// TIA Portal V20 export
// export: Created 2025-12-01T14:57:29.98862Z, ExportSetting None, DisplayName Totally Integrated Automation Portal, DisplayVersion V20 Update 3, DisplayName TIA Portal Openness, DisplayVersion V20 Update 3, DisplayName TIA Portal Version Control Interface, DisplayVersion V20 Update 3, DisplayName STEP 7 Professional, DisplayVersion V20 Update 3, DisplayName STEP 7 Safety, DisplayVersion V20 Update 2, DisplayName WinCC Basic/Comfort/Advanced, DisplayVersion V20 Update 3, DisplayName WinCC Professional, DisplayVersion V20 Update 3, DisplayName WinCC Unified, DisplayVersion V20 Update 3
FUNCTION_BLOCK "FB265_M_TL_E01234_S01234"   // FB265, LAD
TITLE = Control del Ramal de Salidas
{ S7_Optimized_Access := 'FALSE' }
AUTHOR : TE_FSS
NAME : 20170822
VERSION : 3.7
// stored: AutoNumber false, SetENOAutomatically false
   VAR_INPUT
      Mesa : UInt;   // Mesa de la FB
      Error_Tx : Bool;   // Error en el Tx
      EnTension : Bool;   // Existe Tension en la Mesa
      Termico_E1_Tx : Bool;   // Proteccion del Tx en E1E3
      Termico_E2_Tx : Bool;   // Proteccion del Tx en E2E4
      pHsMx_Carretilla : Bool;   // pHs de Carretilla
      pHsMx_1 : Bool;   // pHs de la Mesa Mesa (Para Entrada por E3,E2)
      pHsMx_2 : Bool;   // pHs de la Mesa Mesa (Para Entrada por E1,E4)
      pHsMx_Seg_1 : Bool;   // pHs de Protrusion de la Mesa. Nota: No existe >> ON
      pHsMx_Seg_2 : Bool;   // pHs de Protrusion de la Mesa. Nota: No existe >> ON
      Avance_E1_Tx_Ok : Bool;   // Avance del Tx en E1E3
      Avance_E2_Tx_Ok : Bool;   // Avance del Tx en E2E4
      PosTR_E1 : Bool;   // Posicion del TR en E1E3
      PosTR_E2 : Bool;   // Posicion del TR en E2E4
      EnMovimiento_TR : Bool;   // En movimiento el TR
      TP1_UP : Bool;   // TP1 Arriba. Nota Movimiento E1 >> S3
      TP1_DW : Bool;   // TP1 Abajo. Nota Movimiento E1 >> S3
      EnMovimiento_TP1 { ExternalVisible := 'False'} : Bool;   // En movimiento el TP1
      TP2_UP : Bool;   // TP2 Arriba. Nota Movimiento E2 >> S4
      TP2_DW : Bool;   // TP2 Abajo. Nota Movimiento E2 >> S4
      EnMovimiento_TP2 : Bool;   // En movimiento el TP2
      DescargaAct_Ent_M1 : Bool;   // E1 >> Mesa Anterior DescargaAct
      AVTF_Ent_M1 : Bool;   // E1 >> Mesa Anterior AVTF
      P_Mens_Ent_M1 : Bool;   // E1 >> Mesa Anterior P_Mens
      DescargaAct_Ent_M2 : Bool;   // E2 >> Mesa Anterior DescargaAct
      AVTF_Ent_M2 : Bool;   // E2 >> Mesa Anterior AVTF
      P_Mens_Ent_M2 : Bool;   // E2 >> Mesa Anterior P_Mens
      DescargaAct_Ent_M3 : Bool;   // E3 >> Mesa Anterior DescargaAct
      AVTF_Ent_M3 : Bool;   // E3 >> Mesa Anterior AVTF
      P_Mens_Ent_M3 : Bool;   // E3 >> Mesa Anterior P_Mens
      DescargaAct_Ent_M4 : Bool;   // E4 >> Mesa Anterior DescargaAct
      AVTF_Ent_M4 : Bool;   // E4 >> Mesa Anterior AVTF
      P_Mens_Ent_M4 : Bool;   // E4 >> Mesa Anterior P_Mens
      PTF_Sal_M1 : Bool;   // S1 >> Mesa Siguiente PTF
      FTF_Sal_M1 : Bool;   // S1 >> Mesa Siguiente FTF
      PTF_Sal_M2 : Bool;   // S2 >> Mesa Siguiente PTF
      FTF_Sal_M2 : Bool;   // S2 >> Mesa Siguiente FTF
      PTF_Sal_M3 : Bool;   // S3 >> Mesa Siguiente PTF
      FTF_Sal_M3 : Bool;   // S3 >> Mesa Siguiente FTF
      PTF_Sal_M4 : Bool;   // S4 >> Mesa Siguiente PTF
      FTF_Sal_M4 : Bool;   // S4 >> Mesa Siguiente FTF
      MSig_CargaAct_Sal_M1 : Bool;   // S1 >> Mesa Siguiente En Carga
      MSig_CargaAct_Sal_M2 : Bool;   // S2 >> Mesa Siguiente En Carga
      MSig_CargaAct_Sal_M3 : Bool;   // S3 >> Mesa Siguiente En Carga
      MSig_CargaAct_Sal_M4 : Bool;   // S4 >> Mesa Siguiente En Carga
      PosTR_EnReposo_E2 : Bool;   // Posicion de Reposo en E2 para el Transfer
      PosTR_EnReposo_E1 : Bool;   // Posicion de Reposo en E1 para el Transfer
      PermisoMov_PosTR_E2 : Bool;   // Permiso de Mover el Trasnfer hacia E2
      PermisoMov_PosTR_E1 : Bool;   // Permiso de Mover el Trasnfer hacia E1
      Mx_Centraje : Bool;   // Config >> Activar Centraje de Carga
      Mx_UP_E1E3 : Bool;   // Config >> TR Arriba en E1E3
      Mx_TRElectrico : Bool;   // Config >> Mesa con Transfer Electrico
      Mx_VelocidadLenta_In : Bool;   // Forzar a Velociada Lenta
      F_EnvMens_Mx : Bool;   // Fin de Envio de Mensaje
      OrdSal_M1 : Bool;   // Orden de Salida por S1
      OrdSal_M2 : Bool;   // Orden de Salida por S2
      OrdSal_M3 : Bool;   // Orden de Salida por S3
      OrdSal_M4 : Bool;   // Orden de Salida por S4
      OrdSal_Retirar : Bool;   // Orden de Salida por S0
      BloqueoActivo_OK : Bool;   // Bloqueo Activo de la Mesa
      V_CNT_pHsMx_E1 : Int := 400;   // Valor de Presencia
      V_CNT_pHsMx_FTF_E1 : Int := 200;   // Valor para activar FTF. Nota: < = V_CNT_pHsMx.
      V_CNTSeg_pHsMx_E1 : Int := 2000;   // Valor de Seguriadad para Presencia
      V_CNT_pHsMx_E2 : Int := 400;   // Valor de Presencia
      V_CNT_pHsMx_FTF_E2 : Int := 200;   // Valor para activar FTF. Nota: < = V_CNT_pHsMx.
      V_CNTSeg_pHsMx_E2 : Int := 2000;   // Valor de Seguriadad para Presencia
      V_Subir_TP_Min : Int := 20;   // Valor Minimo para Subir Tope
      V_Bajar_TP_Max : Int := 40;   // Valor Maximo para Bajar Tope
      V_CNT_ApHsMx : Int := 500;   // Valor de Ausencia
      V_CNTSeg_ApHsMx : Int := 2000;   // Valor de Seguriadad para Ausencia
      V_TIM_Bloqueo : Int := 3000;   // Valor del Tiempo de Espera para Bloqueo
      V_TIM_Entrada : Int := 5000;   // Valor de Entrada de Carga >> E0
      V_TIM_Retirar : Int := 5000;   // Valor de Retirada de Carga >> S0
      V_CNT_Centrado : Int := 2000;   // Valor de Centrado de Carga
      V_CNT_Reposo : Int := 500;   // Valor de Reposo de Carga Nota: > Centrado
      V_CNT_Simultaneo : Int := 2000;   // Valor de Simultaneo
      V_InicioSimultaneo : Int := 0;   // Inicio de Simultaneo. Nota: <= V_CNT_Simultaneo
      V_FinSimultaneo : Int := 0;   // Final de Simultaneo. Nota: <= V_InicioSimultaneo
      V_TOut_Tx_Mx_E1 : Int := 10000;   // TimeOut de Entrada por E1
      V_TOut_Tx_Mx_E2 : Int := 10000;   // TimeOut de Entrada por E2
      V_TOut_TR : Int := 5000;   // TimeOut de Transfer
      V_TOut_TP : Int := 5000;   // TimeOut de Tope
      V_TMP_Protrusion : Int := 200;   // TMP de Protrusion
      V_CNT_PerdidapHs : Int := 10;   // CNT de Perdida de pHs
   END_VAR
   VAR_OUTPUT
      P_EnvMens_PMx : Bool;   // Permiso de Enviar Mensaje de Presencia
      P_EnvMens_PBM : Bool;   // Permiso de Enviar Mensaje de Bloqueo
      P_EnvMens_AMx : Bool;   // Permiso de Enviar Mensaje de Ausencia
      P_RecepOK_Mx : Bool;   // Recepcion OK
      PTF_Ent_M1 : Bool;   // E1 >> Mesa Anterior PTF
      FTF_Ent_M1 : Bool;   // E1 >> Mesa Anterior FTF
      PTF_Ent_M2 : Bool;   // E2 >> Mesa Anterior PTF
      FTF_Ent_M2 : Bool;   // E2 >> Mesa Anterior FTF
      PTF_Ent_M3 : Bool;   // E3 >> Mesa Anterior PTF
      FTF_Ent_M3 : Bool;   // E3 >> Mesa Anterior FTF
      PTF_Ent_M4 : Bool;   // E4 >> Mesa Anterior PTF
      FTF_Ent_M4 : Bool;   // E4 >> Mesa Anterior FTF
      AVTF_Sal_M1 : Bool;   // S1 >> Mesa Siguiente AVTF
      P_Mens_Sal_M1 : Bool;   // S1 >> Mesa Siguiente P_Mens
      AVTF_Sal_M2 : Bool;   // S2 >> Mesa Siguiente AVTF
      P_Mens_Sal_M2 : Bool;   // S2 >> Mesa Siguiente P_Mens
      AVTF_Sal_M3 : Bool;   // S3 >> Mesa Siguiente AVTF
      P_Mens_Sal_M3 : Bool;   // S3 >> Mesa Siguiente P_Mens
      AVTF_Sal_M4 : Bool;   // S4 >> Mesa Siguiente AVTF
      P_Mens_Sal_M4 : Bool;   // S4 >> Mesa Siguiente P_Mens
   END_VAR
   VAR
      Anular_prE1 : Bool;   // ???
      Anular_prS3 : Bool;   // ???
      Mx_ET00 : Bool;
      Mx_ET01 : Bool;
      Mx_ET02 : Bool;
      Mx_ET08 : Bool;
      Mx_ET09 : Bool;
      Mx_ET10 : Bool;
      Mx_ET11 : Bool;
      Mx_ET12 : Bool;
      Mx_ET110 : Bool;
      Mx_ET111 : Bool;
      Mx_ET20 : Bool;
      Mx_ET21 : Bool;
      Mx_ET22 : Bool;
      Mx_ET120 : Bool;
      Mx_ET121 : Bool;
      Mx_ET40 : Bool;
      Mx_ET41 : Bool;
      Mx_ET42 : Bool;
      Mx_ET43 : Bool;
      Mx_ET140 : Bool;
      Mx_ET141 : Bool;
      Mx_ET50 : Bool;
      Mx_ET51 : Bool;
      Mx_ET150 : Bool;
      Mx_ET151 : Bool;
      Mx_ET60 : Bool;
      Mx_ET61 : Bool;
      Mx_ET160 : Bool;
      Mx_ET161 : Bool;
      Mx_ET180 : Bool;
      Mx_ET181 : Bool;
      Mx_ET90 : Bool;
      Mx_ET91 : Bool;
      Mx_ET190 : Bool;
      Mx_ET191 : Bool;
      Mx_ET192 : Bool;
      Selec_M1_Entrada : Bool;   // Seleccionado Entrada por E1
      Selec_M1_Salida : Bool;   // Seleccionado Entrada por E2
      Selec_M2_Entrada : Bool;   // Seleccionado Entrada por E3
      Selec_M2_Salida : Bool;   // Seleccionado Entrada por E4
      Selec_M3_Entrada : Bool;   // Seleccionado Salida por S1
      Selec_M3_Salida : Bool;   // Seleccionado Salida por S2
      Selec_M4_Entrada : Bool;   // Seleccionado Salida por S3
      Selec_M4_Salida : Bool;   // Seleccionado Salida por S4
      Selec_Retirar : Bool;   // Seleccionado Retirar
      MEnt_DescargaAct : Bool;   // Interlock >> DesCargaAct de MAnt >> Mx
      ATF_MEnt : Bool;   // Interlock >> AVTF de MAnt >> Mx
      P_Mens_MEnt : Bool;   // Interlock >> P_Mens de MAnt >> Mx
      PTF_MEnt : Bool;   // Interlock >> PTF de MAnt >> Mx
      FTF_MEnt : Bool;   // Interlock >> FTF de MAnt >> Mx
      ATF_MSal : Bool;   // Interlock >> AVTF de Mx >> MSig
      P_Mens_MSal { ExternalAccessible := 'False'; ExternalVisible := 'False'; ExternalWritable := 'False'} : Bool;   // Interlock >> P_Mens de Mx >> MSig
      PTF_MSal : Bool;   // Interlock >> PTF de Mx >> MSig
      FTF_MSal : Bool;   // Interlock >> FTF de Mx >> MSig
      ProtocoloIniciado_Mx : Bool;   // Iniciado el Envio del Mensaje de Presencia
      Simultaneo_Mx : Bool;   // Activo Simultaneo E1E2E3E4
      SaliendoCarga : Bool;   // Saliendo Carga de la Mesa
      CNT_pHsMx_FTF_OK_E1E3 : Bool;   // Enviar ya FTF
      CNT_pHsMx_FTF_OK_E2E4 : Bool;   // Enviar ya FTF
      CNT_pHsMx_E1E3 { S7_SetPoint := 'True'} : "FB910_CNT_UHS";   // CNT de la Presencia
      CNTSeg_pHsMx_E1E3 { S7_SetPoint := 'True'} : "FB910_CNT_UHS";   // CNT de Seguridad de la Presencia
      CNT_pHsMx_E2E4 { S7_SetPoint := 'True'} : "FB910_CNT_UHS";   // CNT de la Presencia
      CNTSeg_pHsMx_E2E4 { S7_SetPoint := 'True'} : "FB910_CNT_UHS";   // CNT de Seguridad de la Presencia
      CNT_ApHsMx { S7_SetPoint := 'True'} : "FB910_CNT_UHS";   // CNT de la Ausencia
      CNTSeg_ApHsMx { S7_SetPoint := 'True'} : "FB910_CNT_UHS";   // CNT de Seguridad de la Ausencia
      TIM_Bloqueo { S7_SetPoint := 'True'} : "FB910_CNT_UHS";   // TIM de Espera para Bloqueo
      TMP_Entrada { S7_SetPoint := 'True'} : "FB910_CNT_UHS";   // TMP de Entrada de Carga
      TMP_Retirar { S7_SetPoint := 'True'} : "FB910_CNT_UHS";   // TMP de Retirada de Carga
      CNT_Centrado { S7_SetPoint := 'True'} : "FB910_CNT_UHS";   // Contador de Centrado de Carga
      CNT_Simultaneo { S7_SetPoint := 'True'} : "FB910_CNT_UHS";   // CNT de Simultaneo
      TMP_EnTension { S7_SetPoint := 'True'} : "FB910_CNT_UHS";
      TOut_Av_Mx_E1E3 { S7_SetPoint := 'True'} : "FB910_CNT_UHS";   // Time Out de Entrada de E1
      TOut_Ret_Mx_E1E3 { S7_SetPoint := 'True'} : "FB910_CNT_UHS";   // Time Out de Entrada de E3
      TOut_Av_Mx_E2E4 { S7_SetPoint := 'True'} : "FB910_CNT_UHS";   // Time Out de Entrada de E2
      TOut_Ret_Mx_E2E4 { S7_SetPoint := 'True'} : "FB910_CNT_UHS";   // Time Out de Entrada de E4
      TOut_Subir_TR { S7_SetPoint := 'True'} : "FB910_CNT_UHS";   // Time Out de Subida del TR
      TOut_Bajar_TR { S7_SetPoint := 'True'} : "FB910_CNT_UHS";   // Time Out de Bajada del TR
      TOut_Subir_Tp { S7_SetPoint := 'True'} : "FB910_CNT_UHS";   // Time Out de Subida del TP
      TOut_Bajar_Tp { S7_SetPoint := 'True'} : "FB910_CNT_UHS";   // Time Out de Bajada del TP
      TMP_Protrusion { S7_SetPoint := 'True'} : "FB910_CNT_UHS";   // TMP de la Protrusion
      CNT_PerdidapHs { S7_SetPoint := 'True'} : "FB910_CNT_UHS";   // CNT de Perdida de pHs
      STAT_EnvMens_PMx : Bool;   // Interna >> Envio del Mensaje de Presencia
      STAT_EnvMens_AMx : Bool;   // Interna >> Envio del Mensaje de Ausencia
      STAT_EnvMens_PBMx : Bool;   // Interna >> Envio del Mensaje de Bloqueo
   END_VAR
   VAR_TEMP
      EstadoZona : "EstadoZona";   // Estado de Zona de la Mesa
      EstadoVI : "EstadosMesa";   // Estado del Vehiculo Inteliguente de la Mesa
      ConfigFB : "UDT_ConfigFB";   // Configuracion de la FB de la Mesa
      V_Protrusion : Int;
      Aux_ET00 : Bool;
      Pos_TR_OK : Bool;
      OK_TP1_DW : Bool;
      OK_TP2_DW : Bool;
   END_VAR
   VAR_TEMP   // added for the SCL form of the ladder/FBD networks
      _w1 : Bool;
      _w2 : Bool;
      _w3 : Bool;
      _w4 : Bool;
   END_VAR
BEGIN

REGION Network 1: INICIALIZAR - Recoger las Variables de Estado de la Mesa
   // Se recoge - Estado_CBx
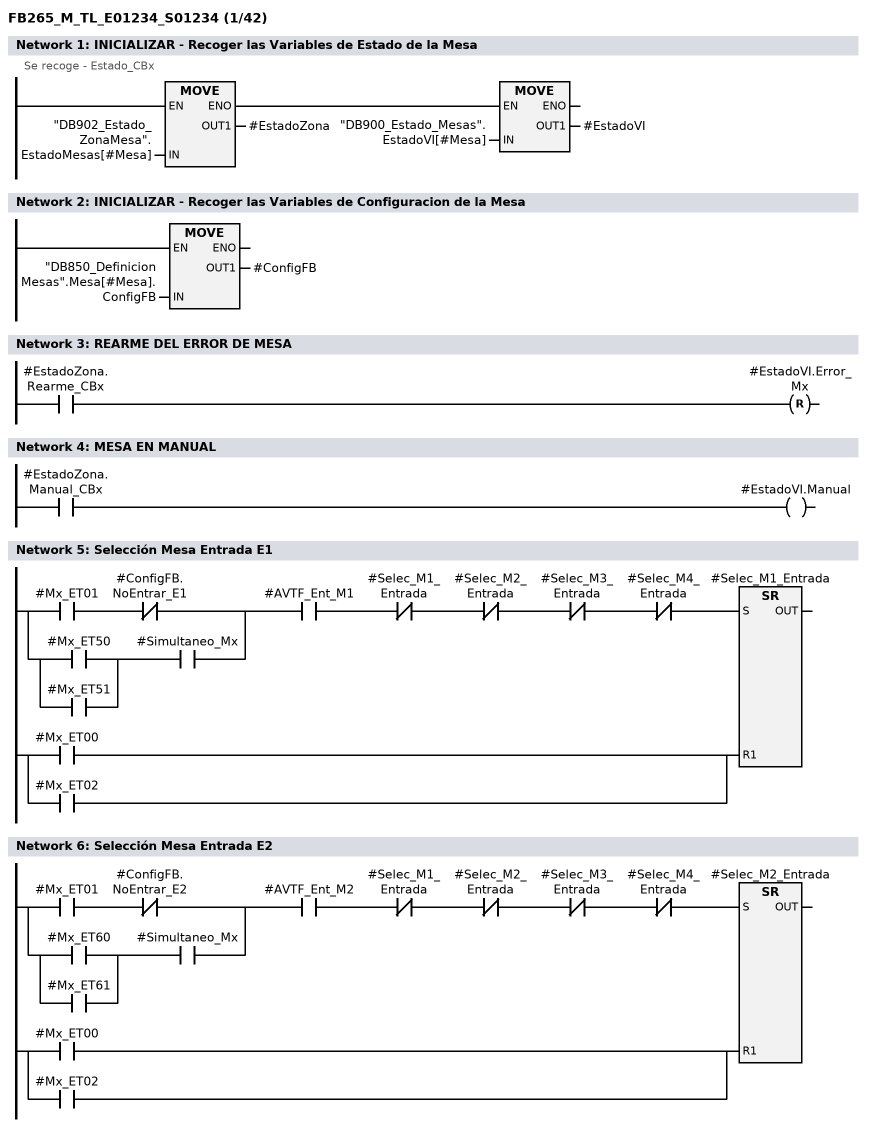
   RUNG wire#powerrail
      Move(in := "DB902_Estado_ZonaMesa".EstadoMesas[#Mesa], out1 => #EstadoZona)
      Move(in := "DB900_Estado_Mesas".EstadoVI[#Mesa], out1 => #EstadoVI)
   END_RUNG
   // the same network as SCL:
   #EstadoZona := "DB902_Estado_ZonaMesa".EstadoMesas[#Mesa];
   #EstadoVI := "DB900_Estado_Mesas".EstadoVI[#Mesa];
END_REGION

REGION Network 2: INICIALIZAR - Recoger las Variables de Configuracion de la Mesa
   RUNG wire#powerrail
      Move(in := "DB850_DefinicionMesas".Mesa[#Mesa].ConfigFB, out1 => #ConfigFB)
   END_RUNG
   // the same network as SCL:
   #ConfigFB := "DB850_DefinicionMesas".Mesa[#Mesa].ConfigFB;
END_REGION

REGION Network 3: REARME DEL ERROR DE MESA
   RUNG wire#powerrail
      Contact( #EstadoZona.Rearme_CBx )
      R_Coil( #EstadoVI.Error_Mx )
   END_RUNG
   // the same network as SCL:
   IF #EstadoZona.Rearme_CBx THEN #EstadoVI.Error_Mx := FALSE; END_IF;
END_REGION

REGION Network 4: MESA EN MANUAL
   RUNG wire#powerrail
      Contact( #EstadoZona.Manual_CBx )
      Coil( #EstadoVI.Manual )
   END_RUNG
   // the same network as SCL:
   #EstadoVI.Manual := #EstadoZona.Manual_CBx;
END_REGION

REGION Network 5: Selección Mesa Entrada E1
   RUNG wire#powerrail
      Contact( #Mx_ET01 )
      I_Contact( #ConfigFB.NoEntrar_E1 )
      wire#w1
      Contact( #AVTF_Ent_M1 )
      I_Contact( #Selec_M1_Entrada )
      I_Contact( #Selec_M2_Entrada )
      I_Contact( #Selec_M3_Entrada )
      I_Contact( #Selec_M4_Entrada )
      S_SR(operand := #Selec_M1_Entrada, r1 := wire#w3)
   END_RUNG
   RUNG wire#powerrail
      Contact( #Mx_ET50 )
      wire#w2
      Contact( #Simultaneo_Mx )
   END_RUNG wire#w1
   RUNG wire#powerrail
      Contact( #Mx_ET51 )
   END_RUNG wire#w2
   RUNG wire#powerrail
      Contact( #Mx_ET00 )
   END_RUNG wire#w3
   RUNG wire#powerrail
      Contact( #Mx_ET02 )
   END_RUNG wire#w3
   // the same network as SCL:
   IF ((#Mx_ET01 AND NOT #ConfigFB.NoEntrar_E1) OR ((#Mx_ET50 OR #Mx_ET51) AND #Simultaneo_Mx)) AND #AVTF_Ent_M1 AND NOT #Selec_M1_Entrada AND NOT #Selec_M2_Entrada AND NOT #Selec_M3_Entrada AND NOT #Selec_M4_Entrada THEN
       #Selec_M1_Entrada := TRUE;   // SR flip-flop
   END_IF;
   IF #Mx_ET00 OR #Mx_ET02 THEN #Selec_M1_Entrada := FALSE; END_IF;
END_REGION

REGION Network 6: Selección Mesa Entrada E2
   RUNG wire#powerrail
      Contact( #Mx_ET01 )
      I_Contact( #ConfigFB.NoEntrar_E2 )
      wire#w1
      Contact( #AVTF_Ent_M2 )
      I_Contact( #Selec_M1_Entrada )
      I_Contact( #Selec_M2_Entrada )
      I_Contact( #Selec_M3_Entrada )
      I_Contact( #Selec_M4_Entrada )
      S_SR(operand := #Selec_M2_Entrada, r1 := wire#w3)
   END_RUNG
   RUNG wire#powerrail
      Contact( #Mx_ET60 )
      wire#w2
      Contact( #Simultaneo_Mx )
   END_RUNG wire#w1
   RUNG wire#powerrail
      Contact( #Mx_ET61 )
   END_RUNG wire#w2
   RUNG wire#powerrail
      Contact( #Mx_ET00 )
   END_RUNG wire#w3
   RUNG wire#powerrail
      Contact( #Mx_ET02 )
   END_RUNG wire#w3
   // the same network as SCL:
   IF ((#Mx_ET01 AND NOT #ConfigFB.NoEntrar_E2) OR ((#Mx_ET60 OR #Mx_ET61) AND #Simultaneo_Mx)) AND #AVTF_Ent_M2 AND NOT #Selec_M1_Entrada AND NOT #Selec_M2_Entrada AND NOT #Selec_M3_Entrada AND NOT #Selec_M4_Entrada THEN
       #Selec_M2_Entrada := TRUE;   // SR flip-flop
   END_IF;
   IF #Mx_ET00 OR #Mx_ET02 THEN #Selec_M2_Entrada := FALSE; END_IF;
END_REGION

REGION Network 7: Selección Mesa Entrada E3
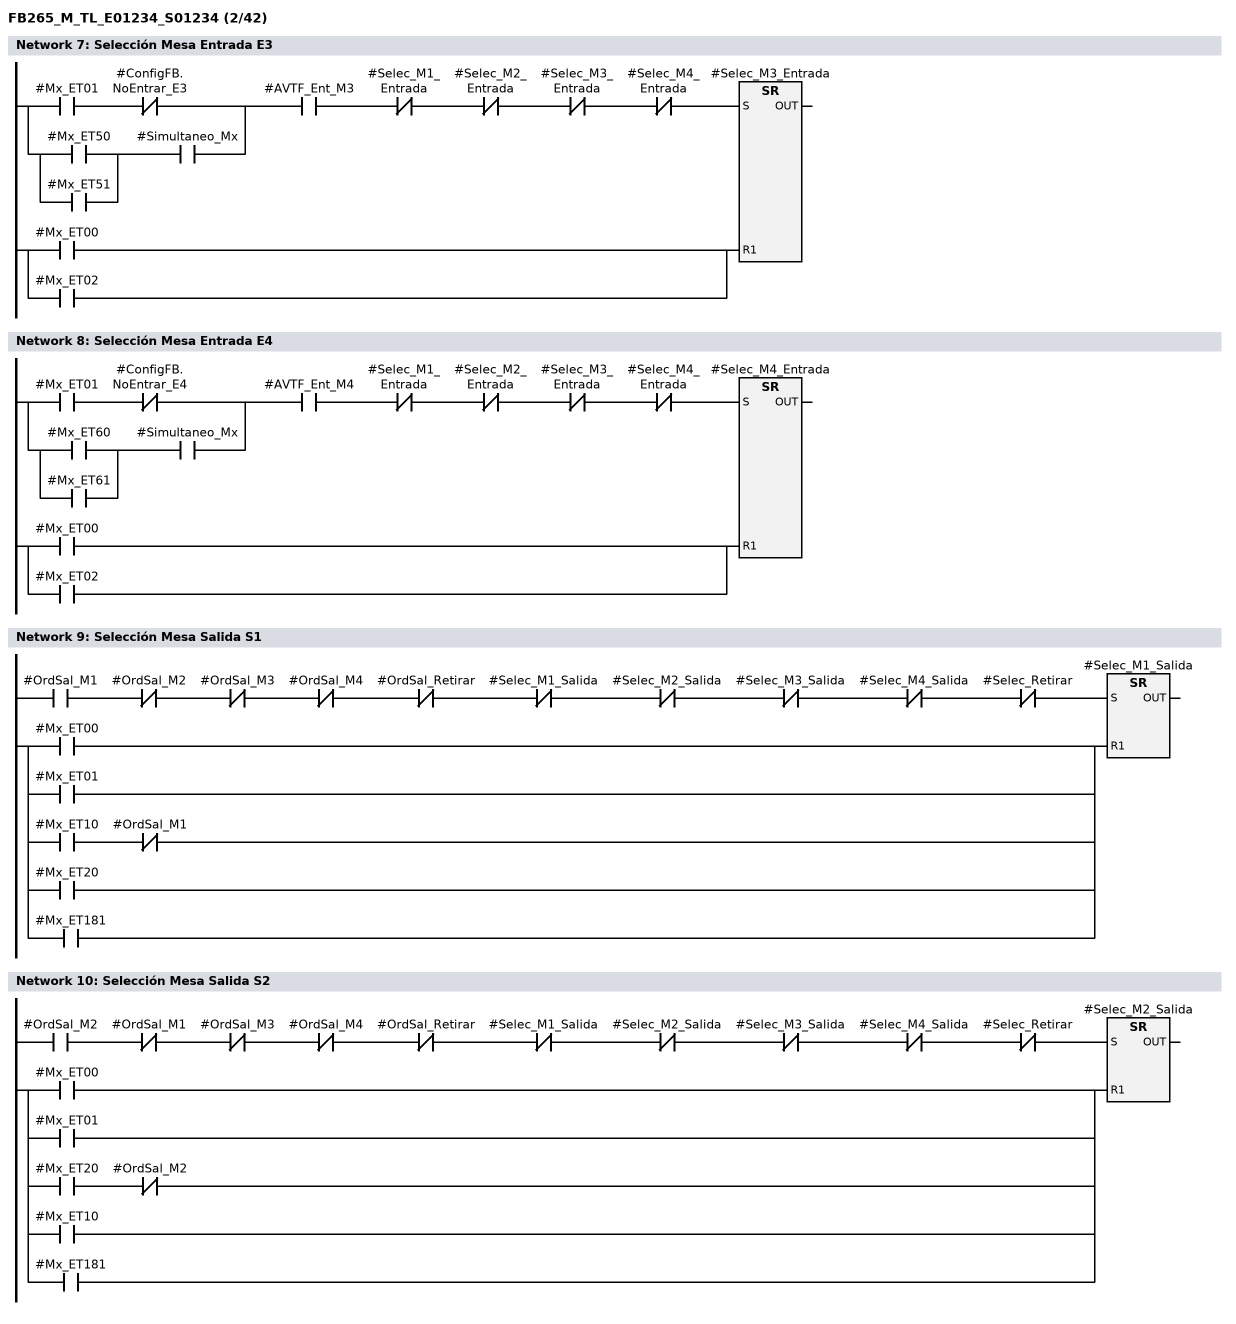
   RUNG wire#powerrail
      Contact( #Mx_ET01 )
      I_Contact( #ConfigFB.NoEntrar_E3 )
      wire#w1
      Contact( #AVTF_Ent_M3 )
      I_Contact( #Selec_M1_Entrada )
      I_Contact( #Selec_M2_Entrada )
      I_Contact( #Selec_M3_Entrada )
      I_Contact( #Selec_M4_Entrada )
      S_SR(operand := #Selec_M3_Entrada, r1 := wire#w3)
   END_RUNG
   RUNG wire#powerrail
      Contact( #Mx_ET50 )
      wire#w2
      Contact( #Simultaneo_Mx )
   END_RUNG wire#w1
   RUNG wire#powerrail
      Contact( #Mx_ET51 )
   END_RUNG wire#w2
   RUNG wire#powerrail
      Contact( #Mx_ET00 )
   END_RUNG wire#w3
   RUNG wire#powerrail
      Contact( #Mx_ET02 )
   END_RUNG wire#w3
   // the same network as SCL:
   IF ((#Mx_ET01 AND NOT #ConfigFB.NoEntrar_E3) OR ((#Mx_ET50 OR #Mx_ET51) AND #Simultaneo_Mx)) AND #AVTF_Ent_M3 AND NOT #Selec_M1_Entrada AND NOT #Selec_M2_Entrada AND NOT #Selec_M3_Entrada AND NOT #Selec_M4_Entrada THEN
       #Selec_M3_Entrada := TRUE;   // SR flip-flop
   END_IF;
   IF #Mx_ET00 OR #Mx_ET02 THEN #Selec_M3_Entrada := FALSE; END_IF;
END_REGION

REGION Network 8: Selección Mesa Entrada E4
   RUNG wire#powerrail
      Contact( #Mx_ET01 )
      I_Contact( #ConfigFB.NoEntrar_E4 )
      wire#w1
      Contact( #AVTF_Ent_M4 )
      I_Contact( #Selec_M1_Entrada )
      I_Contact( #Selec_M2_Entrada )
      I_Contact( #Selec_M3_Entrada )
      I_Contact( #Selec_M4_Entrada )
      S_SR(operand := #Selec_M4_Entrada, r1 := wire#w3)
   END_RUNG
   RUNG wire#powerrail
      Contact( #Mx_ET60 )
      wire#w2
      Contact( #Simultaneo_Mx )
   END_RUNG wire#w1
   RUNG wire#powerrail
      Contact( #Mx_ET61 )
   END_RUNG wire#w2
   RUNG wire#powerrail
      Contact( #Mx_ET00 )
   END_RUNG wire#w3
   RUNG wire#powerrail
      Contact( #Mx_ET02 )
   END_RUNG wire#w3
   // the same network as SCL:
   IF ((#Mx_ET01 AND NOT #ConfigFB.NoEntrar_E4) OR ((#Mx_ET60 OR #Mx_ET61) AND #Simultaneo_Mx)) AND #AVTF_Ent_M4 AND NOT #Selec_M1_Entrada AND NOT #Selec_M2_Entrada AND NOT #Selec_M3_Entrada AND NOT #Selec_M4_Entrada THEN
       #Selec_M4_Entrada := TRUE;   // SR flip-flop
   END_IF;
   IF #Mx_ET00 OR #Mx_ET02 THEN #Selec_M4_Entrada := FALSE; END_IF;
END_REGION

REGION Network 9: Selección Mesa Salida S1
   RUNG wire#powerrail
      Contact( #OrdSal_M1 )
      I_Contact( #OrdSal_M2 )
      I_Contact( #OrdSal_M3 )
      I_Contact( #OrdSal_M4 )
      I_Contact( #OrdSal_Retirar )
      I_Contact( #Selec_M1_Salida )
      I_Contact( #Selec_M2_Salida )
      I_Contact( #Selec_M3_Salida )
      I_Contact( #Selec_M4_Salida )
      I_Contact( #Selec_Retirar )
      S_SR(operand := #Selec_M1_Salida, r1 := wire#w1)
   END_RUNG
   RUNG wire#powerrail
      Contact( #Mx_ET00 )
   END_RUNG wire#w1
   RUNG wire#powerrail
      Contact( #Mx_ET01 )
   END_RUNG wire#w1
   RUNG wire#powerrail
      Contact( #Mx_ET10 )
      I_Contact( #OrdSal_M1 )
   END_RUNG wire#w1
   RUNG wire#powerrail
      Contact( #Mx_ET20 )
   END_RUNG wire#w1
   RUNG wire#powerrail
      Contact( #Mx_ET181 )
   END_RUNG wire#w1
   // the same network as SCL:
   IF #OrdSal_M1 AND NOT #OrdSal_M2 AND NOT #OrdSal_M3 AND NOT #OrdSal_M4 AND NOT #OrdSal_Retirar AND NOT #Selec_M1_Salida AND NOT #Selec_M2_Salida AND NOT #Selec_M3_Salida AND NOT #Selec_M4_Salida AND NOT #Selec_Retirar THEN
       #Selec_M1_Salida := TRUE;   // SR flip-flop
   END_IF;
   IF #Mx_ET00 OR #Mx_ET01 OR (#Mx_ET10 AND NOT #OrdSal_M1) OR #Mx_ET20 OR #Mx_ET181 THEN
       #Selec_M1_Salida := FALSE;
   END_IF;
END_REGION

REGION Network 10: Selección Mesa Salida S2
   RUNG wire#powerrail
      Contact( #OrdSal_M2 )
      I_Contact( #OrdSal_M1 )
      I_Contact( #OrdSal_M3 )
      I_Contact( #OrdSal_M4 )
      I_Contact( #OrdSal_Retirar )
      I_Contact( #Selec_M1_Salida )
      I_Contact( #Selec_M2_Salida )
      I_Contact( #Selec_M3_Salida )
      I_Contact( #Selec_M4_Salida )
      I_Contact( #Selec_Retirar )
      S_SR(operand := #Selec_M2_Salida, r1 := wire#w1)
   END_RUNG
   RUNG wire#powerrail
      Contact( #Mx_ET00 )
   END_RUNG wire#w1
   RUNG wire#powerrail
      Contact( #Mx_ET01 )
   END_RUNG wire#w1
   RUNG wire#powerrail
      Contact( #Mx_ET20 )
      I_Contact( #OrdSal_M2 )
   END_RUNG wire#w1
   RUNG wire#powerrail
      Contact( #Mx_ET10 )
   END_RUNG wire#w1
   RUNG wire#powerrail
      Contact( #Mx_ET181 )
   END_RUNG wire#w1
   // the same network as SCL:
   IF #OrdSal_M2 AND NOT #OrdSal_M1 AND NOT #OrdSal_M3 AND NOT #OrdSal_M4 AND NOT #OrdSal_Retirar AND NOT #Selec_M1_Salida AND NOT #Selec_M2_Salida AND NOT #Selec_M3_Salida AND NOT #Selec_M4_Salida AND NOT #Selec_Retirar THEN
       #Selec_M2_Salida := TRUE;   // SR flip-flop
   END_IF;
   IF #Mx_ET00 OR #Mx_ET01 OR (#Mx_ET20 AND NOT #OrdSal_M2) OR #Mx_ET10 OR #Mx_ET181 THEN
       #Selec_M2_Salida := FALSE;
   END_IF;
END_REGION

REGION Network 11: Selección Mesa Salida S3
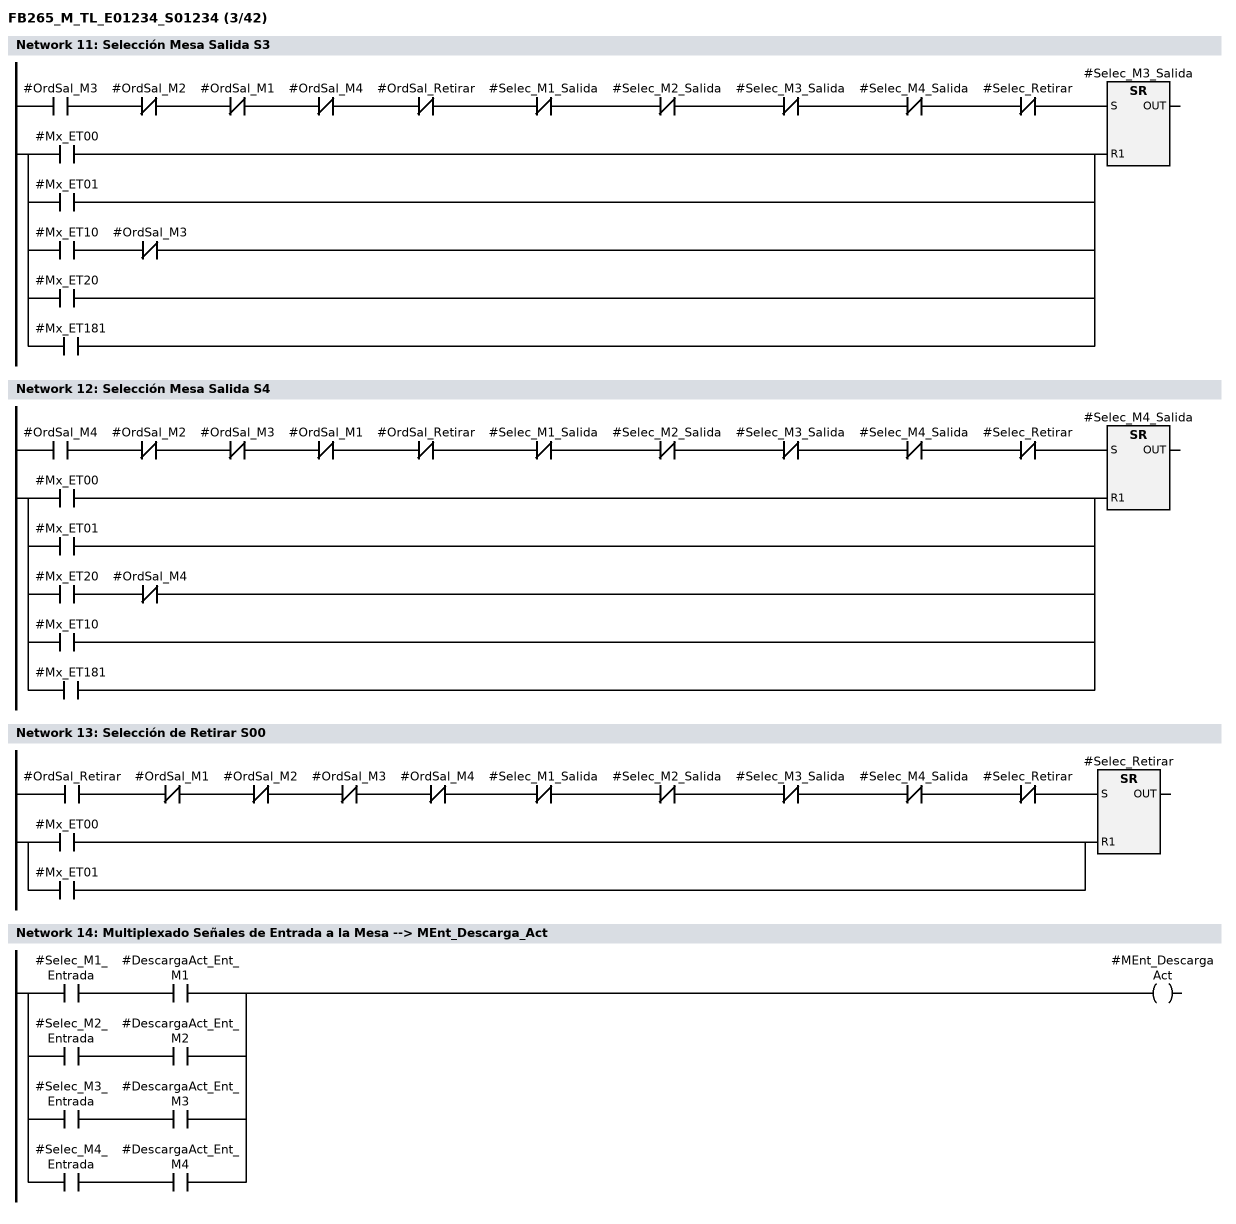
   RUNG wire#powerrail
      Contact( #OrdSal_M3 )
      I_Contact( #OrdSal_M2 )
      I_Contact( #OrdSal_M1 )
      I_Contact( #OrdSal_M4 )
      I_Contact( #OrdSal_Retirar )
      I_Contact( #Selec_M1_Salida )
      I_Contact( #Selec_M2_Salida )
      I_Contact( #Selec_M3_Salida )
      I_Contact( #Selec_M4_Salida )
      I_Contact( #Selec_Retirar )
      S_SR(operand := #Selec_M3_Salida, r1 := wire#w1)
   END_RUNG
   RUNG wire#powerrail
      Contact( #Mx_ET00 )
   END_RUNG wire#w1
   RUNG wire#powerrail
      Contact( #Mx_ET01 )
   END_RUNG wire#w1
   RUNG wire#powerrail
      Contact( #Mx_ET10 )
      I_Contact( #OrdSal_M3 )
   END_RUNG wire#w1
   RUNG wire#powerrail
      Contact( #Mx_ET20 )
   END_RUNG wire#w1
   RUNG wire#powerrail
      Contact( #Mx_ET181 )
   END_RUNG wire#w1
   // the same network as SCL:
   IF #OrdSal_M3 AND NOT #OrdSal_M2 AND NOT #OrdSal_M1 AND NOT #OrdSal_M4 AND NOT #OrdSal_Retirar AND NOT #Selec_M1_Salida AND NOT #Selec_M2_Salida AND NOT #Selec_M3_Salida AND NOT #Selec_M4_Salida AND NOT #Selec_Retirar THEN
       #Selec_M3_Salida := TRUE;   // SR flip-flop
   END_IF;
   IF #Mx_ET00 OR #Mx_ET01 OR (#Mx_ET10 AND NOT #OrdSal_M3) OR #Mx_ET20 OR #Mx_ET181 THEN
       #Selec_M3_Salida := FALSE;
   END_IF;
END_REGION

REGION Network 12: Selección Mesa Salida S4
   RUNG wire#powerrail
      Contact( #OrdSal_M4 )
      I_Contact( #OrdSal_M2 )
      I_Contact( #OrdSal_M3 )
      I_Contact( #OrdSal_M1 )
      I_Contact( #OrdSal_Retirar )
      I_Contact( #Selec_M1_Salida )
      I_Contact( #Selec_M2_Salida )
      I_Contact( #Selec_M3_Salida )
      I_Contact( #Selec_M4_Salida )
      I_Contact( #Selec_Retirar )
      S_SR(operand := #Selec_M4_Salida, r1 := wire#w1)
   END_RUNG
   RUNG wire#powerrail
      Contact( #Mx_ET00 )
   END_RUNG wire#w1
   RUNG wire#powerrail
      Contact( #Mx_ET01 )
   END_RUNG wire#w1
   RUNG wire#powerrail
      Contact( #Mx_ET20 )
      I_Contact( #OrdSal_M4 )
   END_RUNG wire#w1
   RUNG wire#powerrail
      Contact( #Mx_ET10 )
   END_RUNG wire#w1
   RUNG wire#powerrail
      Contact( #Mx_ET181 )
   END_RUNG wire#w1
   // the same network as SCL:
   IF #OrdSal_M4 AND NOT #OrdSal_M2 AND NOT #OrdSal_M3 AND NOT #OrdSal_M1 AND NOT #OrdSal_Retirar AND NOT #Selec_M1_Salida AND NOT #Selec_M2_Salida AND NOT #Selec_M3_Salida AND NOT #Selec_M4_Salida AND NOT #Selec_Retirar THEN
       #Selec_M4_Salida := TRUE;   // SR flip-flop
   END_IF;
   IF #Mx_ET00 OR #Mx_ET01 OR (#Mx_ET20 AND NOT #OrdSal_M4) OR #Mx_ET10 OR #Mx_ET181 THEN
       #Selec_M4_Salida := FALSE;
   END_IF;
END_REGION

REGION Network 13: Selección de Retirar S00
   RUNG wire#powerrail
      Contact( #OrdSal_Retirar )
      I_Contact( #OrdSal_M1 )
      I_Contact( #OrdSal_M2 )
      I_Contact( #OrdSal_M3 )
      I_Contact( #OrdSal_M4 )
      I_Contact( #Selec_M1_Salida )
      I_Contact( #Selec_M2_Salida )
      I_Contact( #Selec_M3_Salida )
      I_Contact( #Selec_M4_Salida )
      I_Contact( #Selec_Retirar )
      S_SR(operand := #Selec_Retirar, r1 := wire#w1)
   END_RUNG
   RUNG wire#powerrail
      Contact( #Mx_ET00 )
   END_RUNG wire#w1
   RUNG wire#powerrail
      Contact( #Mx_ET01 )
   END_RUNG wire#w1
   // the same network as SCL:
   IF #OrdSal_Retirar AND NOT #OrdSal_M1 AND NOT #OrdSal_M2 AND NOT #OrdSal_M3 AND NOT #OrdSal_M4 AND NOT #Selec_M1_Salida AND NOT #Selec_M2_Salida AND NOT #Selec_M3_Salida AND NOT #Selec_M4_Salida AND NOT #Selec_Retirar THEN
       #Selec_Retirar := TRUE;   // SR flip-flop
   END_IF;
   IF #Mx_ET00 OR #Mx_ET01 THEN #Selec_Retirar := FALSE; END_IF;
END_REGION

REGION Network 14: Multiplexado Señales de Entrada a la Mesa --> MEnt_Descarga_Act
   RUNG wire#powerrail
      Contact( #Selec_M1_Entrada )
      Contact( #DescargaAct_Ent_M1 )
      wire#w1
      Coil( #MEnt_DescargaAct )
   END_RUNG
   RUNG wire#powerrail
      Contact( #Selec_M2_Entrada )
      Contact( #DescargaAct_Ent_M2 )
   END_RUNG wire#w1
   RUNG wire#powerrail
      Contact( #Selec_M3_Entrada )
      Contact( #DescargaAct_Ent_M3 )
   END_RUNG wire#w1
   RUNG wire#powerrail
      Contact( #Selec_M4_Entrada )
      Contact( #DescargaAct_Ent_M4 )
   END_RUNG wire#w1
   // the same network as SCL:
   #MEnt_DescargaAct := (#Selec_M1_Entrada AND #DescargaAct_Ent_M1) OR (#Selec_M2_Entrada AND #DescargaAct_Ent_M2) OR (#Selec_M3_Entrada AND #DescargaAct_Ent_M3) OR (#Selec_M4_Entrada AND #DescargaAct_Ent_M4);
END_REGION

REGION Network 15: Multiplexado Señales de Entrada a la Mesa --> AVTF
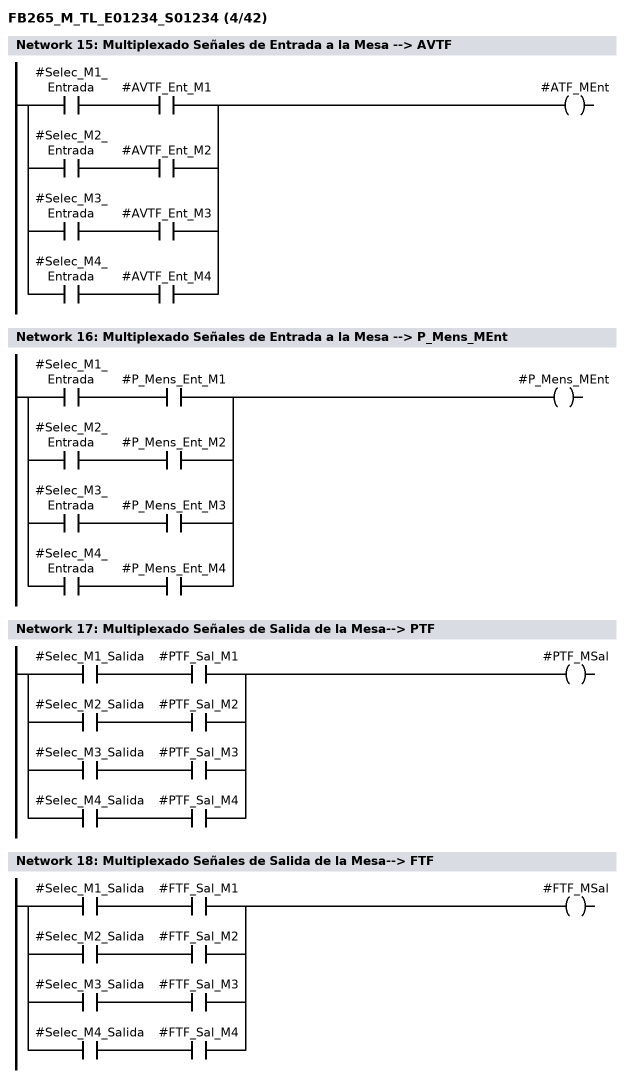
   RUNG wire#powerrail
      Contact( #Selec_M1_Entrada )
      Contact( #AVTF_Ent_M1 )
      wire#w1
      Coil( #ATF_MEnt )
   END_RUNG
   RUNG wire#powerrail
      Contact( #Selec_M2_Entrada )
      Contact( #AVTF_Ent_M2 )
   END_RUNG wire#w1
   RUNG wire#powerrail
      Contact( #Selec_M3_Entrada )
      Contact( #AVTF_Ent_M3 )
   END_RUNG wire#w1
   RUNG wire#powerrail
      Contact( #Selec_M4_Entrada )
      Contact( #AVTF_Ent_M4 )
   END_RUNG wire#w1
   // the same network as SCL:
   #ATF_MEnt := (#Selec_M1_Entrada AND #AVTF_Ent_M1) OR (#Selec_M2_Entrada AND #AVTF_Ent_M2) OR (#Selec_M3_Entrada AND #AVTF_Ent_M3) OR (#Selec_M4_Entrada AND #AVTF_Ent_M4);
END_REGION

REGION Network 16: Multiplexado Señales de Entrada a la Mesa --> P_Mens_MEnt
   RUNG wire#powerrail
      Contact( #Selec_M1_Entrada )
      Contact( #P_Mens_Ent_M1 )
      wire#w1
      Coil( #P_Mens_MEnt )
   END_RUNG
   RUNG wire#powerrail
      Contact( #Selec_M2_Entrada )
      Contact( #P_Mens_Ent_M2 )
   END_RUNG wire#w1
   RUNG wire#powerrail
      Contact( #Selec_M3_Entrada )
      Contact( #P_Mens_Ent_M3 )
   END_RUNG wire#w1
   RUNG wire#powerrail
      Contact( #Selec_M4_Entrada )
      Contact( #P_Mens_Ent_M4 )
   END_RUNG wire#w1
   // the same network as SCL:
   #P_Mens_MEnt := (#Selec_M1_Entrada AND #P_Mens_Ent_M1) OR (#Selec_M2_Entrada AND #P_Mens_Ent_M2) OR (#Selec_M3_Entrada AND #P_Mens_Ent_M3) OR (#Selec_M4_Entrada AND #P_Mens_Ent_M4);
END_REGION

REGION Network 17: Multiplexado Señales de Salida de la Mesa--> PTF
   RUNG wire#powerrail
      Contact( #Selec_M1_Salida )
      Contact( #PTF_Sal_M1 )
      wire#w1
      Coil( #PTF_MSal )
   END_RUNG
   RUNG wire#powerrail
      Contact( #Selec_M2_Salida )
      Contact( #PTF_Sal_M2 )
   END_RUNG wire#w1
   RUNG wire#powerrail
      Contact( #Selec_M3_Salida )
      Contact( #PTF_Sal_M3 )
   END_RUNG wire#w1
   RUNG wire#powerrail
      Contact( #Selec_M4_Salida )
      Contact( #PTF_Sal_M4 )
   END_RUNG wire#w1
   // the same network as SCL:
   #PTF_MSal := (#Selec_M1_Salida AND #PTF_Sal_M1) OR (#Selec_M2_Salida AND #PTF_Sal_M2) OR (#Selec_M3_Salida AND #PTF_Sal_M3) OR (#Selec_M4_Salida AND #PTF_Sal_M4);
END_REGION

REGION Network 18: Multiplexado Señales de Salida de la Mesa--> FTF
   RUNG wire#powerrail
      Contact( #Selec_M1_Salida )
      Contact( #FTF_Sal_M1 )
      wire#w1
      Coil( #FTF_MSal )
   END_RUNG
   RUNG wire#powerrail
      Contact( #Selec_M2_Salida )
      Contact( #FTF_Sal_M2 )
   END_RUNG wire#w1
   RUNG wire#powerrail
      Contact( #Selec_M3_Salida )
      Contact( #FTF_Sal_M3 )
   END_RUNG wire#w1
   RUNG wire#powerrail
      Contact( #Selec_M4_Salida )
      Contact( #FTF_Sal_M4 )
   END_RUNG wire#w1
   // the same network as SCL:
   #FTF_MSal := (#Selec_M1_Salida AND #FTF_Sal_M1) OR (#Selec_M2_Salida AND #FTF_Sal_M2) OR (#Selec_M3_Salida AND #FTF_Sal_M3) OR (#Selec_M4_Salida AND #FTF_Sal_M4);
END_REGION

REGION Network 19: VARIABLES AUXILIARES - Saliendo Carga de la Mesa
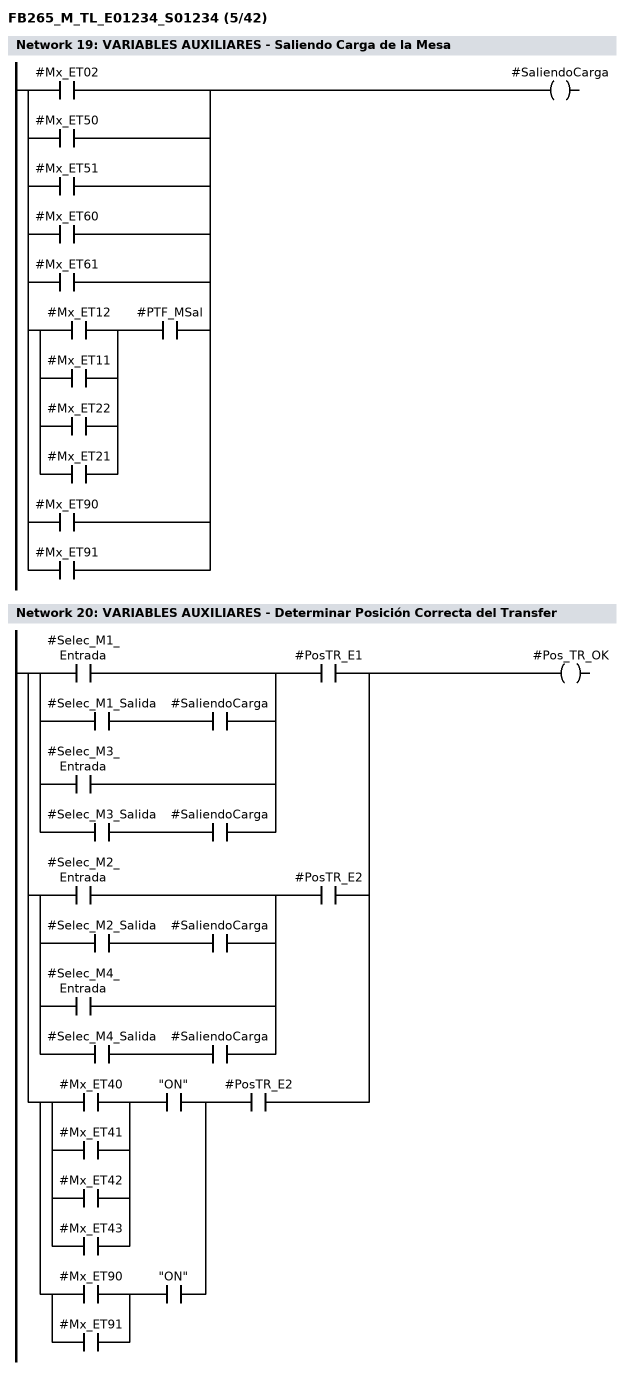
   RUNG wire#powerrail
      Contact( #Mx_ET02 )
      wire#w1
      Coil( #SaliendoCarga )
   END_RUNG
   RUNG wire#powerrail
      Contact( #Mx_ET50 )
   END_RUNG wire#w1
   RUNG wire#powerrail
      Contact( #Mx_ET51 )
   END_RUNG wire#w1
   RUNG wire#powerrail
      Contact( #Mx_ET60 )
   END_RUNG wire#w1
   RUNG wire#powerrail
      Contact( #Mx_ET61 )
   END_RUNG wire#w1
   RUNG wire#powerrail
      Contact( #Mx_ET12 )
      wire#w2
      Contact( #PTF_MSal )
   END_RUNG wire#w1
   RUNG wire#powerrail
      Contact( #Mx_ET11 )
   END_RUNG wire#w2
   RUNG wire#powerrail
      Contact( #Mx_ET22 )
   END_RUNG wire#w2
   RUNG wire#powerrail
      Contact( #Mx_ET21 )
   END_RUNG wire#w2
   RUNG wire#powerrail
      Contact( #Mx_ET90 )
   END_RUNG wire#w1
   RUNG wire#powerrail
      Contact( #Mx_ET91 )
   END_RUNG wire#w1
   // the same network as SCL:
   #SaliendoCarga := #Mx_ET02 OR #Mx_ET50 OR #Mx_ET51 OR #Mx_ET60 OR #Mx_ET61 OR ((#Mx_ET12 OR #Mx_ET11 OR #Mx_ET22 OR #Mx_ET21) AND #PTF_MSal) OR #Mx_ET90 OR #Mx_ET91;
END_REGION

REGION Network 20: VARIABLES AUXILIARES - Determinar Posición Correcta del Transfer
   RUNG wire#powerrail
      Contact( #Selec_M1_Entrada )
      wire#w1
      Contact( #PosTR_E1 )
      wire#w2
      Coil( #Pos_TR_OK )
   END_RUNG
   RUNG wire#powerrail
      Contact( #Selec_M1_Salida )
      Contact( #SaliendoCarga )
   END_RUNG wire#w1
   RUNG wire#powerrail
      Contact( #Selec_M3_Entrada )
   END_RUNG wire#w1
   RUNG wire#powerrail
      Contact( #Selec_M3_Salida )
      Contact( #SaliendoCarga )
   END_RUNG wire#w1
   RUNG wire#powerrail
      Contact( #Selec_M2_Entrada )
      wire#w3
      Contact( #PosTR_E2 )
   END_RUNG wire#w2
   RUNG wire#powerrail
      Contact( #Selec_M2_Salida )
      Contact( #SaliendoCarga )
   END_RUNG wire#w3
   RUNG wire#powerrail
      Contact( #Selec_M4_Entrada )
   END_RUNG wire#w3
   RUNG wire#powerrail
      Contact( #Selec_M4_Salida )
      Contact( #SaliendoCarga )
   END_RUNG wire#w3
   RUNG wire#powerrail
      Contact( #Mx_ET40 )
      wire#w4
      Contact( "ON" )
      wire#w5
      Contact( #PosTR_E2 )
   END_RUNG wire#w2
   RUNG wire#powerrail
      Contact( #Mx_ET41 )
   END_RUNG wire#w4
   RUNG wire#powerrail
      Contact( #Mx_ET42 )
   END_RUNG wire#w4
   RUNG wire#powerrail
      Contact( #Mx_ET43 )
   END_RUNG wire#w4
   RUNG wire#powerrail
      Contact( #Mx_ET90 )
      wire#w6
      Contact( "ON" )
   END_RUNG wire#w5
   RUNG wire#powerrail
      Contact( #Mx_ET91 )
   END_RUNG wire#w6
   // the same network as SCL:
   #Pos_TR_OK := ((#Selec_M1_Entrada OR (#Selec_M1_Salida AND #SaliendoCarga) OR #Selec_M3_Entrada OR (#Selec_M3_Salida AND #SaliendoCarga)) AND #PosTR_E1) OR ((#Selec_M2_Entrada OR (#Selec_M2_Salida AND #SaliendoCarga) OR #Selec_M4_Entrada OR (#Selec_M4_Salida AND #SaliendoCarga)) AND #PosTR_E2) OR ((((#Mx_ET40 OR #Mx_ET41 OR #Mx_ET42 OR #Mx_ET43) AND "ON") OR ((#Mx_ET90 OR #Mx_ET91) AND "ON")) AND #PosTR_E2);
END_REGION

REGION Network 21: VARIABLES AUXILIARES - FTF de Entrada
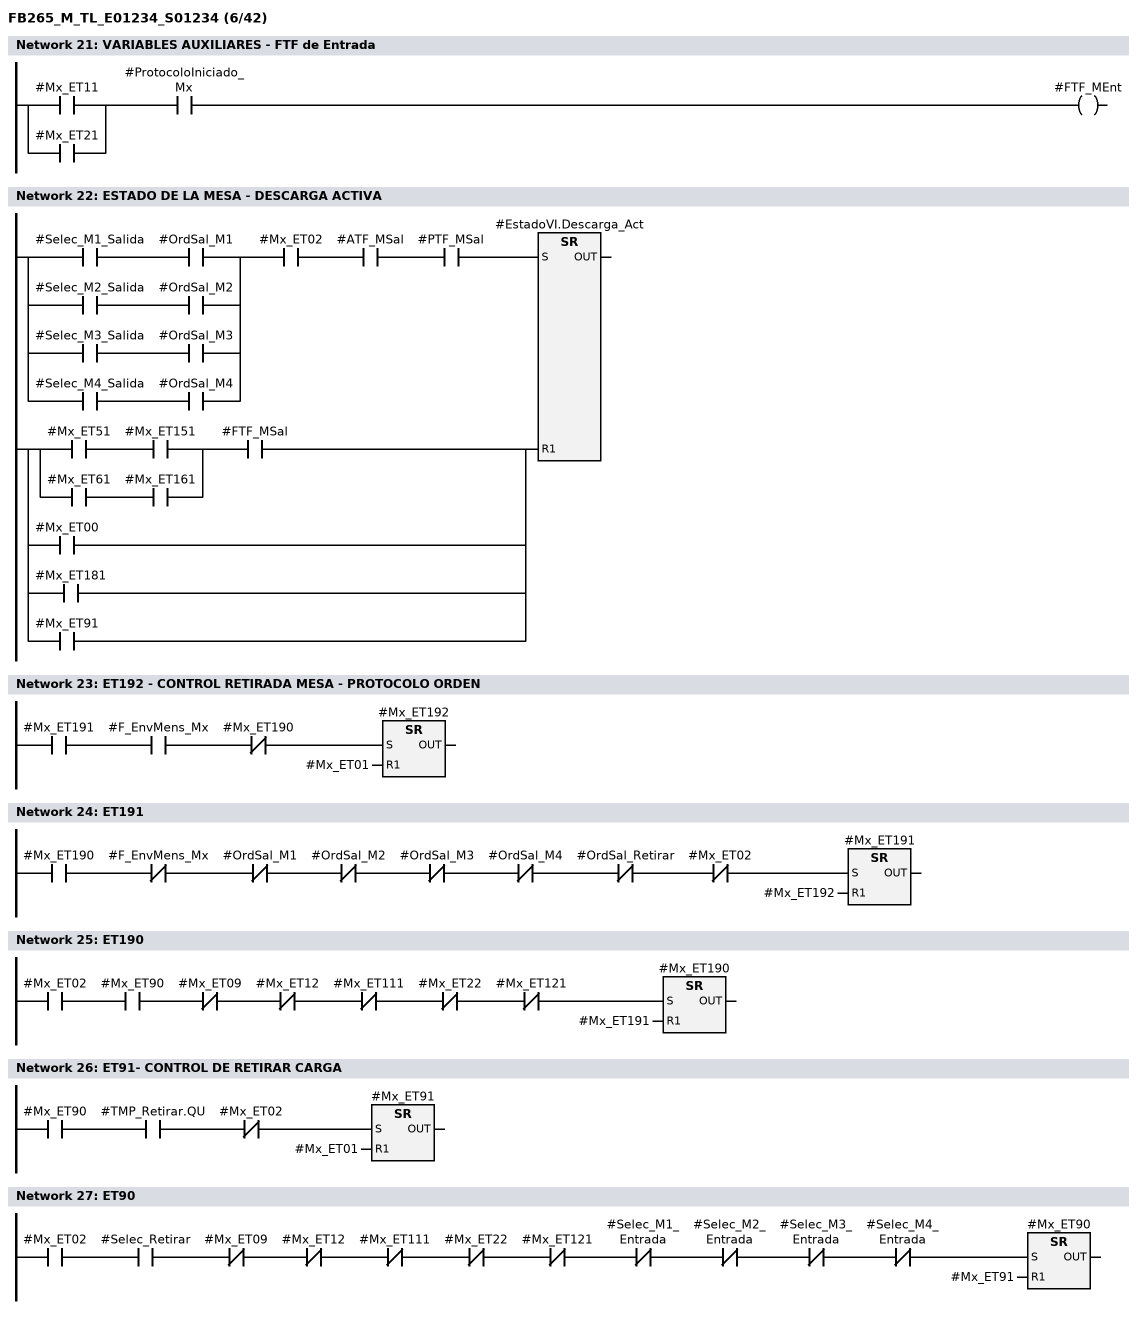
   RUNG wire#powerrail
      Contact( #Mx_ET11 )
      wire#w1
      Contact( #ProtocoloIniciado_Mx )
      Coil( #FTF_MEnt )
   END_RUNG
   RUNG wire#powerrail
      Contact( #Mx_ET21 )
   END_RUNG wire#w1
   // the same network as SCL:
   #FTF_MEnt := (#Mx_ET11 OR #Mx_ET21) AND #ProtocoloIniciado_Mx;
END_REGION

REGION Network 22: ESTADO DE LA MESA - DESCARGA ACTIVA
   RUNG wire#powerrail
      Contact( #Selec_M1_Salida )
      Contact( #OrdSal_M1 )
      wire#w1
      Contact( #Mx_ET02 )
      Contact( #ATF_MSal )
      Contact( #PTF_MSal )
      S_SR(operand := #EstadoVI.Descarga_Act, r1 := wire#w3)
   END_RUNG
   RUNG wire#powerrail
      Contact( #Selec_M2_Salida )
      Contact( #OrdSal_M2 )
   END_RUNG wire#w1
   RUNG wire#powerrail
      Contact( #Selec_M3_Salida )
      Contact( #OrdSal_M3 )
   END_RUNG wire#w1
   RUNG wire#powerrail
      Contact( #Selec_M4_Salida )
      Contact( #OrdSal_M4 )
   END_RUNG wire#w1
   RUNG wire#powerrail
      Contact( #Mx_ET51 )
      Contact( #Mx_ET151 )
      wire#w2
      Contact( #FTF_MSal )
   END_RUNG wire#w3
   RUNG wire#powerrail
      Contact( #Mx_ET61 )
      Contact( #Mx_ET161 )
   END_RUNG wire#w2
   RUNG wire#powerrail
      Contact( #Mx_ET00 )
   END_RUNG wire#w3
   RUNG wire#powerrail
      Contact( #Mx_ET181 )
   END_RUNG wire#w3
   RUNG wire#powerrail
      Contact( #Mx_ET91 )
   END_RUNG wire#w3
   // the same network as SCL:
   IF ((#Selec_M1_Salida AND #OrdSal_M1) OR (#Selec_M2_Salida AND #OrdSal_M2) OR (#Selec_M3_Salida AND #OrdSal_M3) OR (#Selec_M4_Salida AND #OrdSal_M4)) AND #Mx_ET02 AND #ATF_MSal AND #PTF_MSal THEN
       #EstadoVI.Descarga_Act := TRUE;   // SR flip-flop
   END_IF;
   IF (((#Mx_ET51 AND #Mx_ET151) OR (#Mx_ET61 AND #Mx_ET161)) AND #FTF_MSal) OR #Mx_ET00 OR #Mx_ET181 OR #Mx_ET91 THEN
       #EstadoVI.Descarga_Act := FALSE;
   END_IF;
END_REGION

REGION Network 23: ET192 - CONTROL RETIRADA MESA - PROTOCOLO ORDEN
   RUNG wire#powerrail
      Contact( #Mx_ET191 )
      Contact( #F_EnvMens_Mx )
      I_Contact( #Mx_ET190 )
      S_SR(operand := #Mx_ET192, r1 := #Mx_ET01)
   END_RUNG
   // the same network as SCL:
   IF #Mx_ET191 AND #F_EnvMens_Mx AND NOT #Mx_ET190 THEN
       #Mx_ET192 := TRUE;   // SR flip-flop
   END_IF;
   IF #Mx_ET01 THEN #Mx_ET192 := FALSE; END_IF;
END_REGION

REGION Network 24: ET191
   RUNG wire#powerrail
      Contact( #Mx_ET190 )
      I_Contact( #F_EnvMens_Mx )
      I_Contact( #OrdSal_M1 )
      I_Contact( #OrdSal_M2 )
      I_Contact( #OrdSal_M3 )
      I_Contact( #OrdSal_M4 )
      I_Contact( #OrdSal_Retirar )
      I_Contact( #Mx_ET02 )
      S_SR(operand := #Mx_ET191, r1 := #Mx_ET192)
   END_RUNG
   // the same network as SCL:
   IF #Mx_ET190 AND NOT #F_EnvMens_Mx AND NOT #OrdSal_M1 AND NOT #OrdSal_M2 AND NOT #OrdSal_M3 AND NOT #OrdSal_M4 AND NOT #OrdSal_Retirar AND NOT #Mx_ET02 THEN
       #Mx_ET191 := TRUE;   // SR flip-flop
   END_IF;
   IF #Mx_ET192 THEN #Mx_ET191 := FALSE; END_IF;
END_REGION

REGION Network 25: ET190
   RUNG wire#powerrail
      Contact( #Mx_ET02 )
      Contact( #Mx_ET90 )
      I_Contact( #Mx_ET09 )
      I_Contact( #Mx_ET12 )
      I_Contact( #Mx_ET111 )
      I_Contact( #Mx_ET22 )
      I_Contact( #Mx_ET121 )
      S_SR(operand := #Mx_ET190, r1 := #Mx_ET191)
   END_RUNG
   // the same network as SCL:
   IF #Mx_ET02 AND #Mx_ET90 AND NOT #Mx_ET09 AND NOT #Mx_ET12 AND NOT #Mx_ET111 AND NOT #Mx_ET22 AND NOT #Mx_ET121 THEN
       #Mx_ET190 := TRUE;   // SR flip-flop
   END_IF;
   IF #Mx_ET191 THEN #Mx_ET190 := FALSE; END_IF;
END_REGION

REGION Network 26: ET91- CONTROL DE RETIRAR CARGA
   RUNG wire#powerrail
      Contact( #Mx_ET90 )
      Contact( #TMP_Retirar.QU )
      I_Contact( #Mx_ET02 )
      S_SR(operand := #Mx_ET91, r1 := #Mx_ET01)
   END_RUNG
   // the same network as SCL:
   IF #Mx_ET90 AND #TMP_Retirar.QU AND NOT #Mx_ET02 THEN
       #Mx_ET91 := TRUE;   // SR flip-flop
   END_IF;
   IF #Mx_ET01 THEN #Mx_ET91 := FALSE; END_IF;
END_REGION

REGION Network 27: ET90
   RUNG wire#powerrail
      Contact( #Mx_ET02 )
      Contact( #Selec_Retirar )
      I_Contact( #Mx_ET09 )
      I_Contact( #Mx_ET12 )
      I_Contact( #Mx_ET111 )
      I_Contact( #Mx_ET22 )
      I_Contact( #Mx_ET121 )
      I_Contact( #Selec_M1_Entrada )
      I_Contact( #Selec_M2_Entrada )
      I_Contact( #Selec_M3_Entrada )
      I_Contact( #Selec_M4_Entrada )
      S_SR(operand := #Mx_ET90, r1 := #Mx_ET91)
   END_RUNG
   // the same network as SCL:
   IF #Mx_ET02 AND #Selec_Retirar AND NOT #Mx_ET09 AND NOT #Mx_ET12 AND NOT #Mx_ET111 AND NOT #Mx_ET22 AND NOT #Mx_ET121 AND NOT #Selec_M1_Entrada AND NOT #Selec_M2_Entrada AND NOT #Selec_M3_Entrada AND NOT #Selec_M4_Entrada THEN
       #Mx_ET90 := TRUE;   // SR flip-flop
   END_IF;
   IF #Mx_ET91 THEN #Mx_ET90 := FALSE; END_IF;
END_REGION

REGION Network 28: ET181 - BLOQUEO DE MESA - PROTOCOLO PRESENCIA CON BLOQUEO
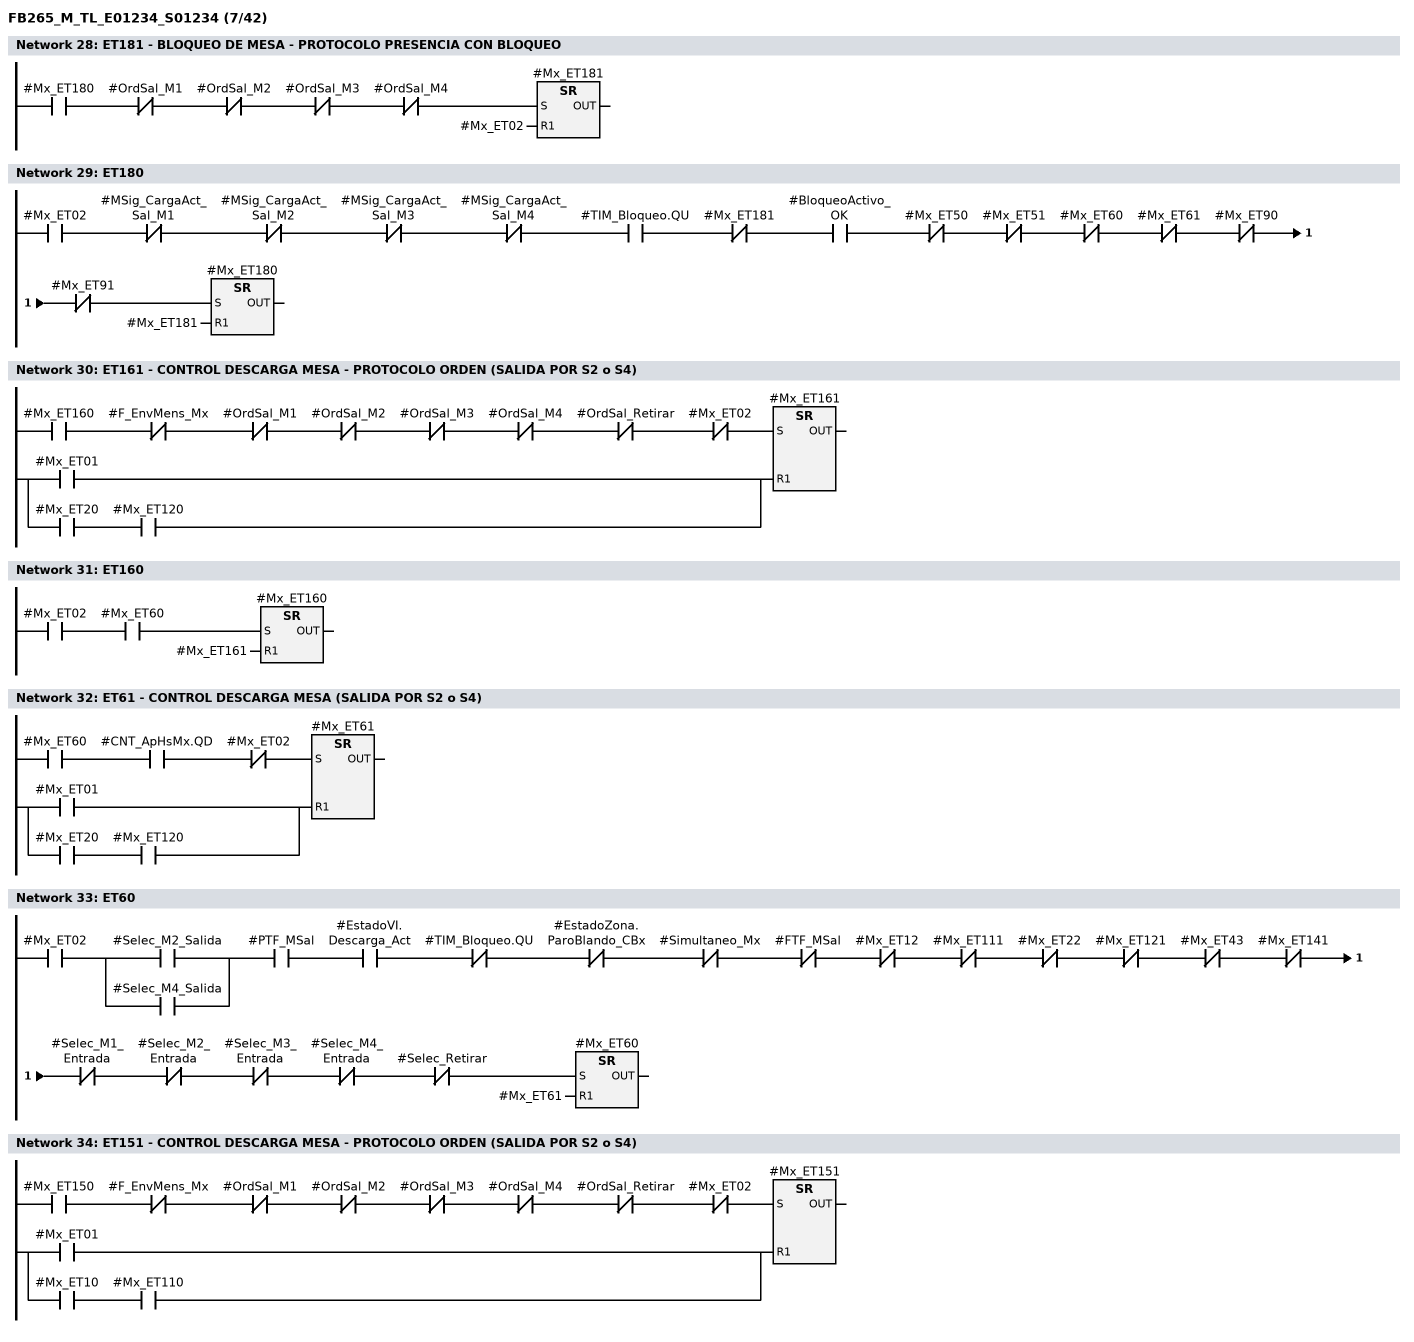
   RUNG wire#powerrail
      Contact( #Mx_ET180 )
      I_Contact( #OrdSal_M1 )
      I_Contact( #OrdSal_M2 )
      I_Contact( #OrdSal_M3 )
      I_Contact( #OrdSal_M4 )
      S_SR(operand := #Mx_ET181, r1 := #Mx_ET02)
   END_RUNG
   // the same network as SCL:
   IF #Mx_ET180 AND NOT #OrdSal_M1 AND NOT #OrdSal_M2 AND NOT #OrdSal_M3 AND NOT #OrdSal_M4 THEN
       #Mx_ET181 := TRUE;   // SR flip-flop
   END_IF;
   IF #Mx_ET02 THEN #Mx_ET181 := FALSE; END_IF;
END_REGION

REGION Network 29: ET180
   RUNG wire#powerrail
      Contact( #Mx_ET02 )
      I_Contact( #MSig_CargaAct_Sal_M1 )
      I_Contact( #MSig_CargaAct_Sal_M2 )
      I_Contact( #MSig_CargaAct_Sal_M3 )
      I_Contact( #MSig_CargaAct_Sal_M4 )
      Contact( #TIM_Bloqueo.QU )
      I_Contact( #Mx_ET181 )
      Contact( #BloqueoActivo_OK )
      I_Contact( #Mx_ET50 )
      I_Contact( #Mx_ET51 )
      I_Contact( #Mx_ET60 )
      I_Contact( #Mx_ET61 )
      I_Contact( #Mx_ET90 )
      I_Contact( #Mx_ET91 )
      S_SR(operand := #Mx_ET180, r1 := #Mx_ET181)
   END_RUNG
   // the same network as SCL:
   IF #Mx_ET02 AND NOT #MSig_CargaAct_Sal_M1 AND NOT #MSig_CargaAct_Sal_M2 AND NOT #MSig_CargaAct_Sal_M3 AND NOT #MSig_CargaAct_Sal_M4 AND #TIM_Bloqueo.QU AND NOT #Mx_ET181 AND #BloqueoActivo_OK AND NOT #Mx_ET50 AND NOT #Mx_ET51 AND NOT #Mx_ET60 AND NOT #Mx_ET61 AND NOT #Mx_ET90 AND NOT #Mx_ET91 THEN
       #Mx_ET180 := TRUE;   // SR flip-flop
   END_IF;
   IF #Mx_ET181 THEN #Mx_ET180 := FALSE; END_IF;
END_REGION

REGION Network 30: ET161 - CONTROL DESCARGA MESA - PROTOCOLO ORDEN (SALIDA POR S2 o S4)
   RUNG wire#powerrail
      Contact( #Mx_ET160 )
      I_Contact( #F_EnvMens_Mx )
      I_Contact( #OrdSal_M1 )
      I_Contact( #OrdSal_M2 )
      I_Contact( #OrdSal_M3 )
      I_Contact( #OrdSal_M4 )
      I_Contact( #OrdSal_Retirar )
      I_Contact( #Mx_ET02 )
      S_SR(operand := #Mx_ET161, r1 := wire#w1)
   END_RUNG
   RUNG wire#powerrail
      Contact( #Mx_ET01 )
   END_RUNG wire#w1
   RUNG wire#powerrail
      Contact( #Mx_ET20 )
      Contact( #Mx_ET120 )
   END_RUNG wire#w1
   // the same network as SCL:
   IF #Mx_ET160 AND NOT #F_EnvMens_Mx AND NOT #OrdSal_M1 AND NOT #OrdSal_M2 AND NOT #OrdSal_M3 AND NOT #OrdSal_M4 AND NOT #OrdSal_Retirar AND NOT #Mx_ET02 THEN
       #Mx_ET161 := TRUE;   // SR flip-flop
   END_IF;
   IF #Mx_ET01 OR (#Mx_ET20 AND #Mx_ET120) THEN #Mx_ET161 := FALSE; END_IF;
END_REGION

REGION Network 31: ET160
   RUNG wire#powerrail
      Contact( #Mx_ET02 )
      Contact( #Mx_ET60 )
      S_SR(operand := #Mx_ET160, r1 := #Mx_ET161)
   END_RUNG
   // the same network as SCL:
   IF #Mx_ET02 AND #Mx_ET60 THEN
       #Mx_ET160 := TRUE;   // SR flip-flop
   END_IF;
   IF #Mx_ET161 THEN #Mx_ET160 := FALSE; END_IF;
END_REGION

REGION Network 32: ET61 - CONTROL DESCARGA MESA (SALIDA POR S2 o S4)
   RUNG wire#powerrail
      Contact( #Mx_ET60 )
      Contact( #CNT_ApHsMx.QD )
      I_Contact( #Mx_ET02 )
      S_SR(operand := #Mx_ET61, r1 := wire#w1)
   END_RUNG
   RUNG wire#powerrail
      Contact( #Mx_ET01 )
   END_RUNG wire#w1
   RUNG wire#powerrail
      Contact( #Mx_ET20 )
      Contact( #Mx_ET120 )
   END_RUNG wire#w1
   // the same network as SCL:
   IF #Mx_ET60 AND #CNT_ApHsMx.QD AND NOT #Mx_ET02 THEN
       #Mx_ET61 := TRUE;   // SR flip-flop
   END_IF;
   IF #Mx_ET01 OR (#Mx_ET20 AND #Mx_ET120) THEN #Mx_ET61 := FALSE; END_IF;
END_REGION

REGION Network 33: ET60
   RUNG wire#powerrail
      Contact( #Mx_ET02 )
      wire#w1
      Contact( #Selec_M2_Salida )
      wire#w2
      Contact( #PTF_MSal )
      Contact( #EstadoVI.Descarga_Act )
      I_Contact( #TIM_Bloqueo.QU )
      I_Contact( #EstadoZona.ParoBlando_CBx )
      I_Contact( #Simultaneo_Mx )
      I_Contact( #FTF_MSal )
      I_Contact( #Mx_ET12 )
      I_Contact( #Mx_ET111 )
      I_Contact( #Mx_ET22 )
      I_Contact( #Mx_ET121 )
      I_Contact( #Mx_ET43 )
      I_Contact( #Mx_ET141 )
      I_Contact( #Selec_M1_Entrada )
      I_Contact( #Selec_M2_Entrada )
      I_Contact( #Selec_M3_Entrada )
      I_Contact( #Selec_M4_Entrada )
      I_Contact( #Selec_Retirar )
      S_SR(operand := #Mx_ET60, r1 := #Mx_ET61)
   END_RUNG
   RUNG wire#w1
      Contact( #Selec_M4_Salida )
   END_RUNG wire#w2
   // the same network as SCL:
   IF #Mx_ET02 AND (#Selec_M2_Salida OR #Selec_M4_Salida) AND #PTF_MSal AND #EstadoVI.Descarga_Act AND NOT #TIM_Bloqueo.QU AND NOT #EstadoZona.ParoBlando_CBx AND NOT #Simultaneo_Mx AND NOT #FTF_MSal AND NOT #Mx_ET12 AND NOT #Mx_ET111 AND NOT #Mx_ET22 AND NOT #Mx_ET121 AND NOT #Mx_ET43 AND NOT #Mx_ET141 AND NOT #Selec_M1_Entrada AND NOT #Selec_M2_Entrada AND NOT #Selec_M3_Entrada AND NOT #Selec_M4_Entrada AND NOT #Selec_Retirar THEN
       #Mx_ET60 := TRUE;   // SR flip-flop
   END_IF;
   IF #Mx_ET61 THEN #Mx_ET60 := FALSE; END_IF;
END_REGION

REGION Network 34: ET151 - CONTROL DESCARGA MESA - PROTOCOLO ORDEN (SALIDA POR S2 o S4)
   RUNG wire#powerrail
      Contact( #Mx_ET150 )
      I_Contact( #F_EnvMens_Mx )
      I_Contact( #OrdSal_M1 )
      I_Contact( #OrdSal_M2 )
      I_Contact( #OrdSal_M3 )
      I_Contact( #OrdSal_M4 )
      I_Contact( #OrdSal_Retirar )
      I_Contact( #Mx_ET02 )
      S_SR(operand := #Mx_ET151, r1 := wire#w1)
   END_RUNG
   RUNG wire#powerrail
      Contact( #Mx_ET01 )
   END_RUNG wire#w1
   RUNG wire#powerrail
      Contact( #Mx_ET10 )
      Contact( #Mx_ET110 )
   END_RUNG wire#w1
   // the same network as SCL:
   IF #Mx_ET150 AND NOT #F_EnvMens_Mx AND NOT #OrdSal_M1 AND NOT #OrdSal_M2 AND NOT #OrdSal_M3 AND NOT #OrdSal_M4 AND NOT #OrdSal_Retirar AND NOT #Mx_ET02 THEN
       #Mx_ET151 := TRUE;   // SR flip-flop
   END_IF;
   IF #Mx_ET01 OR (#Mx_ET10 AND #Mx_ET110) THEN #Mx_ET151 := FALSE; END_IF;
END_REGION

REGION Network 35: ET150
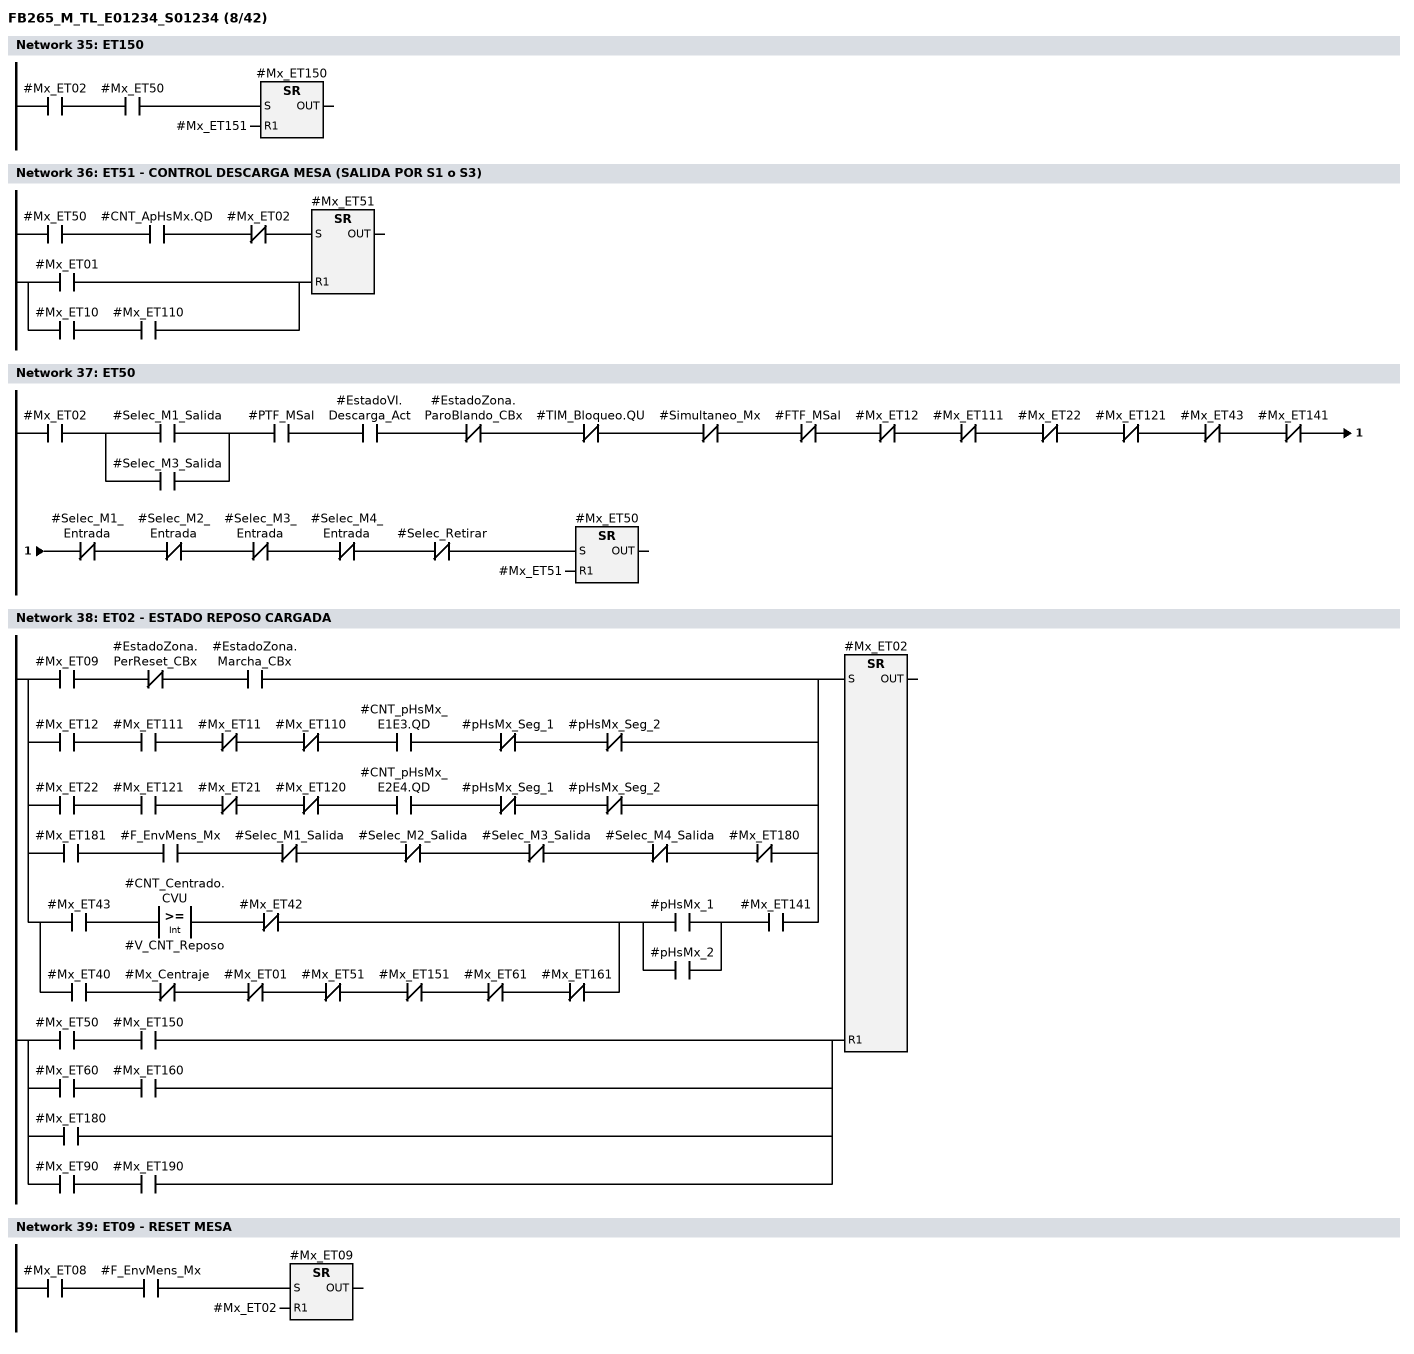
   RUNG wire#powerrail
      Contact( #Mx_ET02 )
      Contact( #Mx_ET50 )
      S_SR(operand := #Mx_ET150, r1 := #Mx_ET151)
   END_RUNG
   // the same network as SCL:
   IF #Mx_ET02 AND #Mx_ET50 THEN
       #Mx_ET150 := TRUE;   // SR flip-flop
   END_IF;
   IF #Mx_ET151 THEN #Mx_ET150 := FALSE; END_IF;
END_REGION

REGION Network 36: ET51 - CONTROL DESCARGA MESA (SALIDA POR S1 o S3)
   RUNG wire#powerrail
      Contact( #Mx_ET50 )
      Contact( #CNT_ApHsMx.QD )
      I_Contact( #Mx_ET02 )
      S_SR(operand := #Mx_ET51, r1 := wire#w1)
   END_RUNG
   RUNG wire#powerrail
      Contact( #Mx_ET01 )
   END_RUNG wire#w1
   RUNG wire#powerrail
      Contact( #Mx_ET10 )
      Contact( #Mx_ET110 )
   END_RUNG wire#w1
   // the same network as SCL:
   IF #Mx_ET50 AND #CNT_ApHsMx.QD AND NOT #Mx_ET02 THEN
       #Mx_ET51 := TRUE;   // SR flip-flop
   END_IF;
   IF #Mx_ET01 OR (#Mx_ET10 AND #Mx_ET110) THEN #Mx_ET51 := FALSE; END_IF;
END_REGION

REGION Network 37: ET50
   RUNG wire#powerrail
      Contact( #Mx_ET02 )
      wire#w1
      Contact( #Selec_M1_Salida )
      wire#w2
      Contact( #PTF_MSal )
      Contact( #EstadoVI.Descarga_Act )
      I_Contact( #EstadoZona.ParoBlando_CBx )
      I_Contact( #TIM_Bloqueo.QU )
      I_Contact( #Simultaneo_Mx )
      I_Contact( #FTF_MSal )
      I_Contact( #Mx_ET12 )
      I_Contact( #Mx_ET111 )
      I_Contact( #Mx_ET22 )
      I_Contact( #Mx_ET121 )
      I_Contact( #Mx_ET43 )
      I_Contact( #Mx_ET141 )
      I_Contact( #Selec_M1_Entrada )
      I_Contact( #Selec_M2_Entrada )
      I_Contact( #Selec_M3_Entrada )
      I_Contact( #Selec_M4_Entrada )
      I_Contact( #Selec_Retirar )
      S_SR(operand := #Mx_ET50, r1 := #Mx_ET51)
   END_RUNG
   RUNG wire#w1
      Contact( #Selec_M3_Salida )
   END_RUNG wire#w2
   // the same network as SCL:
   IF #Mx_ET02 AND (#Selec_M1_Salida OR #Selec_M3_Salida) AND #PTF_MSal AND #EstadoVI.Descarga_Act AND NOT #EstadoZona.ParoBlando_CBx AND NOT #TIM_Bloqueo.QU AND NOT #Simultaneo_Mx AND NOT #FTF_MSal AND NOT #Mx_ET12 AND NOT #Mx_ET111 AND NOT #Mx_ET22 AND NOT #Mx_ET121 AND NOT #Mx_ET43 AND NOT #Mx_ET141 AND NOT #Selec_M1_Entrada AND NOT #Selec_M2_Entrada AND NOT #Selec_M3_Entrada AND NOT #Selec_M4_Entrada AND NOT #Selec_Retirar THEN
       #Mx_ET50 := TRUE;   // SR flip-flop
   END_IF;
   IF #Mx_ET51 THEN #Mx_ET50 := FALSE; END_IF;
END_REGION

REGION Network 38: ET02 - ESTADO REPOSO CARGADA
   RUNG wire#powerrail
      Contact( #Mx_ET09 )
      I_Contact( #EstadoZona.PerReset_CBx )
      Contact( #EstadoZona.Marcha_CBx )
      wire#w1
      S_SR(operand := #Mx_ET02, r1 := wire#w4)
   END_RUNG
   RUNG wire#powerrail
      Contact( #Mx_ET12 )
      Contact( #Mx_ET111 )
      I_Contact( #Mx_ET11 )
      I_Contact( #Mx_ET110 )
      Contact( #CNT_pHsMx_E1E3.QD )
      I_Contact( #pHsMx_Seg_1 )
      I_Contact( #pHsMx_Seg_2 )
   END_RUNG wire#w1
   RUNG wire#powerrail
      Contact( #Mx_ET22 )
      Contact( #Mx_ET121 )
      I_Contact( #Mx_ET21 )
      I_Contact( #Mx_ET120 )
      Contact( #CNT_pHsMx_E2E4.QD )
      I_Contact( #pHsMx_Seg_1 )
      I_Contact( #pHsMx_Seg_2 )
   END_RUNG wire#w1
   RUNG wire#powerrail
      Contact( #Mx_ET181 )
      Contact( #F_EnvMens_Mx )
      I_Contact( #Selec_M1_Salida )
      I_Contact( #Selec_M2_Salida )
      I_Contact( #Selec_M3_Salida )
      I_Contact( #Selec_M4_Salida )
      I_Contact( #Mx_ET180 )
   END_RUNG wire#w1
   RUNG wire#powerrail
      Contact( #Mx_ET43 )
      { S7_Templates := "SrcType := Int" } GE_Contact(in1 := #CNT_Centrado.CVU, in2 := #V_CNT_Reposo)
      I_Contact( #Mx_ET42 )
      wire#w2
      Contact( #pHsMx_1 )
      wire#w3
      Contact( #Mx_ET141 )
   END_RUNG wire#w1
   RUNG wire#powerrail
      Contact( #Mx_ET40 )
      I_Contact( #Mx_Centraje )
      I_Contact( #Mx_ET01 )
      I_Contact( #Mx_ET51 )
      I_Contact( #Mx_ET151 )
      I_Contact( #Mx_ET61 )
      I_Contact( #Mx_ET161 )
   END_RUNG wire#w2
   RUNG wire#w2
      Contact( #pHsMx_2 )
   END_RUNG wire#w3
   RUNG wire#powerrail
      Contact( #Mx_ET50 )
      Contact( #Mx_ET150 )
   END_RUNG wire#w4
   RUNG wire#powerrail
      Contact( #Mx_ET60 )
      Contact( #Mx_ET160 )
   END_RUNG wire#w4
   RUNG wire#powerrail
      Contact( #Mx_ET180 )
   END_RUNG wire#w4
   RUNG wire#powerrail
      Contact( #Mx_ET90 )
      Contact( #Mx_ET190 )
   END_RUNG wire#w4
   // the same network as SCL:
   IF (#Mx_ET09 AND NOT #EstadoZona.PerReset_CBx AND #EstadoZona.Marcha_CBx) OR (#Mx_ET12 AND #Mx_ET111 AND NOT #Mx_ET11 AND NOT #Mx_ET110 AND #CNT_pHsMx_E1E3.QD AND NOT #pHsMx_Seg_1 AND NOT #pHsMx_Seg_2) OR (#Mx_ET22 AND #Mx_ET121 AND NOT #Mx_ET21 AND NOT #Mx_ET120 AND #CNT_pHsMx_E2E4.QD AND NOT #pHsMx_Seg_1 AND NOT #pHsMx_Seg_2) OR (#Mx_ET181 AND #F_EnvMens_Mx AND NOT #Selec_M1_Salida AND NOT #Selec_M2_Salida AND NOT #Selec_M3_Salida AND NOT #Selec_M4_Salida AND NOT #Mx_ET180) OR (((#Mx_ET43 AND (#CNT_Centrado.CVU >= #V_CNT_Reposo) AND NOT #Mx_ET42) OR (#Mx_ET40 AND NOT #Mx_Centraje AND NOT #Mx_ET01 AND NOT #Mx_ET51 AND NOT #Mx_ET151 AND NOT #Mx_ET61 AND NOT #Mx_ET161)) AND (#pHsMx_1 OR #pHsMx_2) AND #Mx_ET141) THEN
       #Mx_ET02 := TRUE;   // SR flip-flop
   END_IF;
   IF (#Mx_ET50 AND #Mx_ET150) OR (#Mx_ET60 AND #Mx_ET160) OR #Mx_ET180 OR (#Mx_ET90 AND #Mx_ET190) THEN
       #Mx_ET02 := FALSE;
   END_IF;
END_REGION

REGION Network 39: ET09 - RESET MESA
   RUNG wire#powerrail
      Contact( #Mx_ET08 )
      Contact( #F_EnvMens_Mx )
      S_SR(operand := #Mx_ET09, r1 := #Mx_ET02)
   END_RUNG
   // the same network as SCL:
   IF #Mx_ET08 AND #F_EnvMens_Mx THEN
       #Mx_ET09 := TRUE;   // SR flip-flop
   END_IF;
   IF #Mx_ET02 THEN #Mx_ET09 := FALSE; END_IF;
END_REGION

REGION Network 40: ET08
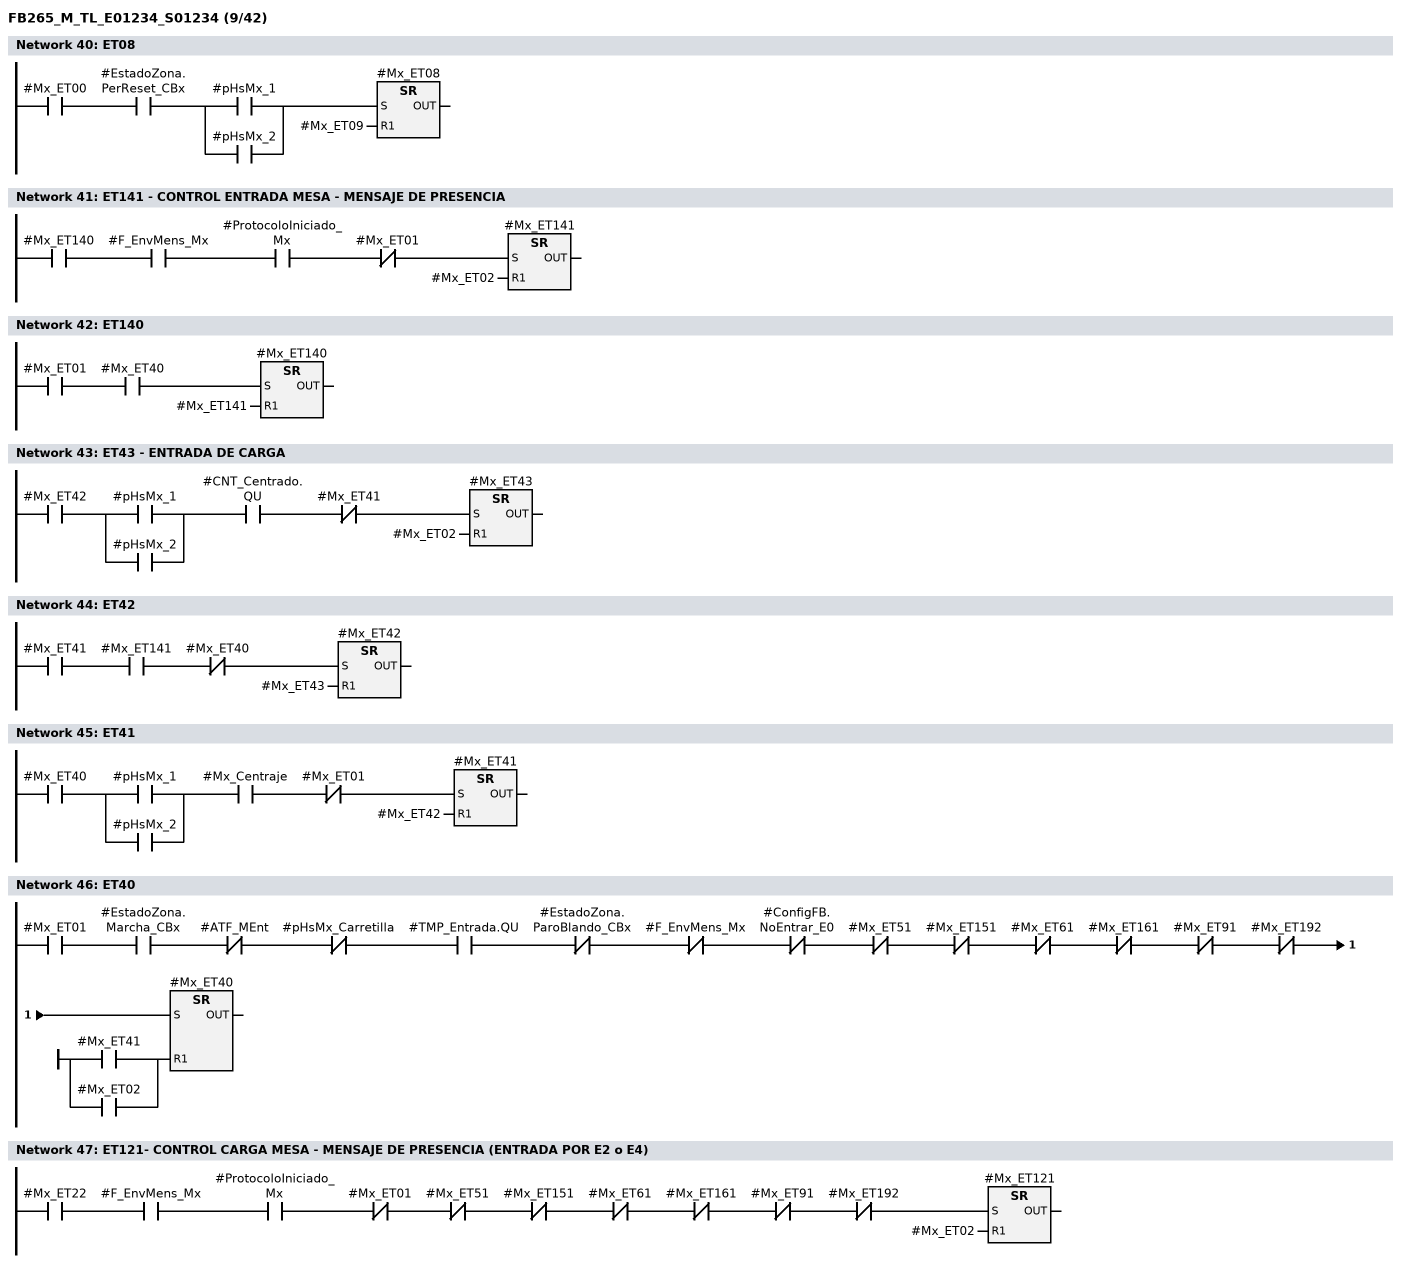
   RUNG wire#powerrail
      Contact( #Mx_ET00 )
      Contact( #EstadoZona.PerReset_CBx )
      wire#w1
      Contact( #pHsMx_1 )
      wire#w2
      S_SR(operand := #Mx_ET08, r1 := #Mx_ET09)
   END_RUNG
   RUNG wire#w1
      Contact( #pHsMx_2 )
   END_RUNG wire#w2
   // the same network as SCL:
   IF #Mx_ET00 AND #EstadoZona.PerReset_CBx AND (#pHsMx_1 OR #pHsMx_2) THEN
       #Mx_ET08 := TRUE;   // SR flip-flop
   END_IF;
   IF #Mx_ET09 THEN #Mx_ET08 := FALSE; END_IF;
END_REGION

REGION Network 41: ET141 - CONTROL ENTRADA MESA - MENSAJE DE PRESENCIA
   RUNG wire#powerrail
      Contact( #Mx_ET140 )
      Contact( #F_EnvMens_Mx )
      Contact( #ProtocoloIniciado_Mx )
      I_Contact( #Mx_ET01 )
      S_SR(operand := #Mx_ET141, r1 := #Mx_ET02)
   END_RUNG
   // the same network as SCL:
   IF #Mx_ET140 AND #F_EnvMens_Mx AND #ProtocoloIniciado_Mx AND NOT #Mx_ET01 THEN
       #Mx_ET141 := TRUE;   // SR flip-flop
   END_IF;
   IF #Mx_ET02 THEN #Mx_ET141 := FALSE; END_IF;
END_REGION

REGION Network 42: ET140
   RUNG wire#powerrail
      Contact( #Mx_ET01 )
      Contact( #Mx_ET40 )
      S_SR(operand := #Mx_ET140, r1 := #Mx_ET141)
   END_RUNG
   // the same network as SCL:
   IF #Mx_ET01 AND #Mx_ET40 THEN
       #Mx_ET140 := TRUE;   // SR flip-flop
   END_IF;
   IF #Mx_ET141 THEN #Mx_ET140 := FALSE; END_IF;
END_REGION

REGION Network 43: ET43 - ENTRADA DE CARGA
   RUNG wire#powerrail
      Contact( #Mx_ET42 )
      wire#w1
      Contact( #pHsMx_1 )
      wire#w2
      Contact( #CNT_Centrado.QU )
      I_Contact( #Mx_ET41 )
      S_SR(operand := #Mx_ET43, r1 := #Mx_ET02)
   END_RUNG
   RUNG wire#w1
      Contact( #pHsMx_2 )
   END_RUNG wire#w2
   // the same network as SCL:
   IF #Mx_ET42 AND (#pHsMx_1 OR #pHsMx_2) AND #CNT_Centrado.QU AND NOT #Mx_ET41 THEN
       #Mx_ET43 := TRUE;   // SR flip-flop
   END_IF;
   IF #Mx_ET02 THEN #Mx_ET43 := FALSE; END_IF;
END_REGION

REGION Network 44: ET42
   RUNG wire#powerrail
      Contact( #Mx_ET41 )
      Contact( #Mx_ET141 )
      I_Contact( #Mx_ET40 )
      S_SR(operand := #Mx_ET42, r1 := #Mx_ET43)
   END_RUNG
   // the same network as SCL:
   IF #Mx_ET41 AND #Mx_ET141 AND NOT #Mx_ET40 THEN
       #Mx_ET42 := TRUE;   // SR flip-flop
   END_IF;
   IF #Mx_ET43 THEN #Mx_ET42 := FALSE; END_IF;
END_REGION

REGION Network 45: ET41
   RUNG wire#powerrail
      Contact( #Mx_ET40 )
      wire#w1
      Contact( #pHsMx_1 )
      wire#w2
      Contact( #Mx_Centraje )
      I_Contact( #Mx_ET01 )
      S_SR(operand := #Mx_ET41, r1 := #Mx_ET42)
   END_RUNG
   RUNG wire#w1
      Contact( #pHsMx_2 )
   END_RUNG wire#w2
   // the same network as SCL:
   IF #Mx_ET40 AND (#pHsMx_1 OR #pHsMx_2) AND #Mx_Centraje AND NOT #Mx_ET01 THEN
       #Mx_ET41 := TRUE;   // SR flip-flop
   END_IF;
   IF #Mx_ET42 THEN #Mx_ET41 := FALSE; END_IF;
END_REGION

REGION Network 46: ET40
   RUNG wire#powerrail
      Contact( #Mx_ET01 )
      Contact( #EstadoZona.Marcha_CBx )
      I_Contact( #ATF_MEnt )
      I_Contact( #pHsMx_Carretilla )
      Contact( #TMP_Entrada.QU )
      I_Contact( #EstadoZona.ParoBlando_CBx )
      I_Contact( #F_EnvMens_Mx )
      I_Contact( #ConfigFB.NoEntrar_E0 )
      I_Contact( #Mx_ET51 )
      I_Contact( #Mx_ET151 )
      I_Contact( #Mx_ET61 )
      I_Contact( #Mx_ET161 )
      I_Contact( #Mx_ET91 )
      I_Contact( #Mx_ET192 )
      S_SR(operand := #Mx_ET40, r1 := wire#w1)
   END_RUNG
   RUNG wire#powerrail
      Contact( #Mx_ET41 )
   END_RUNG wire#w1
   RUNG wire#powerrail
      Contact( #Mx_ET02 )
   END_RUNG wire#w1
   // the same network as SCL:
   IF #Mx_ET01 AND #EstadoZona.Marcha_CBx AND NOT #ATF_MEnt AND NOT #pHsMx_Carretilla AND #TMP_Entrada.QU AND NOT #EstadoZona.ParoBlando_CBx AND NOT #F_EnvMens_Mx AND NOT #ConfigFB.NoEntrar_E0 AND NOT #Mx_ET51 AND NOT #Mx_ET151 AND NOT #Mx_ET61 AND NOT #Mx_ET161 AND NOT #Mx_ET91 AND NOT #Mx_ET192 THEN
       #Mx_ET40 := TRUE;   // SR flip-flop
   END_IF;
   IF #Mx_ET41 OR #Mx_ET02 THEN #Mx_ET40 := FALSE; END_IF;
END_REGION

REGION Network 47: ET121- CONTROL CARGA MESA - MENSAJE DE PRESENCIA (ENTRADA POR E2 o E4)
   RUNG wire#powerrail
      Contact( #Mx_ET22 )
      Contact( #F_EnvMens_Mx )
      Contact( #ProtocoloIniciado_Mx )
      I_Contact( #Mx_ET01 )
      I_Contact( #Mx_ET51 )
      I_Contact( #Mx_ET151 )
      I_Contact( #Mx_ET61 )
      I_Contact( #Mx_ET161 )
      I_Contact( #Mx_ET91 )
      I_Contact( #Mx_ET192 )
      S_SR(operand := #Mx_ET121, r1 := #Mx_ET02)
   END_RUNG
   // the same network as SCL:
   IF #Mx_ET22 AND #F_EnvMens_Mx AND #ProtocoloIniciado_Mx AND NOT #Mx_ET01 AND NOT #Mx_ET51 AND NOT #Mx_ET151 AND NOT #Mx_ET61 AND NOT #Mx_ET161 AND NOT #Mx_ET91 AND NOT #Mx_ET192 THEN
       #Mx_ET121 := TRUE;   // SR flip-flop
   END_IF;
   IF #Mx_ET02 THEN #Mx_ET121 := FALSE; END_IF;
END_REGION

REGION Network 48: ET120
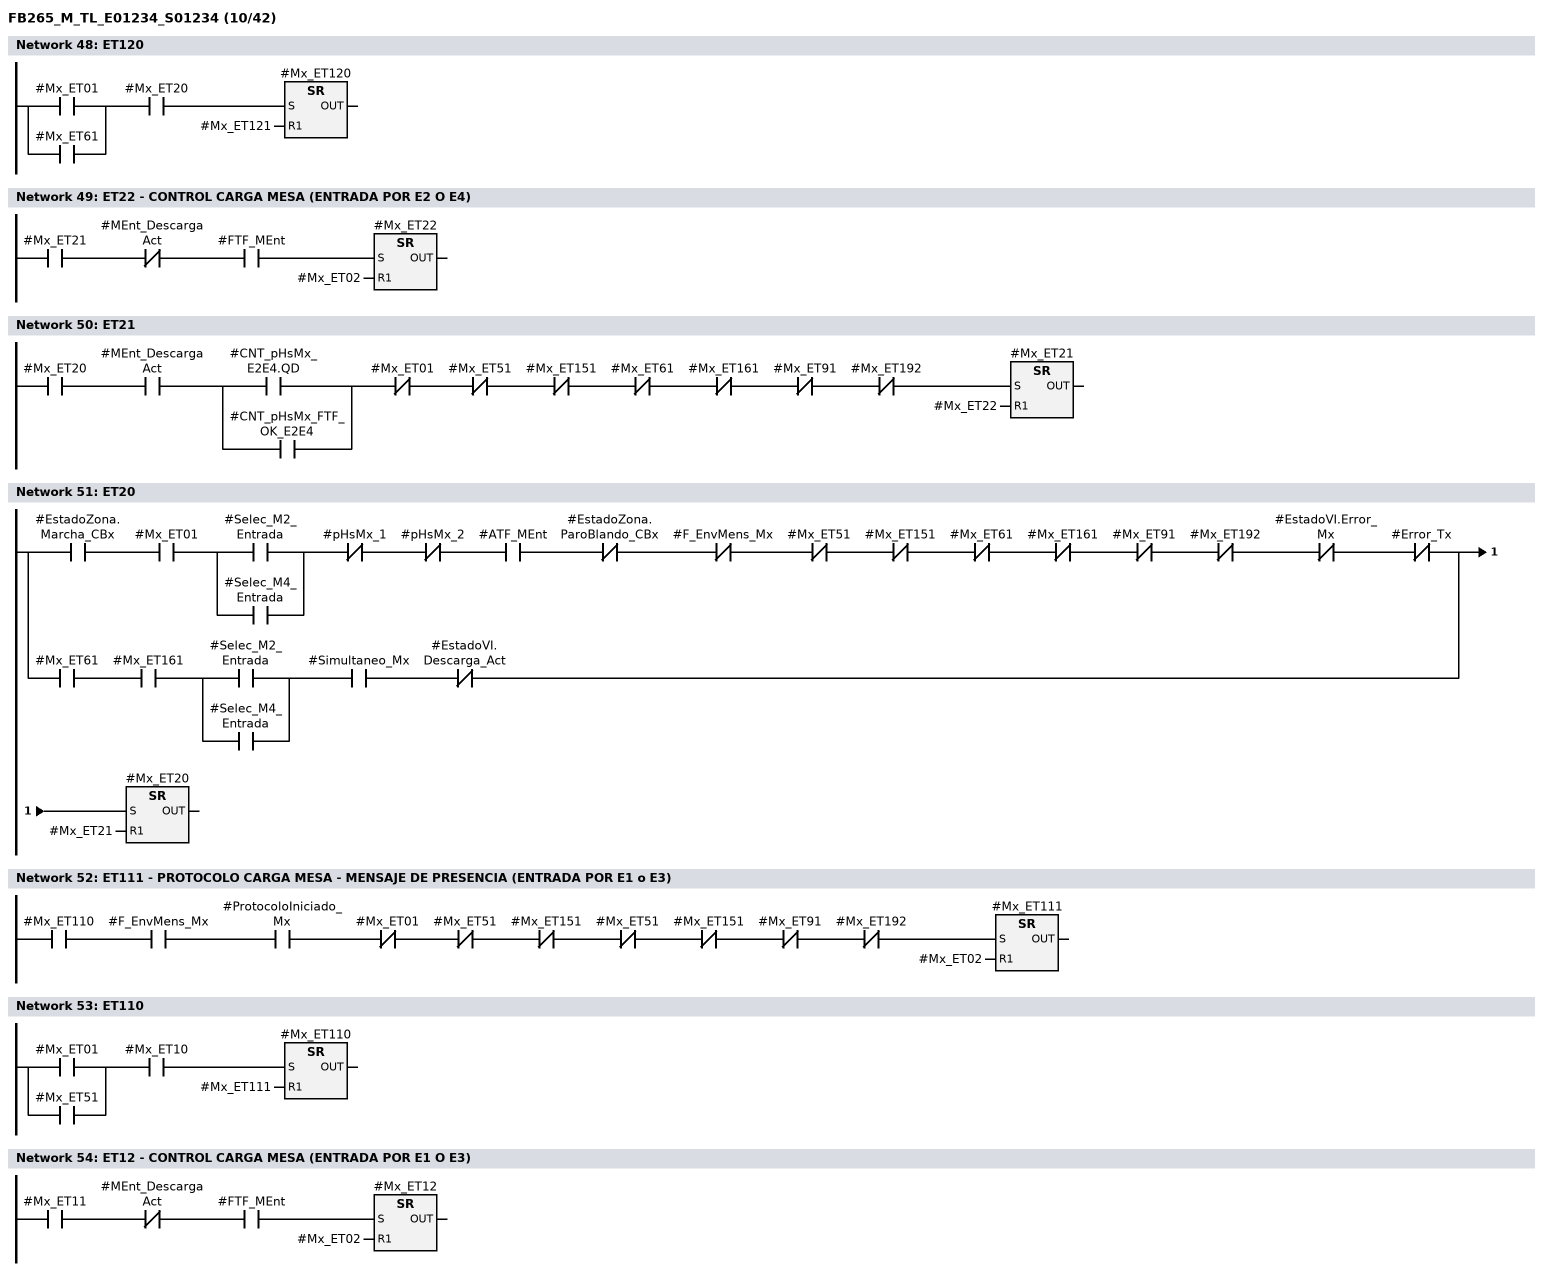
   RUNG wire#powerrail
      Contact( #Mx_ET01 )
      wire#w1
      Contact( #Mx_ET20 )
      S_SR(operand := #Mx_ET120, r1 := #Mx_ET121)
   END_RUNG
   RUNG wire#powerrail
      Contact( #Mx_ET61 )
   END_RUNG wire#w1
   // the same network as SCL:
   IF (#Mx_ET01 OR #Mx_ET61) AND #Mx_ET20 THEN
       #Mx_ET120 := TRUE;   // SR flip-flop
   END_IF;
   IF #Mx_ET121 THEN #Mx_ET120 := FALSE; END_IF;
END_REGION

REGION Network 49: ET22 - CONTROL CARGA MESA (ENTRADA POR E2 O E4)
   RUNG wire#powerrail
      Contact( #Mx_ET21 )
      I_Contact( #MEnt_DescargaAct )
      Contact( #FTF_MEnt )
      S_SR(operand := #Mx_ET22, r1 := #Mx_ET02)
   END_RUNG
   // the same network as SCL:
   IF #Mx_ET21 AND NOT #MEnt_DescargaAct AND #FTF_MEnt THEN
       #Mx_ET22 := TRUE;   // SR flip-flop
   END_IF;
   IF #Mx_ET02 THEN #Mx_ET22 := FALSE; END_IF;
END_REGION

REGION Network 50: ET21
   RUNG wire#powerrail
      Contact( #Mx_ET20 )
      Contact( #MEnt_DescargaAct )
      wire#w1
      Contact( #CNT_pHsMx_E2E4.QD )
      wire#w2
      I_Contact( #Mx_ET01 )
      I_Contact( #Mx_ET51 )
      I_Contact( #Mx_ET151 )
      I_Contact( #Mx_ET61 )
      I_Contact( #Mx_ET161 )
      I_Contact( #Mx_ET91 )
      I_Contact( #Mx_ET192 )
      S_SR(operand := #Mx_ET21, r1 := #Mx_ET22)
   END_RUNG
   RUNG wire#w1
      Contact( #CNT_pHsMx_FTF_OK_E2E4 )
   END_RUNG wire#w2
   // the same network as SCL:
   IF #Mx_ET20 AND #MEnt_DescargaAct AND (#CNT_pHsMx_E2E4.QD OR #CNT_pHsMx_FTF_OK_E2E4) AND NOT #Mx_ET01 AND NOT #Mx_ET51 AND NOT #Mx_ET151 AND NOT #Mx_ET61 AND NOT #Mx_ET161 AND NOT #Mx_ET91 AND NOT #Mx_ET192 THEN
       #Mx_ET21 := TRUE;   // SR flip-flop
   END_IF;
   IF #Mx_ET22 THEN #Mx_ET21 := FALSE; END_IF;
END_REGION

REGION Network 51: ET20
   RUNG wire#powerrail
      Contact( #EstadoZona.Marcha_CBx )
      Contact( #Mx_ET01 )
      wire#w1
      Contact( #Selec_M2_Entrada )
      wire#w2
      I_Contact( #pHsMx_1 )
      I_Contact( #pHsMx_2 )
      Contact( #ATF_MEnt )
      I_Contact( #EstadoZona.ParoBlando_CBx )
      I_Contact( #F_EnvMens_Mx )
      I_Contact( #Mx_ET51 )
      I_Contact( #Mx_ET151 )
      I_Contact( #Mx_ET61 )
      I_Contact( #Mx_ET161 )
      I_Contact( #Mx_ET91 )
      I_Contact( #Mx_ET192 )
      I_Contact( #EstadoVI.Error_Mx )
      I_Contact( #Error_Tx )
      wire#w3
      S_SR(operand := #Mx_ET20, r1 := #Mx_ET21)
   END_RUNG
   RUNG wire#w1
      Contact( #Selec_M4_Entrada )
   END_RUNG wire#w2
   RUNG wire#powerrail
      Contact( #Mx_ET61 )
      Contact( #Mx_ET161 )
      wire#w4
      Contact( #Selec_M2_Entrada )
      wire#w5
      Contact( #Simultaneo_Mx )
      I_Contact( #EstadoVI.Descarga_Act )
   END_RUNG wire#w3
   RUNG wire#w4
      Contact( #Selec_M4_Entrada )
   END_RUNG wire#w5
   // the same network as SCL:
   IF (#EstadoZona.Marcha_CBx AND #Mx_ET01 AND (#Selec_M2_Entrada OR #Selec_M4_Entrada) AND NOT #pHsMx_1 AND NOT #pHsMx_2 AND #ATF_MEnt AND NOT #EstadoZona.ParoBlando_CBx AND NOT #F_EnvMens_Mx AND NOT #Mx_ET51 AND NOT #Mx_ET151 AND NOT #Mx_ET61 AND NOT #Mx_ET161 AND NOT #Mx_ET91 AND NOT #Mx_ET192 AND NOT #EstadoVI.Error_Mx AND NOT #Error_Tx) OR (#Mx_ET61 AND #Mx_ET161 AND (#Selec_M2_Entrada OR #Selec_M4_Entrada) AND #Simultaneo_Mx AND NOT #EstadoVI.Descarga_Act) THEN
       #Mx_ET20 := TRUE;   // SR flip-flop
   END_IF;
   IF #Mx_ET21 THEN #Mx_ET20 := FALSE; END_IF;
END_REGION

REGION Network 52: ET111 - PROTOCOLO CARGA MESA - MENSAJE DE PRESENCIA (ENTRADA POR E1 o E3)
   RUNG wire#powerrail
      Contact( #Mx_ET110 )
      Contact( #F_EnvMens_Mx )
      Contact( #ProtocoloIniciado_Mx )
      I_Contact( #Mx_ET01 )
      I_Contact( #Mx_ET51 )
      I_Contact( #Mx_ET151 )
      I_Contact( #Mx_ET51 )
      I_Contact( #Mx_ET151 )
      I_Contact( #Mx_ET91 )
      I_Contact( #Mx_ET192 )
      S_SR(operand := #Mx_ET111, r1 := #Mx_ET02)
   END_RUNG
   // the same network as SCL:
   IF #Mx_ET110 AND #F_EnvMens_Mx AND #ProtocoloIniciado_Mx AND NOT #Mx_ET01 AND NOT #Mx_ET51 AND NOT #Mx_ET151 AND NOT #Mx_ET51 AND NOT #Mx_ET151 AND NOT #Mx_ET91 AND NOT #Mx_ET192 THEN
       #Mx_ET111 := TRUE;   // SR flip-flop
   END_IF;
   IF #Mx_ET02 THEN #Mx_ET111 := FALSE; END_IF;
END_REGION

REGION Network 53: ET110
   RUNG wire#powerrail
      Contact( #Mx_ET01 )
      wire#w1
      Contact( #Mx_ET10 )
      S_SR(operand := #Mx_ET110, r1 := #Mx_ET111)
   END_RUNG
   RUNG wire#powerrail
      Contact( #Mx_ET51 )
   END_RUNG wire#w1
   // the same network as SCL:
   IF (#Mx_ET01 OR #Mx_ET51) AND #Mx_ET10 THEN
       #Mx_ET110 := TRUE;   // SR flip-flop
   END_IF;
   IF #Mx_ET111 THEN #Mx_ET110 := FALSE; END_IF;
END_REGION

REGION Network 54: ET12 - CONTROL CARGA MESA (ENTRADA POR E1 O E3)
   RUNG wire#powerrail
      Contact( #Mx_ET11 )
      I_Contact( #MEnt_DescargaAct )
      Contact( #FTF_MEnt )
      S_SR(operand := #Mx_ET12, r1 := #Mx_ET02)
   END_RUNG
   // the same network as SCL:
   IF #Mx_ET11 AND NOT #MEnt_DescargaAct AND #FTF_MEnt THEN
       #Mx_ET12 := TRUE;   // SR flip-flop
   END_IF;
   IF #Mx_ET02 THEN #Mx_ET12 := FALSE; END_IF;
END_REGION

REGION Network 55: ET11
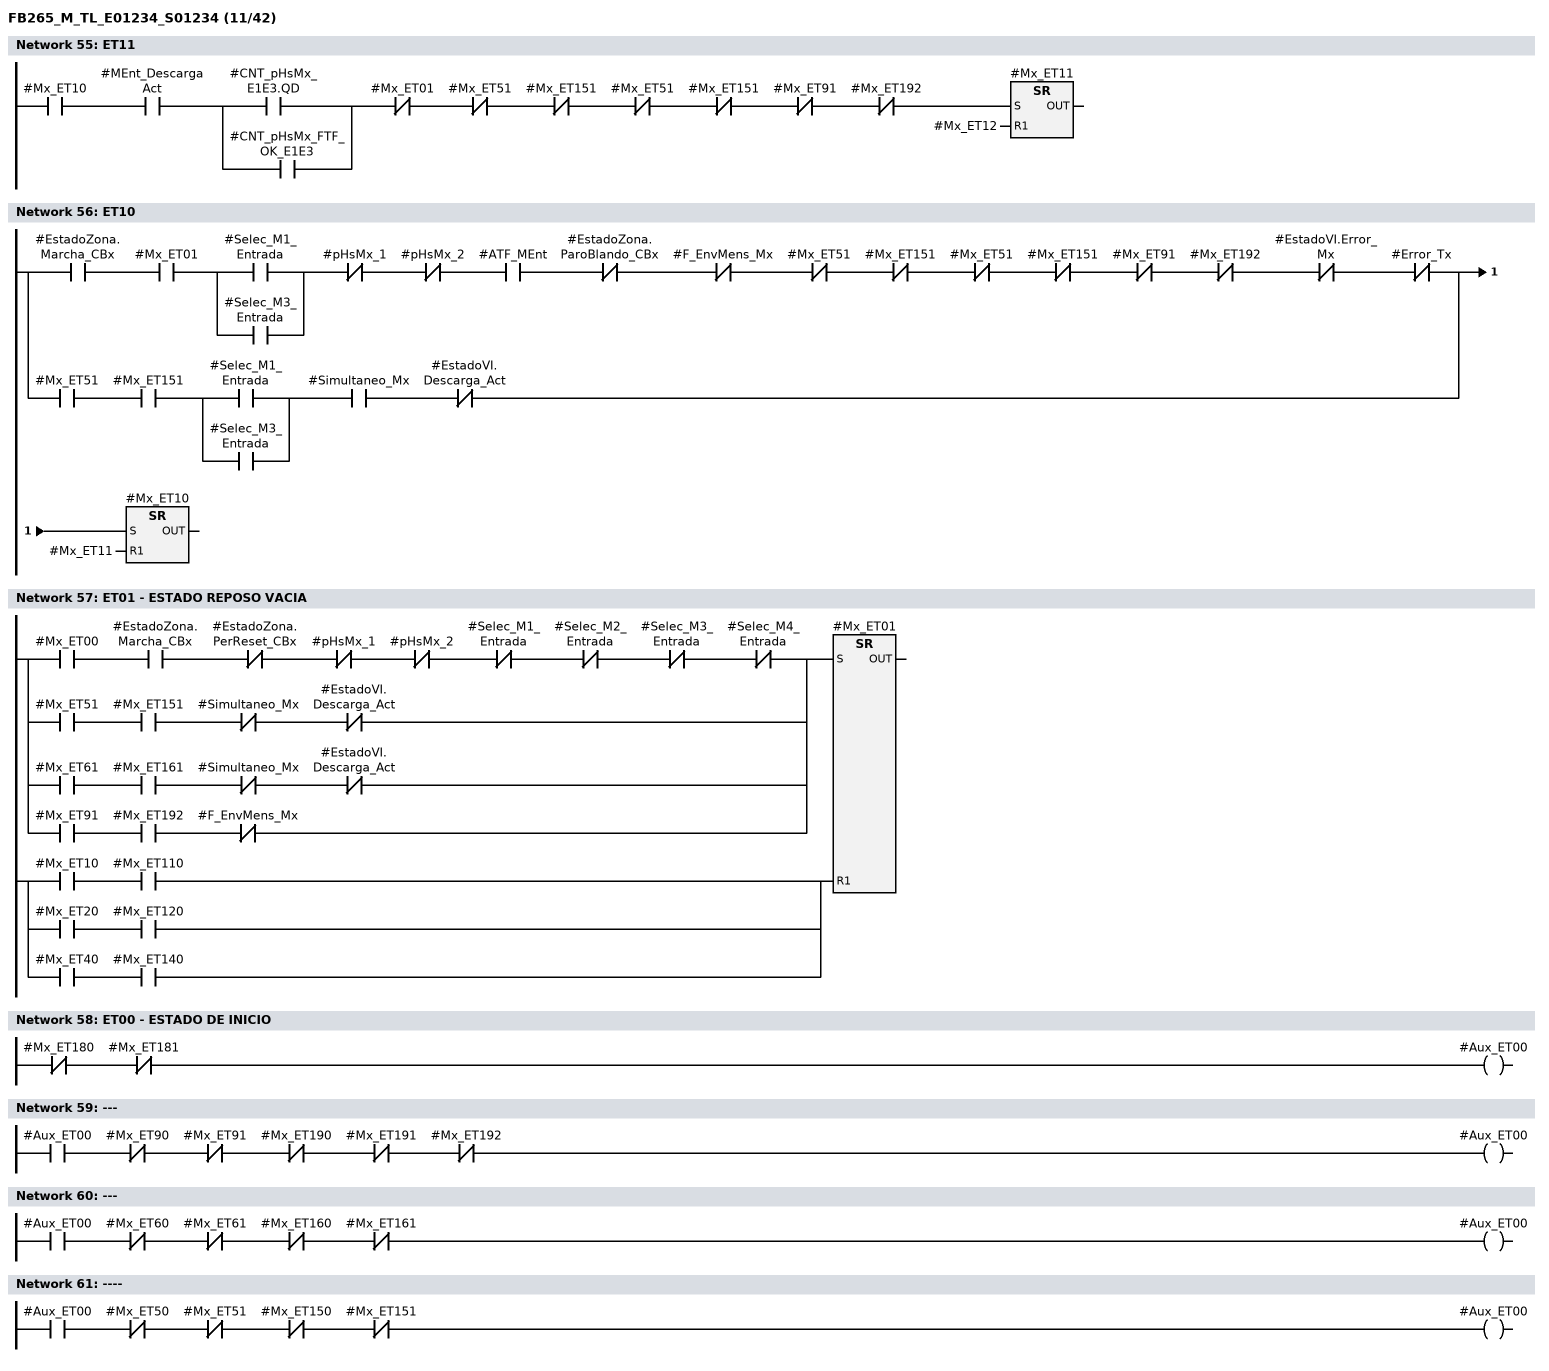
   RUNG wire#powerrail
      Contact( #Mx_ET10 )
      Contact( #MEnt_DescargaAct )
      wire#w1
      Contact( #CNT_pHsMx_E1E3.QD )
      wire#w2
      I_Contact( #Mx_ET01 )
      I_Contact( #Mx_ET51 )
      I_Contact( #Mx_ET151 )
      I_Contact( #Mx_ET51 )
      I_Contact( #Mx_ET151 )
      I_Contact( #Mx_ET91 )
      I_Contact( #Mx_ET192 )
      S_SR(operand := #Mx_ET11, r1 := #Mx_ET12)
   END_RUNG
   RUNG wire#w1
      Contact( #CNT_pHsMx_FTF_OK_E1E3 )
   END_RUNG wire#w2
   // the same network as SCL:
   IF #Mx_ET10 AND #MEnt_DescargaAct AND (#CNT_pHsMx_E1E3.QD OR #CNT_pHsMx_FTF_OK_E1E3) AND NOT #Mx_ET01 AND NOT #Mx_ET51 AND NOT #Mx_ET151 AND NOT #Mx_ET51 AND NOT #Mx_ET151 AND NOT #Mx_ET91 AND NOT #Mx_ET192 THEN
       #Mx_ET11 := TRUE;   // SR flip-flop
   END_IF;
   IF #Mx_ET12 THEN #Mx_ET11 := FALSE; END_IF;
END_REGION

REGION Network 56: ET10
   RUNG wire#powerrail
      Contact( #EstadoZona.Marcha_CBx )
      Contact( #Mx_ET01 )
      wire#w1
      Contact( #Selec_M1_Entrada )
      wire#w2
      I_Contact( #pHsMx_1 )
      I_Contact( #pHsMx_2 )
      Contact( #ATF_MEnt )
      I_Contact( #EstadoZona.ParoBlando_CBx )
      I_Contact( #F_EnvMens_Mx )
      I_Contact( #Mx_ET51 )
      I_Contact( #Mx_ET151 )
      I_Contact( #Mx_ET51 )
      I_Contact( #Mx_ET151 )
      I_Contact( #Mx_ET91 )
      I_Contact( #Mx_ET192 )
      I_Contact( #EstadoVI.Error_Mx )
      I_Contact( #Error_Tx )
      wire#w3
      S_SR(operand := #Mx_ET10, r1 := #Mx_ET11)
   END_RUNG
   RUNG wire#w1
      Contact( #Selec_M3_Entrada )
   END_RUNG wire#w2
   RUNG wire#powerrail
      Contact( #Mx_ET51 )
      Contact( #Mx_ET151 )
      wire#w4
      Contact( #Selec_M1_Entrada )
      wire#w5
      Contact( #Simultaneo_Mx )
      I_Contact( #EstadoVI.Descarga_Act )
   END_RUNG wire#w3
   RUNG wire#w4
      Contact( #Selec_M3_Entrada )
   END_RUNG wire#w5
   // the same network as SCL:
   IF (#EstadoZona.Marcha_CBx AND #Mx_ET01 AND (#Selec_M1_Entrada OR #Selec_M3_Entrada) AND NOT #pHsMx_1 AND NOT #pHsMx_2 AND #ATF_MEnt AND NOT #EstadoZona.ParoBlando_CBx AND NOT #F_EnvMens_Mx AND NOT #Mx_ET51 AND NOT #Mx_ET151 AND NOT #Mx_ET51 AND NOT #Mx_ET151 AND NOT #Mx_ET91 AND NOT #Mx_ET192 AND NOT #EstadoVI.Error_Mx AND NOT #Error_Tx) OR (#Mx_ET51 AND #Mx_ET151 AND (#Selec_M1_Entrada OR #Selec_M3_Entrada) AND #Simultaneo_Mx AND NOT #EstadoVI.Descarga_Act) THEN
       #Mx_ET10 := TRUE;   // SR flip-flop
   END_IF;
   IF #Mx_ET11 THEN #Mx_ET10 := FALSE; END_IF;
END_REGION

REGION Network 57: ET01 - ESTADO REPOSO VACIA
   RUNG wire#powerrail
      Contact( #Mx_ET00 )
      Contact( #EstadoZona.Marcha_CBx )
      I_Contact( #EstadoZona.PerReset_CBx )
      I_Contact( #pHsMx_1 )
      I_Contact( #pHsMx_2 )
      I_Contact( #Selec_M1_Entrada )
      I_Contact( #Selec_M2_Entrada )
      I_Contact( #Selec_M3_Entrada )
      I_Contact( #Selec_M4_Entrada )
      wire#w1
      S_SR(operand := #Mx_ET01, r1 := wire#w2)
   END_RUNG
   RUNG wire#powerrail
      Contact( #Mx_ET51 )
      Contact( #Mx_ET151 )
      I_Contact( #Simultaneo_Mx )
      I_Contact( #EstadoVI.Descarga_Act )
   END_RUNG wire#w1
   RUNG wire#powerrail
      Contact( #Mx_ET61 )
      Contact( #Mx_ET161 )
      I_Contact( #Simultaneo_Mx )
      I_Contact( #EstadoVI.Descarga_Act )
   END_RUNG wire#w1
   RUNG wire#powerrail
      Contact( #Mx_ET91 )
      Contact( #Mx_ET192 )
      I_Contact( #F_EnvMens_Mx )
   END_RUNG wire#w1
   RUNG wire#powerrail
      Contact( #Mx_ET10 )
      Contact( #Mx_ET110 )
   END_RUNG wire#w2
   RUNG wire#powerrail
      Contact( #Mx_ET20 )
      Contact( #Mx_ET120 )
   END_RUNG wire#w2
   RUNG wire#powerrail
      Contact( #Mx_ET40 )
      Contact( #Mx_ET140 )
   END_RUNG wire#w2
   // the same network as SCL:
   IF (#Mx_ET00 AND #EstadoZona.Marcha_CBx AND NOT #EstadoZona.PerReset_CBx AND NOT #pHsMx_1 AND NOT #pHsMx_2 AND NOT #Selec_M1_Entrada AND NOT #Selec_M2_Entrada AND NOT #Selec_M3_Entrada AND NOT #Selec_M4_Entrada) OR (#Mx_ET51 AND #Mx_ET151 AND NOT #Simultaneo_Mx AND NOT #EstadoVI.Descarga_Act) OR (#Mx_ET61 AND #Mx_ET161 AND NOT #Simultaneo_Mx AND NOT #EstadoVI.Descarga_Act) OR (#Mx_ET91 AND #Mx_ET192 AND NOT #F_EnvMens_Mx) THEN
       #Mx_ET01 := TRUE;   // SR flip-flop
   END_IF;
   IF (#Mx_ET10 AND #Mx_ET110) OR (#Mx_ET20 AND #Mx_ET120) OR (#Mx_ET40 AND #Mx_ET140) THEN
       #Mx_ET01 := FALSE;
   END_IF;
END_REGION

REGION Network 58: ET00 - ESTADO DE INICIO
   RUNG wire#powerrail
      I_Contact( #Mx_ET180 )
      I_Contact( #Mx_ET181 )
      Coil( #Aux_ET00 )
   END_RUNG
   // the same network as SCL:
   #Aux_ET00 := NOT #Mx_ET180 AND NOT #Mx_ET181;
END_REGION

REGION Network 59: ---
   RUNG wire#powerrail
      Contact( #Aux_ET00 )
      I_Contact( #Mx_ET90 )
      I_Contact( #Mx_ET91 )
      I_Contact( #Mx_ET190 )
      I_Contact( #Mx_ET191 )
      I_Contact( #Mx_ET192 )
      Coil( #Aux_ET00 )
   END_RUNG
   // the same network as SCL:
   #Aux_ET00 := #Aux_ET00 AND NOT #Mx_ET90 AND NOT #Mx_ET91 AND NOT #Mx_ET190 AND NOT #Mx_ET191 AND NOT #Mx_ET192;
END_REGION

REGION Network 60: ---
   RUNG wire#powerrail
      Contact( #Aux_ET00 )
      I_Contact( #Mx_ET60 )
      I_Contact( #Mx_ET61 )
      I_Contact( #Mx_ET160 )
      I_Contact( #Mx_ET161 )
      Coil( #Aux_ET00 )
   END_RUNG
   // the same network as SCL:
   #Aux_ET00 := #Aux_ET00 AND NOT #Mx_ET60 AND NOT #Mx_ET61 AND NOT #Mx_ET160 AND NOT #Mx_ET161;
END_REGION

REGION Network 61: ----
   RUNG wire#powerrail
      Contact( #Aux_ET00 )
      I_Contact( #Mx_ET50 )
      I_Contact( #Mx_ET51 )
      I_Contact( #Mx_ET150 )
      I_Contact( #Mx_ET151 )
      Coil( #Aux_ET00 )
   END_RUNG
   // the same network as SCL:
   #Aux_ET00 := #Aux_ET00 AND NOT #Mx_ET50 AND NOT #Mx_ET51 AND NOT #Mx_ET150 AND NOT #Mx_ET151;
END_REGION

REGION Network 62: ----
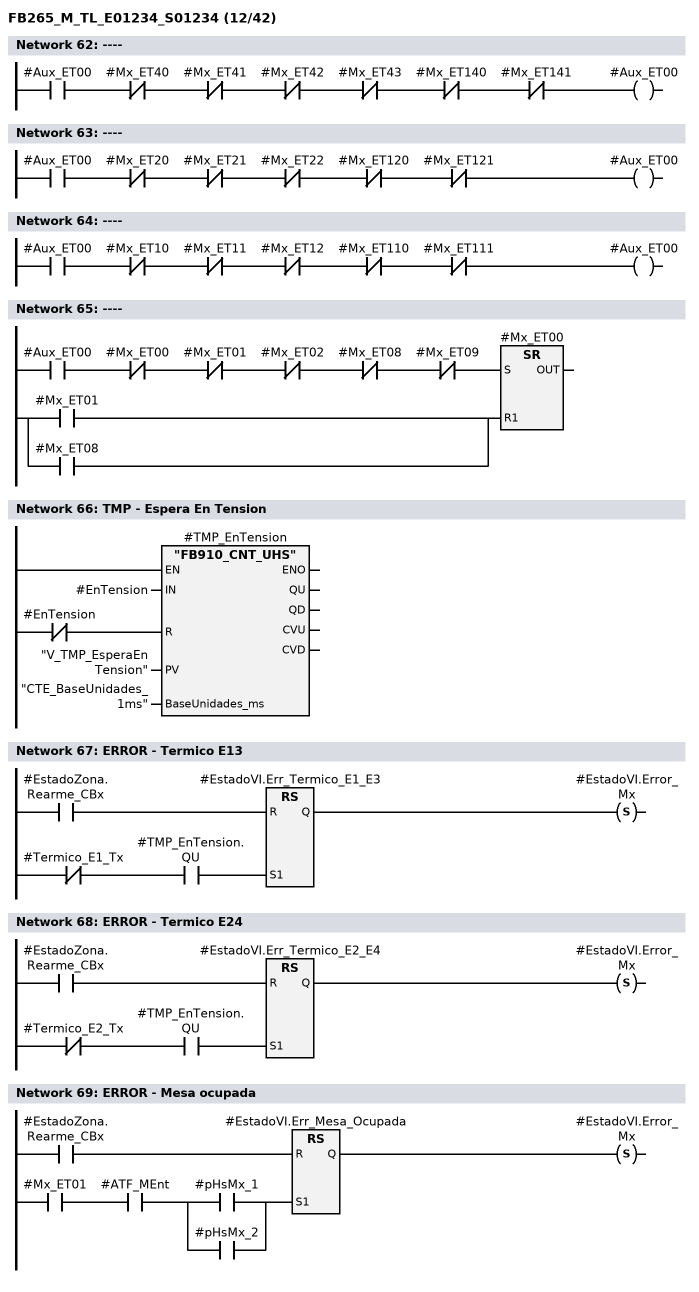
   RUNG wire#powerrail
      Contact( #Aux_ET00 )
      I_Contact( #Mx_ET40 )
      I_Contact( #Mx_ET41 )
      I_Contact( #Mx_ET42 )
      I_Contact( #Mx_ET43 )
      I_Contact( #Mx_ET140 )
      I_Contact( #Mx_ET141 )
      Coil( #Aux_ET00 )
   END_RUNG
   // the same network as SCL:
   #Aux_ET00 := #Aux_ET00 AND NOT #Mx_ET40 AND NOT #Mx_ET41 AND NOT #Mx_ET42 AND NOT #Mx_ET43 AND NOT #Mx_ET140 AND NOT #Mx_ET141;
END_REGION

REGION Network 63: ----
   RUNG wire#powerrail
      Contact( #Aux_ET00 )
      I_Contact( #Mx_ET20 )
      I_Contact( #Mx_ET21 )
      I_Contact( #Mx_ET22 )
      I_Contact( #Mx_ET120 )
      I_Contact( #Mx_ET121 )
      Coil( #Aux_ET00 )
   END_RUNG
   // the same network as SCL:
   #Aux_ET00 := #Aux_ET00 AND NOT #Mx_ET20 AND NOT #Mx_ET21 AND NOT #Mx_ET22 AND NOT #Mx_ET120 AND NOT #Mx_ET121;
END_REGION

REGION Network 64: ----
   RUNG wire#powerrail
      Contact( #Aux_ET00 )
      I_Contact( #Mx_ET10 )
      I_Contact( #Mx_ET11 )
      I_Contact( #Mx_ET12 )
      I_Contact( #Mx_ET110 )
      I_Contact( #Mx_ET111 )
      Coil( #Aux_ET00 )
   END_RUNG
   // the same network as SCL:
   #Aux_ET00 := #Aux_ET00 AND NOT #Mx_ET10 AND NOT #Mx_ET11 AND NOT #Mx_ET12 AND NOT #Mx_ET110 AND NOT #Mx_ET111;
END_REGION

REGION Network 65: ----
   RUNG wire#powerrail
      Contact( #Aux_ET00 )
      I_Contact( #Mx_ET00 )
      I_Contact( #Mx_ET01 )
      I_Contact( #Mx_ET02 )
      I_Contact( #Mx_ET08 )
      I_Contact( #Mx_ET09 )
      S_SR(operand := #Mx_ET00, r1 := wire#w1)
   END_RUNG
   RUNG wire#powerrail
      Contact( #Mx_ET01 )
   END_RUNG wire#w1
   RUNG wire#powerrail
      Contact( #Mx_ET08 )
   END_RUNG wire#w1
   // the same network as SCL:
   IF #Aux_ET00 AND NOT #Mx_ET00 AND NOT #Mx_ET01 AND NOT #Mx_ET02 AND NOT #Mx_ET08 AND NOT #Mx_ET09 THEN
       #Mx_ET00 := TRUE;   // SR flip-flop
   END_IF;
   IF #Mx_ET01 OR #Mx_ET08 THEN #Mx_ET00 := FALSE; END_IF;
END_REGION

REGION Network 66: TMP - Espera En Tension
   RUNG wire#powerrail
      #TMP_EnTension(R := wire#w1, IN := #EnTension, PV := "V_TMP_EsperaEnTension", BaseUnidades_ms := "CTE_BaseUnidades_1ms", QU =>, QD =>, CVU =>, CVD =>)
   END_RUNG
   RUNG wire#powerrail
      I_Contact( #EnTension )
   END_RUNG wire#w1
   // the same network as SCL:
   #TMP_EnTension(IN := #EnTension,   // "FB910_CNT_UHS"
                  R := NOT #EnTension,
                  PV := "V_TMP_EsperaEnTension",
                  BaseUnidades_ms := "CTE_BaseUnidades_1ms");
END_REGION

REGION Network 67: ERROR - Termico E13
   RUNG wire#powerrail
      Contact( #EstadoZona.Rearme_CBx )
      S_RS(operand := #EstadoVI.Err_Termico_E1_E3, s1 := wire#w1)
      S_Coil( #EstadoVI.Error_Mx )
   END_RUNG
   RUNG wire#powerrail
      I_Contact( #Termico_E1_Tx )
      Contact( #TMP_EnTension.QU )
   END_RUNG wire#w1
   // the same network as SCL:
   IF #EstadoZona.Rearme_CBx THEN
       #EstadoVI.Err_Termico_E1_E3 := FALSE;   // RS flip-flop
   END_IF;
   IF NOT #Termico_E1_Tx AND #TMP_EnTension.QU THEN #EstadoVI.Err_Termico_E1_E3 := TRUE; END_IF;
   IF #EstadoVI.Err_Termico_E1_E3 THEN #EstadoVI.Error_Mx := TRUE; END_IF;
END_REGION

REGION Network 68: ERROR - Termico E24
   RUNG wire#powerrail
      Contact( #EstadoZona.Rearme_CBx )
      S_RS(operand := #EstadoVI.Err_Termico_E2_E4, s1 := wire#w1)
      S_Coil( #EstadoVI.Error_Mx )
   END_RUNG
   RUNG wire#powerrail
      I_Contact( #Termico_E2_Tx )
      Contact( #TMP_EnTension.QU )
   END_RUNG wire#w1
   // the same network as SCL:
   IF #EstadoZona.Rearme_CBx THEN
       #EstadoVI.Err_Termico_E2_E4 := FALSE;   // RS flip-flop
   END_IF;
   IF NOT #Termico_E2_Tx AND #TMP_EnTension.QU THEN #EstadoVI.Err_Termico_E2_E4 := TRUE; END_IF;
   IF #EstadoVI.Err_Termico_E2_E4 THEN #EstadoVI.Error_Mx := TRUE; END_IF;
END_REGION

REGION Network 69: ERROR - Mesa ocupada
   RUNG wire#powerrail
      Contact( #EstadoZona.Rearme_CBx )
      S_RS(operand := #EstadoVI.Err_Mesa_Ocupada, s1 := wire#w2)
      S_Coil( #EstadoVI.Error_Mx )
   END_RUNG
   RUNG wire#powerrail
      Contact( #Mx_ET01 )
      Contact( #ATF_MEnt )
      wire#w1
      Contact( #pHsMx_1 )
   END_RUNG wire#w2
   RUNG wire#w1
      Contact( #pHsMx_2 )
   END_RUNG wire#w2
   // the same network as SCL:
   IF #EstadoZona.Rearme_CBx THEN
       #EstadoVI.Err_Mesa_Ocupada := FALSE;   // RS flip-flop
   END_IF;
   IF #Mx_ET01 AND #ATF_MEnt AND (#pHsMx_1 OR #pHsMx_2) THEN #EstadoVI.Err_Mesa_Ocupada := TRUE; END_IF;
   IF #EstadoVI.Err_Mesa_Ocupada THEN #EstadoVI.Error_Mx := TRUE; END_IF;
END_REGION

REGION Network 70: CNT - ERROR - Arrastre
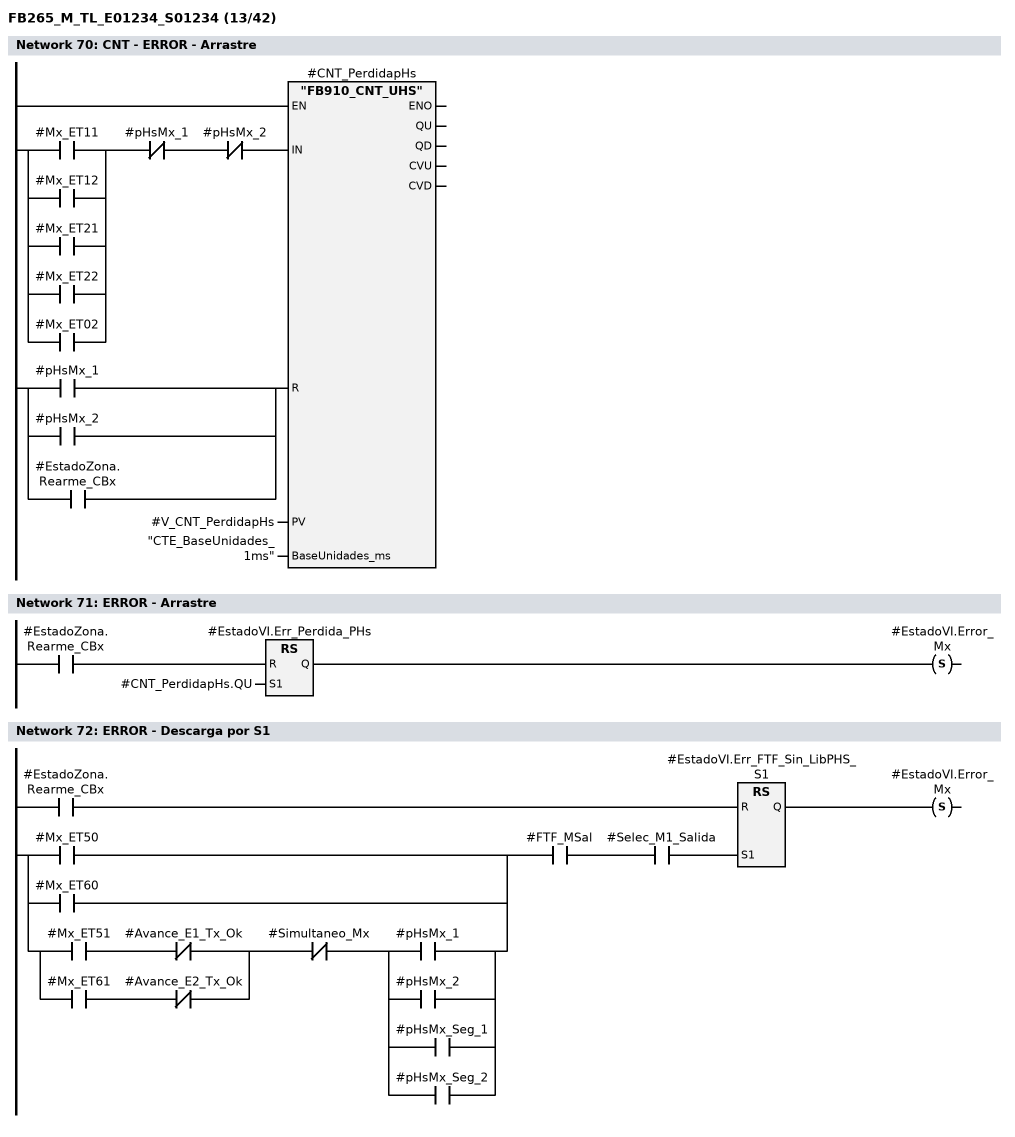
   RUNG wire#powerrail
      #CNT_PerdidapHs(IN := wire#w2, R := wire#w3, PV := #V_CNT_PerdidapHs, BaseUnidades_ms := "CTE_BaseUnidades_1ms", QU =>, QD =>, CVU =>, CVD =>)
   END_RUNG
   RUNG wire#powerrail
      Contact( #Mx_ET11 )
      wire#w1
      I_Contact( #pHsMx_1 )
      I_Contact( #pHsMx_2 )
   END_RUNG wire#w2
   RUNG wire#powerrail
      Contact( #Mx_ET12 )
   END_RUNG wire#w1
   RUNG wire#powerrail
      Contact( #Mx_ET21 )
   END_RUNG wire#w1
   RUNG wire#powerrail
      Contact( #Mx_ET22 )
   END_RUNG wire#w1
   RUNG wire#powerrail
      Contact( #Mx_ET02 )
   END_RUNG wire#w1
   RUNG wire#powerrail
      Contact( #pHsMx_1 )
   END_RUNG wire#w3
   RUNG wire#powerrail
      Contact( #pHsMx_2 )
   END_RUNG wire#w3
   RUNG wire#powerrail
      Contact( #EstadoZona.Rearme_CBx )
   END_RUNG wire#w3
   // the same network as SCL:
   #CNT_PerdidapHs(IN := (#Mx_ET11 OR #Mx_ET12 OR #Mx_ET21 OR #Mx_ET22 OR #Mx_ET02) AND NOT #pHsMx_1 AND NOT #pHsMx_2,   // "FB910_CNT_UHS"
                   R := #pHsMx_1 OR #pHsMx_2 OR #EstadoZona.Rearme_CBx,
                   PV := #V_CNT_PerdidapHs,
                   BaseUnidades_ms := "CTE_BaseUnidades_1ms");
END_REGION

REGION Network 71: ERROR - Arrastre
   RUNG wire#powerrail
      Contact( #EstadoZona.Rearme_CBx )
      S_RS(operand := #EstadoVI.Err_Perdida_PHs, s1 := #CNT_PerdidapHs.QU)
      S_Coil( #EstadoVI.Error_Mx )
   END_RUNG
   // the same network as SCL:
   IF #EstadoZona.Rearme_CBx THEN
       #EstadoVI.Err_Perdida_PHs := FALSE;   // RS flip-flop
   END_IF;
   IF #CNT_PerdidapHs.QU THEN #EstadoVI.Err_Perdida_PHs := TRUE; END_IF;
   IF #EstadoVI.Err_Perdida_PHs THEN #EstadoVI.Error_Mx := TRUE; END_IF;
END_REGION

REGION Network 72: ERROR - Descarga por S1
   RUNG wire#powerrail
      Contact( #EstadoZona.Rearme_CBx )
      S_RS(operand := #EstadoVI.Err_FTF_Sin_LibPHS_S1, s1 := wire#w4)
      S_Coil( #EstadoVI.Error_Mx )
   END_RUNG
   RUNG wire#powerrail
      Contact( #Mx_ET50 )
      wire#w1
      Contact( #FTF_MSal )
      Contact( #Selec_M1_Salida )
   END_RUNG wire#w4
   RUNG wire#powerrail
      Contact( #Mx_ET60 )
   END_RUNG wire#w1
   RUNG wire#powerrail
      Contact( #Mx_ET51 )
      I_Contact( #Avance_E1_Tx_Ok )
      wire#w2
      I_Contact( #Simultaneo_Mx )
      wire#w3
      Contact( #pHsMx_1 )
   END_RUNG wire#w1
   RUNG wire#powerrail
      Contact( #Mx_ET61 )
      I_Contact( #Avance_E2_Tx_Ok )
   END_RUNG wire#w2
   RUNG wire#w3
      Contact( #pHsMx_2 )
   END_RUNG wire#w1
   RUNG wire#w3
      Contact( #pHsMx_Seg_1 )
   END_RUNG wire#w1
   RUNG wire#w3
      Contact( #pHsMx_Seg_2 )
   END_RUNG wire#w1
   // the same network as SCL:
   IF #EstadoZona.Rearme_CBx THEN
       #EstadoVI.Err_FTF_Sin_LibPHS_S1 := FALSE;   // RS flip-flop
   END_IF;
   IF (#Mx_ET50 OR #Mx_ET60 OR (((#Mx_ET51 AND NOT #Avance_E1_Tx_Ok) OR (#Mx_ET61 AND NOT #Avance_E2_Tx_Ok)) AND NOT #Simultaneo_Mx AND (#pHsMx_1 OR #pHsMx_2 OR #pHsMx_Seg_1 OR #pHsMx_Seg_2))) AND #FTF_MSal AND #Selec_M1_Salida THEN
       #EstadoVI.Err_FTF_Sin_LibPHS_S1 := TRUE;
   END_IF;
   IF #EstadoVI.Err_FTF_Sin_LibPHS_S1 THEN #EstadoVI.Error_Mx := TRUE; END_IF;
END_REGION

REGION Network 73: ERROR - Descarga por S2
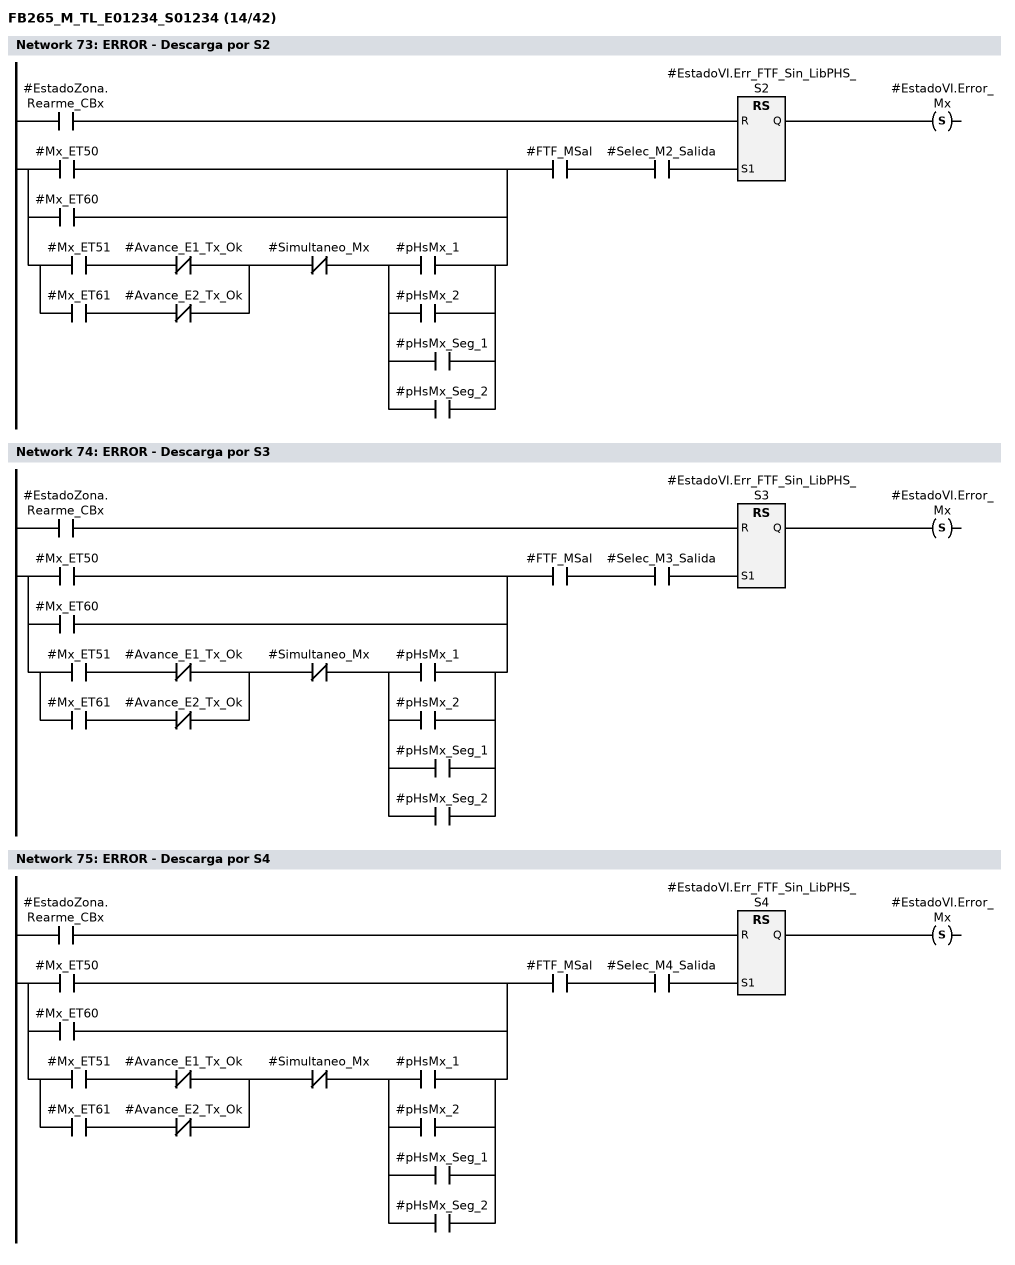
   RUNG wire#powerrail
      Contact( #EstadoZona.Rearme_CBx )
      S_RS(operand := #EstadoVI.Err_FTF_Sin_LibPHS_S2, s1 := wire#w4)
      S_Coil( #EstadoVI.Error_Mx )
   END_RUNG
   RUNG wire#powerrail
      Contact( #Mx_ET50 )
      wire#w1
      Contact( #FTF_MSal )
      Contact( #Selec_M2_Salida )
   END_RUNG wire#w4
   RUNG wire#powerrail
      Contact( #Mx_ET60 )
   END_RUNG wire#w1
   RUNG wire#powerrail
      Contact( #Mx_ET51 )
      I_Contact( #Avance_E1_Tx_Ok )
      wire#w2
      I_Contact( #Simultaneo_Mx )
      wire#w3
      Contact( #pHsMx_1 )
   END_RUNG wire#w1
   RUNG wire#powerrail
      Contact( #Mx_ET61 )
      I_Contact( #Avance_E2_Tx_Ok )
   END_RUNG wire#w2
   RUNG wire#w3
      Contact( #pHsMx_2 )
   END_RUNG wire#w1
   RUNG wire#w3
      Contact( #pHsMx_Seg_1 )
   END_RUNG wire#w1
   RUNG wire#w3
      Contact( #pHsMx_Seg_2 )
   END_RUNG wire#w1
   // the same network as SCL:
   IF #EstadoZona.Rearme_CBx THEN
       #EstadoVI.Err_FTF_Sin_LibPHS_S2 := FALSE;   // RS flip-flop
   END_IF;
   IF (#Mx_ET50 OR #Mx_ET60 OR (((#Mx_ET51 AND NOT #Avance_E1_Tx_Ok) OR (#Mx_ET61 AND NOT #Avance_E2_Tx_Ok)) AND NOT #Simultaneo_Mx AND (#pHsMx_1 OR #pHsMx_2 OR #pHsMx_Seg_1 OR #pHsMx_Seg_2))) AND #FTF_MSal AND #Selec_M2_Salida THEN
       #EstadoVI.Err_FTF_Sin_LibPHS_S2 := TRUE;
   END_IF;
   IF #EstadoVI.Err_FTF_Sin_LibPHS_S2 THEN #EstadoVI.Error_Mx := TRUE; END_IF;
END_REGION

REGION Network 74: ERROR - Descarga por S3
   RUNG wire#powerrail
      Contact( #EstadoZona.Rearme_CBx )
      S_RS(operand := #EstadoVI.Err_FTF_Sin_LibPHS_S3, s1 := wire#w4)
      S_Coil( #EstadoVI.Error_Mx )
   END_RUNG
   RUNG wire#powerrail
      Contact( #Mx_ET50 )
      wire#w1
      Contact( #FTF_MSal )
      Contact( #Selec_M3_Salida )
   END_RUNG wire#w4
   RUNG wire#powerrail
      Contact( #Mx_ET60 )
   END_RUNG wire#w1
   RUNG wire#powerrail
      Contact( #Mx_ET51 )
      I_Contact( #Avance_E1_Tx_Ok )
      wire#w2
      I_Contact( #Simultaneo_Mx )
      wire#w3
      Contact( #pHsMx_1 )
   END_RUNG wire#w1
   RUNG wire#powerrail
      Contact( #Mx_ET61 )
      I_Contact( #Avance_E2_Tx_Ok )
   END_RUNG wire#w2
   RUNG wire#w3
      Contact( #pHsMx_2 )
   END_RUNG wire#w1
   RUNG wire#w3
      Contact( #pHsMx_Seg_1 )
   END_RUNG wire#w1
   RUNG wire#w3
      Contact( #pHsMx_Seg_2 )
   END_RUNG wire#w1
   // the same network as SCL:
   IF #EstadoZona.Rearme_CBx THEN
       #EstadoVI.Err_FTF_Sin_LibPHS_S3 := FALSE;   // RS flip-flop
   END_IF;
   IF (#Mx_ET50 OR #Mx_ET60 OR (((#Mx_ET51 AND NOT #Avance_E1_Tx_Ok) OR (#Mx_ET61 AND NOT #Avance_E2_Tx_Ok)) AND NOT #Simultaneo_Mx AND (#pHsMx_1 OR #pHsMx_2 OR #pHsMx_Seg_1 OR #pHsMx_Seg_2))) AND #FTF_MSal AND #Selec_M3_Salida THEN
       #EstadoVI.Err_FTF_Sin_LibPHS_S3 := TRUE;
   END_IF;
   IF #EstadoVI.Err_FTF_Sin_LibPHS_S3 THEN #EstadoVI.Error_Mx := TRUE; END_IF;
END_REGION

REGION Network 75: ERROR - Descarga por S4
   RUNG wire#powerrail
      Contact( #EstadoZona.Rearme_CBx )
      S_RS(operand := #EstadoVI.Err_FTF_Sin_LibPHS_S4, s1 := wire#w4)
      S_Coil( #EstadoVI.Error_Mx )
   END_RUNG
   RUNG wire#powerrail
      Contact( #Mx_ET50 )
      wire#w1
      Contact( #FTF_MSal )
      Contact( #Selec_M4_Salida )
   END_RUNG wire#w4
   RUNG wire#powerrail
      Contact( #Mx_ET60 )
   END_RUNG wire#w1
   RUNG wire#powerrail
      Contact( #Mx_ET51 )
      I_Contact( #Avance_E1_Tx_Ok )
      wire#w2
      I_Contact( #Simultaneo_Mx )
      wire#w3
      Contact( #pHsMx_1 )
   END_RUNG wire#w1
   RUNG wire#powerrail
      Contact( #Mx_ET61 )
      I_Contact( #Avance_E2_Tx_Ok )
   END_RUNG wire#w2
   RUNG wire#w3
      Contact( #pHsMx_2 )
   END_RUNG wire#w1
   RUNG wire#w3
      Contact( #pHsMx_Seg_1 )
   END_RUNG wire#w1
   RUNG wire#w3
      Contact( #pHsMx_Seg_2 )
   END_RUNG wire#w1
   // the same network as SCL:
   IF #EstadoZona.Rearme_CBx THEN
       #EstadoVI.Err_FTF_Sin_LibPHS_S4 := FALSE;   // RS flip-flop
   END_IF;
   IF (#Mx_ET50 OR #Mx_ET60 OR (((#Mx_ET51 AND NOT #Avance_E1_Tx_Ok) OR (#Mx_ET61 AND NOT #Avance_E2_Tx_Ok)) AND NOT #Simultaneo_Mx AND (#pHsMx_1 OR #pHsMx_2 OR #pHsMx_Seg_1 OR #pHsMx_Seg_2))) AND #FTF_MSal AND #Selec_M4_Salida THEN
       #EstadoVI.Err_FTF_Sin_LibPHS_S4 := TRUE;
   END_IF;
   IF #EstadoVI.Err_FTF_Sin_LibPHS_S4 THEN #EstadoVI.Error_Mx := TRUE; END_IF;
END_REGION

REGION Network 76: TMP - ERROR - Tout Avance E1E3
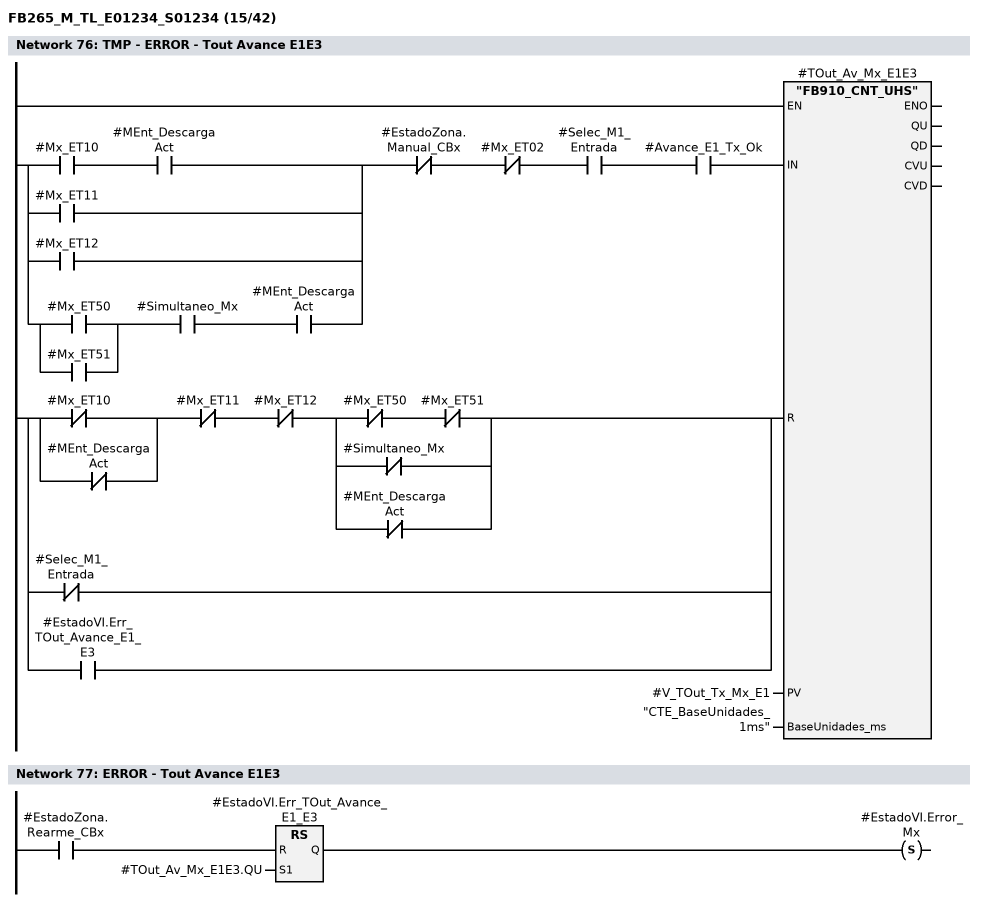
   RUNG wire#powerrail
      #TOut_Av_Mx_E1E3(IN := wire#w3, R := wire#w6, PV := #V_TOut_Tx_Mx_E1, BaseUnidades_ms := "CTE_BaseUnidades_1ms", QU =>, QD =>, CVU =>, CVD =>)
   END_RUNG
   RUNG wire#powerrail
      Contact( #Mx_ET10 )
      Contact( #MEnt_DescargaAct )
      wire#w1
      I_Contact( #EstadoZona.Manual_CBx )
      I_Contact( #Mx_ET02 )
      Contact( #Selec_M1_Entrada )
      Contact( #Avance_E1_Tx_Ok )
   END_RUNG wire#w3
   RUNG wire#powerrail
      Contact( #Mx_ET11 )
   END_RUNG wire#w1
   RUNG wire#powerrail
      Contact( #Mx_ET12 )
   END_RUNG wire#w1
   RUNG wire#powerrail
      Contact( #Mx_ET50 )
      wire#w2
      Contact( #Simultaneo_Mx )
      Contact( #MEnt_DescargaAct )
   END_RUNG wire#w1
   RUNG wire#powerrail
      Contact( #Mx_ET51 )
   END_RUNG wire#w2
   RUNG wire#powerrail
      I_Contact( #Mx_ET10 )
      wire#w4
      I_Contact( #Mx_ET11 )
      I_Contact( #Mx_ET12 )
      wire#w5
      I_Contact( #Mx_ET50 )
      I_Contact( #Mx_ET51 )
   END_RUNG wire#w6
   RUNG wire#powerrail
      I_Contact( #MEnt_DescargaAct )
   END_RUNG wire#w4
   RUNG wire#w5
      I_Contact( #Simultaneo_Mx )
   END_RUNG wire#w6
   RUNG wire#w5
      I_Contact( #MEnt_DescargaAct )
   END_RUNG wire#w6
   RUNG wire#powerrail
      I_Contact( #Selec_M1_Entrada )
   END_RUNG wire#w6
   RUNG wire#powerrail
      Contact( #EstadoVI.Err_TOut_Avance_E1_E3 )
   END_RUNG wire#w6
   // the same network as SCL:
   #TOut_Av_Mx_E1E3(IN := ((#Mx_ET10 AND #MEnt_DescargaAct) OR #Mx_ET11 OR #Mx_ET12 OR ((#Mx_ET50 OR #Mx_ET51) AND #Simultaneo_Mx AND #MEnt_DescargaAct)) AND NOT #EstadoZona.Manual_CBx AND NOT #Mx_ET02 AND #Selec_M1_Entrada AND #Avance_E1_Tx_Ok,   // "FB910_CNT_UHS"
                    R := ((NOT #Mx_ET10 OR NOT #MEnt_DescargaAct) AND NOT #Mx_ET11 AND NOT #Mx_ET12 AND ((NOT #Mx_ET50 AND NOT #Mx_ET51) OR NOT #Simultaneo_Mx OR NOT #MEnt_DescargaAct)) OR NOT #Selec_M1_Entrada OR #EstadoVI.Err_TOut_Avance_E1_E3,
                    PV := #V_TOut_Tx_Mx_E1,
                    BaseUnidades_ms := "CTE_BaseUnidades_1ms");
END_REGION

REGION Network 77: ERROR - Tout Avance E1E3
   RUNG wire#powerrail
      Contact( #EstadoZona.Rearme_CBx )
      S_RS(operand := #EstadoVI.Err_TOut_Avance_E1_E3, s1 := #TOut_Av_Mx_E1E3.QU)
      S_Coil( #EstadoVI.Error_Mx )
   END_RUNG
   // the same network as SCL:
   IF #EstadoZona.Rearme_CBx THEN
       #EstadoVI.Err_TOut_Avance_E1_E3 := FALSE;   // RS flip-flop
   END_IF;
   IF #TOut_Av_Mx_E1E3.QU THEN #EstadoVI.Err_TOut_Avance_E1_E3 := TRUE; END_IF;
   IF #EstadoVI.Err_TOut_Avance_E1_E3 THEN #EstadoVI.Error_Mx := TRUE; END_IF;
END_REGION

REGION Network 78: TMP - ERROR - Tout Retroceso E1E3
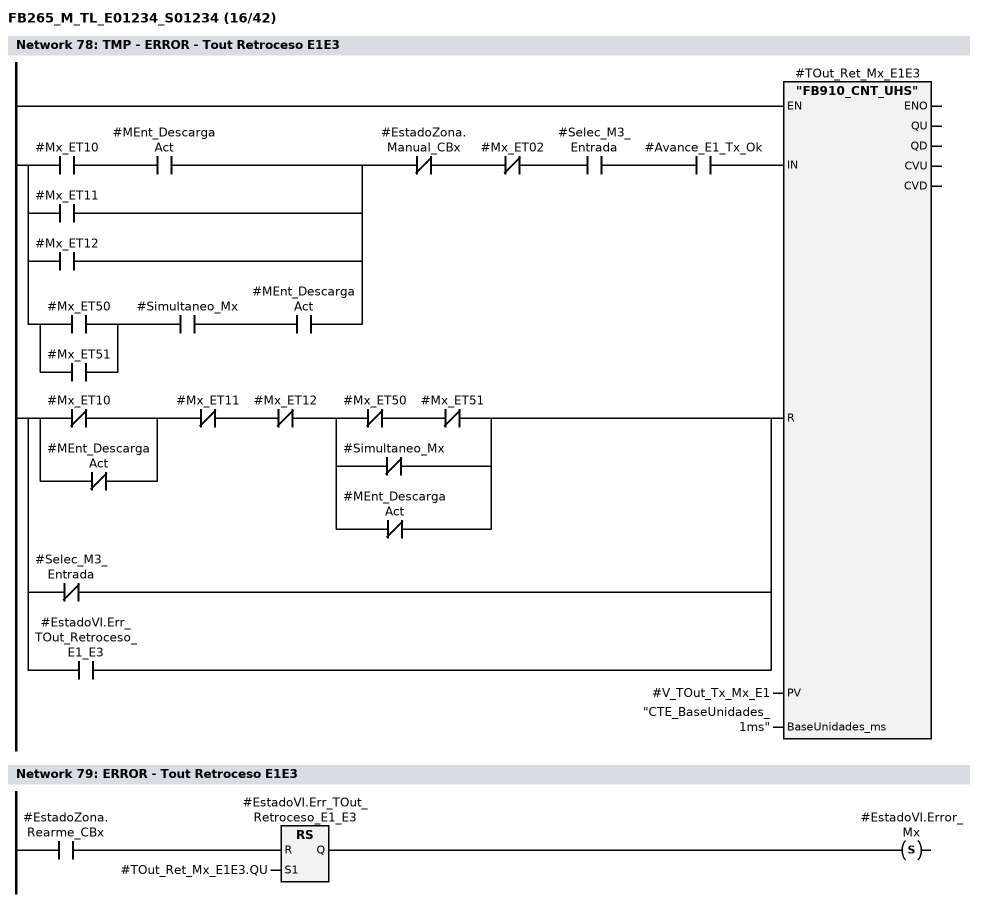
   RUNG wire#powerrail
      #TOut_Ret_Mx_E1E3(IN := wire#w3, R := wire#w6, PV := #V_TOut_Tx_Mx_E1, BaseUnidades_ms := "CTE_BaseUnidades_1ms", QU =>, QD =>, CVU =>, CVD =>)
   END_RUNG
   RUNG wire#powerrail
      Contact( #Mx_ET10 )
      Contact( #MEnt_DescargaAct )
      wire#w1
      I_Contact( #EstadoZona.Manual_CBx )
      I_Contact( #Mx_ET02 )
      Contact( #Selec_M3_Entrada )
      Contact( #Avance_E1_Tx_Ok )
   END_RUNG wire#w3
   RUNG wire#powerrail
      Contact( #Mx_ET11 )
   END_RUNG wire#w1
   RUNG wire#powerrail
      Contact( #Mx_ET12 )
   END_RUNG wire#w1
   RUNG wire#powerrail
      Contact( #Mx_ET50 )
      wire#w2
      Contact( #Simultaneo_Mx )
      Contact( #MEnt_DescargaAct )
   END_RUNG wire#w1
   RUNG wire#powerrail
      Contact( #Mx_ET51 )
   END_RUNG wire#w2
   RUNG wire#powerrail
      I_Contact( #Mx_ET10 )
      wire#w4
      I_Contact( #Mx_ET11 )
      I_Contact( #Mx_ET12 )
      wire#w5
      I_Contact( #Mx_ET50 )
      I_Contact( #Mx_ET51 )
   END_RUNG wire#w6
   RUNG wire#powerrail
      I_Contact( #MEnt_DescargaAct )
   END_RUNG wire#w4
   RUNG wire#w5
      I_Contact( #Simultaneo_Mx )
   END_RUNG wire#w6
   RUNG wire#w5
      I_Contact( #MEnt_DescargaAct )
   END_RUNG wire#w6
   RUNG wire#powerrail
      I_Contact( #Selec_M3_Entrada )
   END_RUNG wire#w6
   RUNG wire#powerrail
      Contact( #EstadoVI.Err_TOut_Retroceso_E1_E3 )
   END_RUNG wire#w6
   // the same network as SCL:
   #TOut_Ret_Mx_E1E3(IN := ((#Mx_ET10 AND #MEnt_DescargaAct) OR #Mx_ET11 OR #Mx_ET12 OR ((#Mx_ET50 OR #Mx_ET51) AND #Simultaneo_Mx AND #MEnt_DescargaAct)) AND NOT #EstadoZona.Manual_CBx AND NOT #Mx_ET02 AND #Selec_M3_Entrada AND #Avance_E1_Tx_Ok,   // "FB910_CNT_UHS"
                     R := ((NOT #Mx_ET10 OR NOT #MEnt_DescargaAct) AND NOT #Mx_ET11 AND NOT #Mx_ET12 AND ((NOT #Mx_ET50 AND NOT #Mx_ET51) OR NOT #Simultaneo_Mx OR NOT #MEnt_DescargaAct)) OR NOT #Selec_M3_Entrada OR #EstadoVI.Err_TOut_Retroceso_E1_E3,
                     PV := #V_TOut_Tx_Mx_E1,
                     BaseUnidades_ms := "CTE_BaseUnidades_1ms");
END_REGION

REGION Network 79: ERROR - Tout Retroceso E1E3
   RUNG wire#powerrail
      Contact( #EstadoZona.Rearme_CBx )
      S_RS(operand := #EstadoVI.Err_TOut_Retroceso_E1_E3, s1 := #TOut_Ret_Mx_E1E3.QU)
      S_Coil( #EstadoVI.Error_Mx )
   END_RUNG
   // the same network as SCL:
   IF #EstadoZona.Rearme_CBx THEN
       #EstadoVI.Err_TOut_Retroceso_E1_E3 := FALSE;   // RS flip-flop
   END_IF;
   IF #TOut_Ret_Mx_E1E3.QU THEN #EstadoVI.Err_TOut_Retroceso_E1_E3 := TRUE; END_IF;
   IF #EstadoVI.Err_TOut_Retroceso_E1_E3 THEN #EstadoVI.Error_Mx := TRUE; END_IF;
END_REGION

REGION Network 80: TMP - ERROR - Tout Avance E2E4
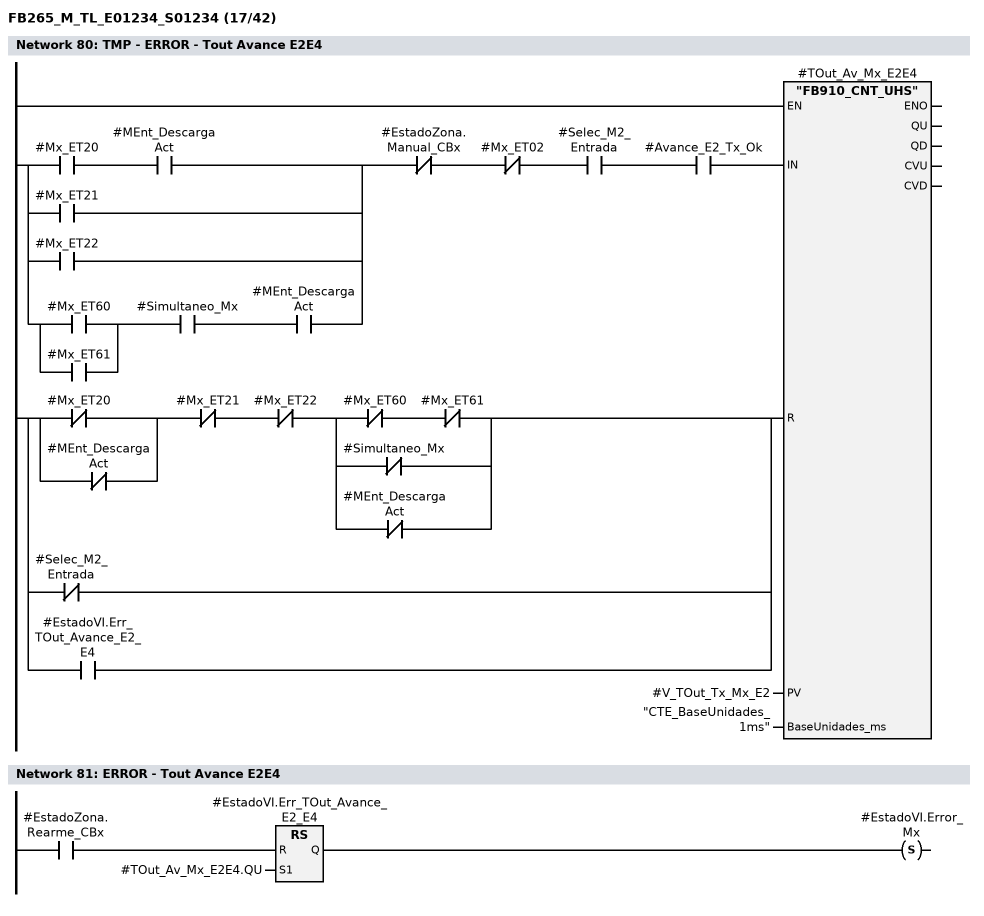
   RUNG wire#powerrail
      #TOut_Av_Mx_E2E4(IN := wire#w3, R := wire#w6, PV := #V_TOut_Tx_Mx_E2, BaseUnidades_ms := "CTE_BaseUnidades_1ms", QU =>, QD =>, CVU =>, CVD =>)
   END_RUNG
   RUNG wire#powerrail
      Contact( #Mx_ET20 )
      Contact( #MEnt_DescargaAct )
      wire#w1
      I_Contact( #EstadoZona.Manual_CBx )
      I_Contact( #Mx_ET02 )
      Contact( #Selec_M2_Entrada )
      Contact( #Avance_E2_Tx_Ok )
   END_RUNG wire#w3
   RUNG wire#powerrail
      Contact( #Mx_ET21 )
   END_RUNG wire#w1
   RUNG wire#powerrail
      Contact( #Mx_ET22 )
   END_RUNG wire#w1
   RUNG wire#powerrail
      Contact( #Mx_ET60 )
      wire#w2
      Contact( #Simultaneo_Mx )
      Contact( #MEnt_DescargaAct )
   END_RUNG wire#w1
   RUNG wire#powerrail
      Contact( #Mx_ET61 )
   END_RUNG wire#w2
   RUNG wire#powerrail
      I_Contact( #Mx_ET20 )
      wire#w4
      I_Contact( #Mx_ET21 )
      I_Contact( #Mx_ET22 )
      wire#w5
      I_Contact( #Mx_ET60 )
      I_Contact( #Mx_ET61 )
   END_RUNG wire#w6
   RUNG wire#powerrail
      I_Contact( #MEnt_DescargaAct )
   END_RUNG wire#w4
   RUNG wire#w5
      I_Contact( #Simultaneo_Mx )
   END_RUNG wire#w6
   RUNG wire#w5
      I_Contact( #MEnt_DescargaAct )
   END_RUNG wire#w6
   RUNG wire#powerrail
      I_Contact( #Selec_M2_Entrada )
   END_RUNG wire#w6
   RUNG wire#powerrail
      Contact( #EstadoVI.Err_TOut_Avance_E2_E4 )
   END_RUNG wire#w6
   // the same network as SCL:
   #TOut_Av_Mx_E2E4(IN := ((#Mx_ET20 AND #MEnt_DescargaAct) OR #Mx_ET21 OR #Mx_ET22 OR ((#Mx_ET60 OR #Mx_ET61) AND #Simultaneo_Mx AND #MEnt_DescargaAct)) AND NOT #EstadoZona.Manual_CBx AND NOT #Mx_ET02 AND #Selec_M2_Entrada AND #Avance_E2_Tx_Ok,   // "FB910_CNT_UHS"
                    R := ((NOT #Mx_ET20 OR NOT #MEnt_DescargaAct) AND NOT #Mx_ET21 AND NOT #Mx_ET22 AND ((NOT #Mx_ET60 AND NOT #Mx_ET61) OR NOT #Simultaneo_Mx OR NOT #MEnt_DescargaAct)) OR NOT #Selec_M2_Entrada OR #EstadoVI.Err_TOut_Avance_E2_E4,
                    PV := #V_TOut_Tx_Mx_E2,
                    BaseUnidades_ms := "CTE_BaseUnidades_1ms");
END_REGION

REGION Network 81: ERROR - Tout Avance E2E4
   RUNG wire#powerrail
      Contact( #EstadoZona.Rearme_CBx )
      S_RS(operand := #EstadoVI.Err_TOut_Avance_E2_E4, s1 := #TOut_Av_Mx_E2E4.QU)
      S_Coil( #EstadoVI.Error_Mx )
   END_RUNG
   // the same network as SCL:
   IF #EstadoZona.Rearme_CBx THEN
       #EstadoVI.Err_TOut_Avance_E2_E4 := FALSE;   // RS flip-flop
   END_IF;
   IF #TOut_Av_Mx_E2E4.QU THEN #EstadoVI.Err_TOut_Avance_E2_E4 := TRUE; END_IF;
   IF #EstadoVI.Err_TOut_Avance_E2_E4 THEN #EstadoVI.Error_Mx := TRUE; END_IF;
END_REGION

REGION Network 82: TMP - ERROR - Tout Retroceso E2E4
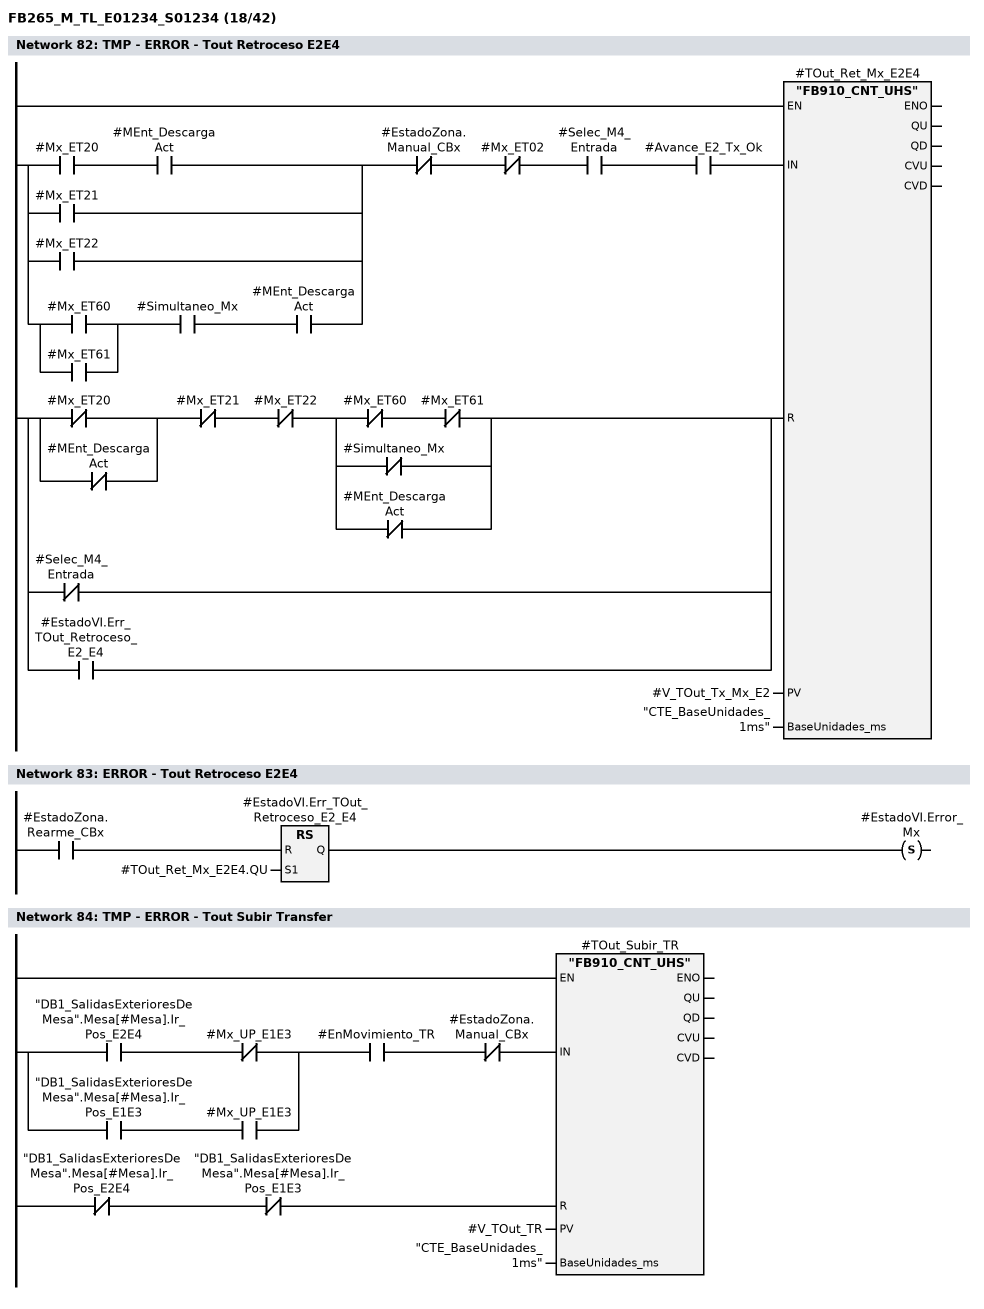
   RUNG wire#powerrail
      #TOut_Ret_Mx_E2E4(IN := wire#w3, R := wire#w6, PV := #V_TOut_Tx_Mx_E2, BaseUnidades_ms := "CTE_BaseUnidades_1ms", QU =>, QD =>, CVU =>, CVD =>)
   END_RUNG
   RUNG wire#powerrail
      Contact( #Mx_ET20 )
      Contact( #MEnt_DescargaAct )
      wire#w1
      I_Contact( #EstadoZona.Manual_CBx )
      I_Contact( #Mx_ET02 )
      Contact( #Selec_M4_Entrada )
      Contact( #Avance_E2_Tx_Ok )
   END_RUNG wire#w3
   RUNG wire#powerrail
      Contact( #Mx_ET21 )
   END_RUNG wire#w1
   RUNG wire#powerrail
      Contact( #Mx_ET22 )
   END_RUNG wire#w1
   RUNG wire#powerrail
      Contact( #Mx_ET60 )
      wire#w2
      Contact( #Simultaneo_Mx )
      Contact( #MEnt_DescargaAct )
   END_RUNG wire#w1
   RUNG wire#powerrail
      Contact( #Mx_ET61 )
   END_RUNG wire#w2
   RUNG wire#powerrail
      I_Contact( #Mx_ET20 )
      wire#w4
      I_Contact( #Mx_ET21 )
      I_Contact( #Mx_ET22 )
      wire#w5
      I_Contact( #Mx_ET60 )
      I_Contact( #Mx_ET61 )
   END_RUNG wire#w6
   RUNG wire#powerrail
      I_Contact( #MEnt_DescargaAct )
   END_RUNG wire#w4
   RUNG wire#w5
      I_Contact( #Simultaneo_Mx )
   END_RUNG wire#w6
   RUNG wire#w5
      I_Contact( #MEnt_DescargaAct )
   END_RUNG wire#w6
   RUNG wire#powerrail
      I_Contact( #Selec_M4_Entrada )
   END_RUNG wire#w6
   RUNG wire#powerrail
      Contact( #EstadoVI.Err_TOut_Retroceso_E2_E4 )
   END_RUNG wire#w6
   // the same network as SCL:
   #TOut_Ret_Mx_E2E4(IN := ((#Mx_ET20 AND #MEnt_DescargaAct) OR #Mx_ET21 OR #Mx_ET22 OR ((#Mx_ET60 OR #Mx_ET61) AND #Simultaneo_Mx AND #MEnt_DescargaAct)) AND NOT #EstadoZona.Manual_CBx AND NOT #Mx_ET02 AND #Selec_M4_Entrada AND #Avance_E2_Tx_Ok,   // "FB910_CNT_UHS"
                     R := ((NOT #Mx_ET20 OR NOT #MEnt_DescargaAct) AND NOT #Mx_ET21 AND NOT #Mx_ET22 AND ((NOT #Mx_ET60 AND NOT #Mx_ET61) OR NOT #Simultaneo_Mx OR NOT #MEnt_DescargaAct)) OR NOT #Selec_M4_Entrada OR #EstadoVI.Err_TOut_Retroceso_E2_E4,
                     PV := #V_TOut_Tx_Mx_E2,
                     BaseUnidades_ms := "CTE_BaseUnidades_1ms");
END_REGION

REGION Network 83: ERROR - Tout Retroceso E2E4
   RUNG wire#powerrail
      Contact( #EstadoZona.Rearme_CBx )
      S_RS(operand := #EstadoVI.Err_TOut_Retroceso_E2_E4, s1 := #TOut_Ret_Mx_E2E4.QU)
      S_Coil( #EstadoVI.Error_Mx )
   END_RUNG
   // the same network as SCL:
   IF #EstadoZona.Rearme_CBx THEN
       #EstadoVI.Err_TOut_Retroceso_E2_E4 := FALSE;   // RS flip-flop
   END_IF;
   IF #TOut_Ret_Mx_E2E4.QU THEN #EstadoVI.Err_TOut_Retroceso_E2_E4 := TRUE; END_IF;
   IF #EstadoVI.Err_TOut_Retroceso_E2_E4 THEN #EstadoVI.Error_Mx := TRUE; END_IF;
END_REGION

REGION Network 84: TMP - ERROR - Tout Subir Transfer
   RUNG wire#powerrail
      #TOut_Subir_TR(IN := wire#w2, R := wire#w3, PV := #V_TOut_TR, BaseUnidades_ms := "CTE_BaseUnidades_1ms", QU =>, QD =>, CVU =>, CVD =>)
   END_RUNG
   RUNG wire#powerrail
      Contact( "DB1_SalidasExterioresDeMesa".Mesa[#Mesa].Ir_Pos_E2E4 )
      I_Contact( #Mx_UP_E1E3 )
      wire#w1
      Contact( #EnMovimiento_TR )
      I_Contact( #EstadoZona.Manual_CBx )
   END_RUNG wire#w2
   RUNG wire#powerrail
      Contact( "DB1_SalidasExterioresDeMesa".Mesa[#Mesa].Ir_Pos_E1E3 )
      Contact( #Mx_UP_E1E3 )
   END_RUNG wire#w1
   RUNG wire#powerrail
      I_Contact( "DB1_SalidasExterioresDeMesa".Mesa[#Mesa].Ir_Pos_E2E4 )
      I_Contact( "DB1_SalidasExterioresDeMesa".Mesa[#Mesa].Ir_Pos_E1E3 )
   END_RUNG wire#w3
   // the same network as SCL:
   #TOut_Subir_TR(IN := (("DB1_SalidasExterioresDeMesa".Mesa[#Mesa].Ir_Pos_E2E4 AND NOT #Mx_UP_E1E3) OR ("DB1_SalidasExterioresDeMesa".Mesa[#Mesa].Ir_Pos_E1E3 AND #Mx_UP_E1E3)) AND #EnMovimiento_TR AND NOT #EstadoZona.Manual_CBx,   // "FB910_CNT_UHS"
                  R := NOT "DB1_SalidasExterioresDeMesa".Mesa[#Mesa].Ir_Pos_E2E4 AND NOT "DB1_SalidasExterioresDeMesa".Mesa[#Mesa].Ir_Pos_E1E3,
                  PV := #V_TOut_TR,
                  BaseUnidades_ms := "CTE_BaseUnidades_1ms");
END_REGION

REGION Network 85: ERROR - Tout subir TR
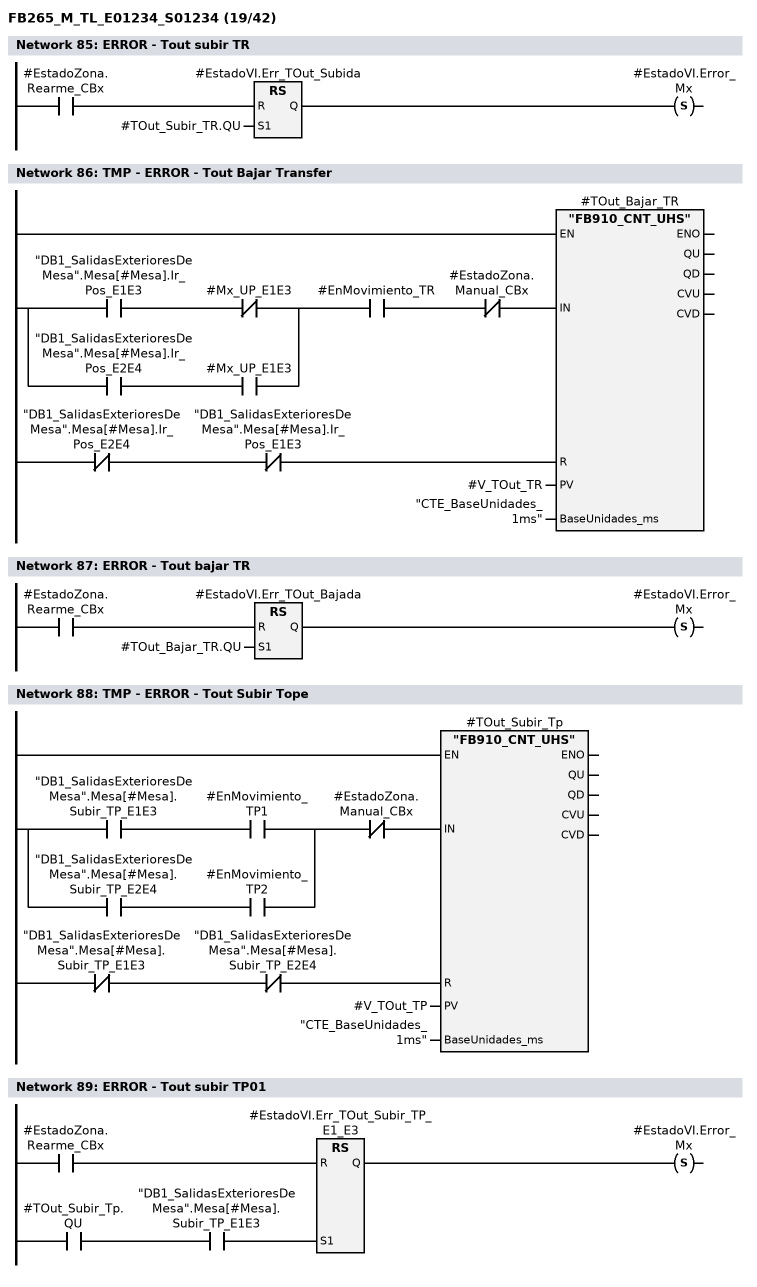
   RUNG wire#powerrail
      Contact( #EstadoZona.Rearme_CBx )
      S_RS(operand := #EstadoVI.Err_TOut_Subida, s1 := #TOut_Subir_TR.QU)
      S_Coil( #EstadoVI.Error_Mx )
   END_RUNG
   // the same network as SCL:
   IF #EstadoZona.Rearme_CBx THEN
       #EstadoVI.Err_TOut_Subida := FALSE;   // RS flip-flop
   END_IF;
   IF #TOut_Subir_TR.QU THEN #EstadoVI.Err_TOut_Subida := TRUE; END_IF;
   IF #EstadoVI.Err_TOut_Subida THEN #EstadoVI.Error_Mx := TRUE; END_IF;
END_REGION

REGION Network 86: TMP - ERROR - Tout Bajar Transfer
   RUNG wire#powerrail
      #TOut_Bajar_TR(IN := wire#w2, R := wire#w3, PV := #V_TOut_TR, BaseUnidades_ms := "CTE_BaseUnidades_1ms", QU =>, QD =>, CVU =>, CVD =>)
   END_RUNG
   RUNG wire#powerrail
      Contact( "DB1_SalidasExterioresDeMesa".Mesa[#Mesa].Ir_Pos_E1E3 )
      I_Contact( #Mx_UP_E1E3 )
      wire#w1
      Contact( #EnMovimiento_TR )
      I_Contact( #EstadoZona.Manual_CBx )
   END_RUNG wire#w2
   RUNG wire#powerrail
      Contact( "DB1_SalidasExterioresDeMesa".Mesa[#Mesa].Ir_Pos_E2E4 )
      Contact( #Mx_UP_E1E3 )
   END_RUNG wire#w1
   RUNG wire#powerrail
      I_Contact( "DB1_SalidasExterioresDeMesa".Mesa[#Mesa].Ir_Pos_E2E4 )
      I_Contact( "DB1_SalidasExterioresDeMesa".Mesa[#Mesa].Ir_Pos_E1E3 )
   END_RUNG wire#w3
   // the same network as SCL:
   #TOut_Bajar_TR(IN := (("DB1_SalidasExterioresDeMesa".Mesa[#Mesa].Ir_Pos_E1E3 AND NOT #Mx_UP_E1E3) OR ("DB1_SalidasExterioresDeMesa".Mesa[#Mesa].Ir_Pos_E2E4 AND #Mx_UP_E1E3)) AND #EnMovimiento_TR AND NOT #EstadoZona.Manual_CBx,   // "FB910_CNT_UHS"
                  R := NOT "DB1_SalidasExterioresDeMesa".Mesa[#Mesa].Ir_Pos_E2E4 AND NOT "DB1_SalidasExterioresDeMesa".Mesa[#Mesa].Ir_Pos_E1E3,
                  PV := #V_TOut_TR,
                  BaseUnidades_ms := "CTE_BaseUnidades_1ms");
END_REGION

REGION Network 87: ERROR - Tout bajar TR
   RUNG wire#powerrail
      Contact( #EstadoZona.Rearme_CBx )
      S_RS(operand := #EstadoVI.Err_TOut_Bajada, s1 := #TOut_Bajar_TR.QU)
      S_Coil( #EstadoVI.Error_Mx )
   END_RUNG
   // the same network as SCL:
   IF #EstadoZona.Rearme_CBx THEN
       #EstadoVI.Err_TOut_Bajada := FALSE;   // RS flip-flop
   END_IF;
   IF #TOut_Bajar_TR.QU THEN #EstadoVI.Err_TOut_Bajada := TRUE; END_IF;
   IF #EstadoVI.Err_TOut_Bajada THEN #EstadoVI.Error_Mx := TRUE; END_IF;
END_REGION

REGION Network 88: TMP - ERROR - Tout Subir Tope
   RUNG wire#powerrail
      #TOut_Subir_Tp(IN := wire#w2, R := wire#w3, PV := #V_TOut_TP, BaseUnidades_ms := "CTE_BaseUnidades_1ms", QU =>, QD =>, CVU =>, CVD =>)
   END_RUNG
   RUNG wire#powerrail
      Contact( "DB1_SalidasExterioresDeMesa".Mesa[#Mesa].Subir_TP_E1E3 )
      Contact( #EnMovimiento_TP1 )
      wire#w1
      I_Contact( #EstadoZona.Manual_CBx )
   END_RUNG wire#w2
   RUNG wire#powerrail
      Contact( "DB1_SalidasExterioresDeMesa".Mesa[#Mesa].Subir_TP_E2E4 )
      Contact( #EnMovimiento_TP2 )
   END_RUNG wire#w1
   RUNG wire#powerrail
      I_Contact( "DB1_SalidasExterioresDeMesa".Mesa[#Mesa].Subir_TP_E1E3 )
      I_Contact( "DB1_SalidasExterioresDeMesa".Mesa[#Mesa].Subir_TP_E2E4 )
   END_RUNG wire#w3
   // the same network as SCL:
   #TOut_Subir_Tp(IN := (("DB1_SalidasExterioresDeMesa".Mesa[#Mesa].Subir_TP_E1E3 AND #EnMovimiento_TP1) OR ("DB1_SalidasExterioresDeMesa".Mesa[#Mesa].Subir_TP_E2E4 AND #EnMovimiento_TP2)) AND NOT #EstadoZona.Manual_CBx,   // "FB910_CNT_UHS"
                  R := NOT "DB1_SalidasExterioresDeMesa".Mesa[#Mesa].Subir_TP_E1E3 AND NOT "DB1_SalidasExterioresDeMesa".Mesa[#Mesa].Subir_TP_E2E4,
                  PV := #V_TOut_TP,
                  BaseUnidades_ms := "CTE_BaseUnidades_1ms");
END_REGION

REGION Network 89: ERROR - Tout subir TP01
   RUNG wire#powerrail
      Contact( #EstadoZona.Rearme_CBx )
      S_RS(operand := #EstadoVI.Err_TOut_Subir_TP_E1_E3, s1 := wire#w1)
      S_Coil( #EstadoVI.Error_Mx )
   END_RUNG
   RUNG wire#powerrail
      Contact( #TOut_Subir_Tp.QU )
      Contact( "DB1_SalidasExterioresDeMesa".Mesa[#Mesa].Subir_TP_E1E3 )
   END_RUNG wire#w1
   // the same network as SCL:
   IF #EstadoZona.Rearme_CBx THEN
       #EstadoVI.Err_TOut_Subir_TP_E1_E3 := FALSE;   // RS flip-flop
   END_IF;
   IF #TOut_Subir_Tp.QU AND "DB1_SalidasExterioresDeMesa".Mesa[#Mesa].Subir_TP_E1E3 THEN
       #EstadoVI.Err_TOut_Subir_TP_E1_E3 := TRUE;
   END_IF;
   IF #EstadoVI.Err_TOut_Subir_TP_E1_E3 THEN #EstadoVI.Error_Mx := TRUE; END_IF;
END_REGION

REGION Network 90: ERROR - Tout subir TP02
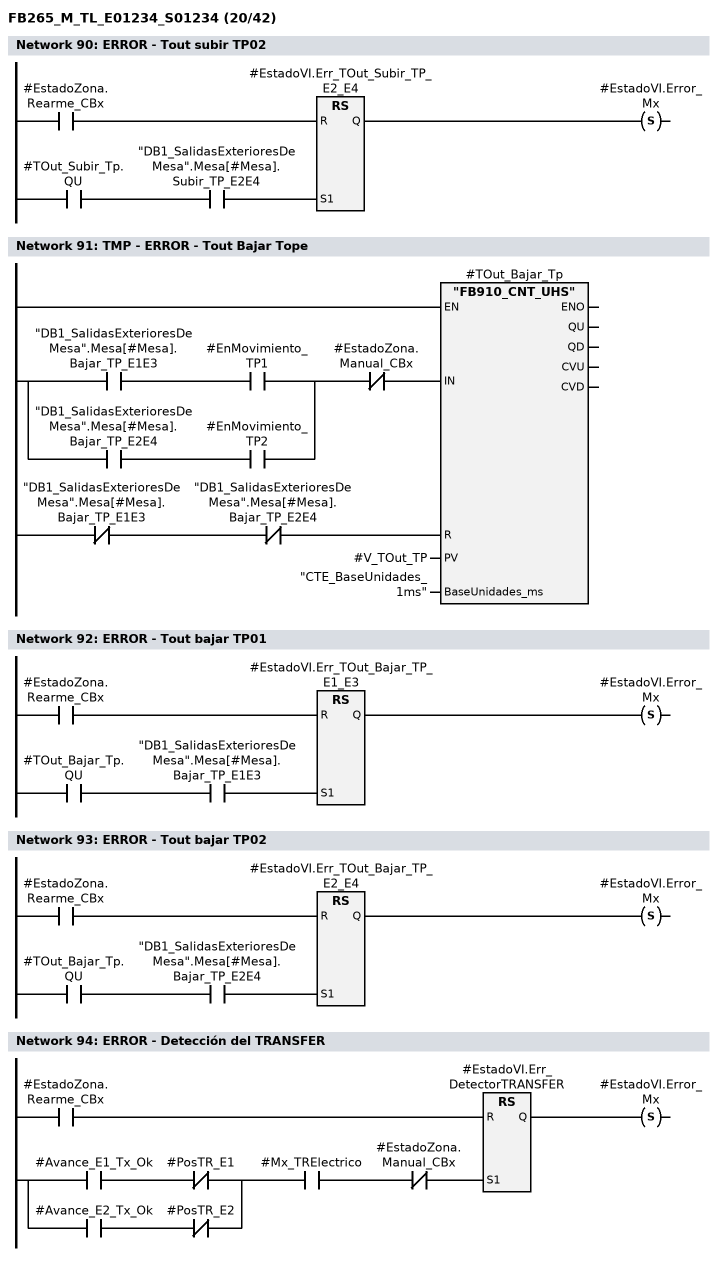
   RUNG wire#powerrail
      Contact( #EstadoZona.Rearme_CBx )
      S_RS(operand := #EstadoVI.Err_TOut_Subir_TP_E2_E4, s1 := wire#w1)
      S_Coil( #EstadoVI.Error_Mx )
   END_RUNG
   RUNG wire#powerrail
      Contact( #TOut_Subir_Tp.QU )
      Contact( "DB1_SalidasExterioresDeMesa".Mesa[#Mesa].Subir_TP_E2E4 )
   END_RUNG wire#w1
   // the same network as SCL:
   IF #EstadoZona.Rearme_CBx THEN
       #EstadoVI.Err_TOut_Subir_TP_E2_E4 := FALSE;   // RS flip-flop
   END_IF;
   IF #TOut_Subir_Tp.QU AND "DB1_SalidasExterioresDeMesa".Mesa[#Mesa].Subir_TP_E2E4 THEN
       #EstadoVI.Err_TOut_Subir_TP_E2_E4 := TRUE;
   END_IF;
   IF #EstadoVI.Err_TOut_Subir_TP_E2_E4 THEN #EstadoVI.Error_Mx := TRUE; END_IF;
END_REGION

REGION Network 91: TMP - ERROR - Tout Bajar Tope
   RUNG wire#powerrail
      #TOut_Bajar_Tp(IN := wire#w2, R := wire#w3, PV := #V_TOut_TP, BaseUnidades_ms := "CTE_BaseUnidades_1ms", QU =>, QD =>, CVU =>, CVD =>)
   END_RUNG
   RUNG wire#powerrail
      Contact( "DB1_SalidasExterioresDeMesa".Mesa[#Mesa].Bajar_TP_E1E3 )
      Contact( #EnMovimiento_TP1 )
      wire#w1
      I_Contact( #EstadoZona.Manual_CBx )
   END_RUNG wire#w2
   RUNG wire#powerrail
      Contact( "DB1_SalidasExterioresDeMesa".Mesa[#Mesa].Bajar_TP_E2E4 )
      Contact( #EnMovimiento_TP2 )
   END_RUNG wire#w1
   RUNG wire#powerrail
      I_Contact( "DB1_SalidasExterioresDeMesa".Mesa[#Mesa].Bajar_TP_E1E3 )
      I_Contact( "DB1_SalidasExterioresDeMesa".Mesa[#Mesa].Bajar_TP_E2E4 )
   END_RUNG wire#w3
   // the same network as SCL:
   #TOut_Bajar_Tp(IN := (("DB1_SalidasExterioresDeMesa".Mesa[#Mesa].Bajar_TP_E1E3 AND #EnMovimiento_TP1) OR ("DB1_SalidasExterioresDeMesa".Mesa[#Mesa].Bajar_TP_E2E4 AND #EnMovimiento_TP2)) AND NOT #EstadoZona.Manual_CBx,   // "FB910_CNT_UHS"
                  R := NOT "DB1_SalidasExterioresDeMesa".Mesa[#Mesa].Bajar_TP_E1E3 AND NOT "DB1_SalidasExterioresDeMesa".Mesa[#Mesa].Bajar_TP_E2E4,
                  PV := #V_TOut_TP,
                  BaseUnidades_ms := "CTE_BaseUnidades_1ms");
END_REGION

REGION Network 92: ERROR - Tout bajar TP01
   RUNG wire#powerrail
      Contact( #EstadoZona.Rearme_CBx )
      S_RS(operand := #EstadoVI.Err_TOut_Bajar_TP_E1_E3, s1 := wire#w1)
      S_Coil( #EstadoVI.Error_Mx )
   END_RUNG
   RUNG wire#powerrail
      Contact( #TOut_Bajar_Tp.QU )
      Contact( "DB1_SalidasExterioresDeMesa".Mesa[#Mesa].Bajar_TP_E1E3 )
   END_RUNG wire#w1
   // the same network as SCL:
   IF #EstadoZona.Rearme_CBx THEN
       #EstadoVI.Err_TOut_Bajar_TP_E1_E3 := FALSE;   // RS flip-flop
   END_IF;
   IF #TOut_Bajar_Tp.QU AND "DB1_SalidasExterioresDeMesa".Mesa[#Mesa].Bajar_TP_E1E3 THEN
       #EstadoVI.Err_TOut_Bajar_TP_E1_E3 := TRUE;
   END_IF;
   IF #EstadoVI.Err_TOut_Bajar_TP_E1_E3 THEN #EstadoVI.Error_Mx := TRUE; END_IF;
END_REGION

REGION Network 93: ERROR - Tout bajar TP02
   RUNG wire#powerrail
      Contact( #EstadoZona.Rearme_CBx )
      S_RS(operand := #EstadoVI.Err_TOut_Bajar_TP_E2_E4, s1 := wire#w1)
      S_Coil( #EstadoVI.Error_Mx )
   END_RUNG
   RUNG wire#powerrail
      Contact( #TOut_Bajar_Tp.QU )
      Contact( "DB1_SalidasExterioresDeMesa".Mesa[#Mesa].Bajar_TP_E2E4 )
   END_RUNG wire#w1
   // the same network as SCL:
   IF #EstadoZona.Rearme_CBx THEN
       #EstadoVI.Err_TOut_Bajar_TP_E2_E4 := FALSE;   // RS flip-flop
   END_IF;
   IF #TOut_Bajar_Tp.QU AND "DB1_SalidasExterioresDeMesa".Mesa[#Mesa].Bajar_TP_E2E4 THEN
       #EstadoVI.Err_TOut_Bajar_TP_E2_E4 := TRUE;
   END_IF;
   IF #EstadoVI.Err_TOut_Bajar_TP_E2_E4 THEN #EstadoVI.Error_Mx := TRUE; END_IF;
END_REGION

REGION Network 94: ERROR - Detección del TRANSFER
   RUNG wire#powerrail
      Contact( #EstadoZona.Rearme_CBx )
      S_RS(operand := #EstadoVI.Err_DetectorTRANSFER, s1 := wire#w2)
      S_Coil( #EstadoVI.Error_Mx )
   END_RUNG
   RUNG wire#powerrail
      Contact( #Avance_E1_Tx_Ok )
      I_Contact( #PosTR_E1 )
      wire#w1
      Contact( #Mx_TRElectrico )
      I_Contact( #EstadoZona.Manual_CBx )
   END_RUNG wire#w2
   RUNG wire#powerrail
      Contact( #Avance_E2_Tx_Ok )
      I_Contact( #PosTR_E2 )
   END_RUNG wire#w1
   // the same network as SCL:
   IF #EstadoZona.Rearme_CBx THEN
       #EstadoVI.Err_DetectorTRANSFER := FALSE;   // RS flip-flop
   END_IF;
   IF ((#Avance_E1_Tx_Ok AND NOT #PosTR_E1) OR (#Avance_E2_Tx_Ok AND NOT #PosTR_E2)) AND #Mx_TRElectrico AND NOT #EstadoZona.Manual_CBx THEN
       #EstadoVI.Err_DetectorTRANSFER := TRUE;
   END_IF;
   IF #EstadoVI.Err_DetectorTRANSFER THEN #EstadoVI.Error_Mx := TRUE; END_IF;
END_REGION

REGION Network 95: CONTADOR DE SEGURIDAD DE PRESENCIA - CNTSeg_pHsMx_E1E3
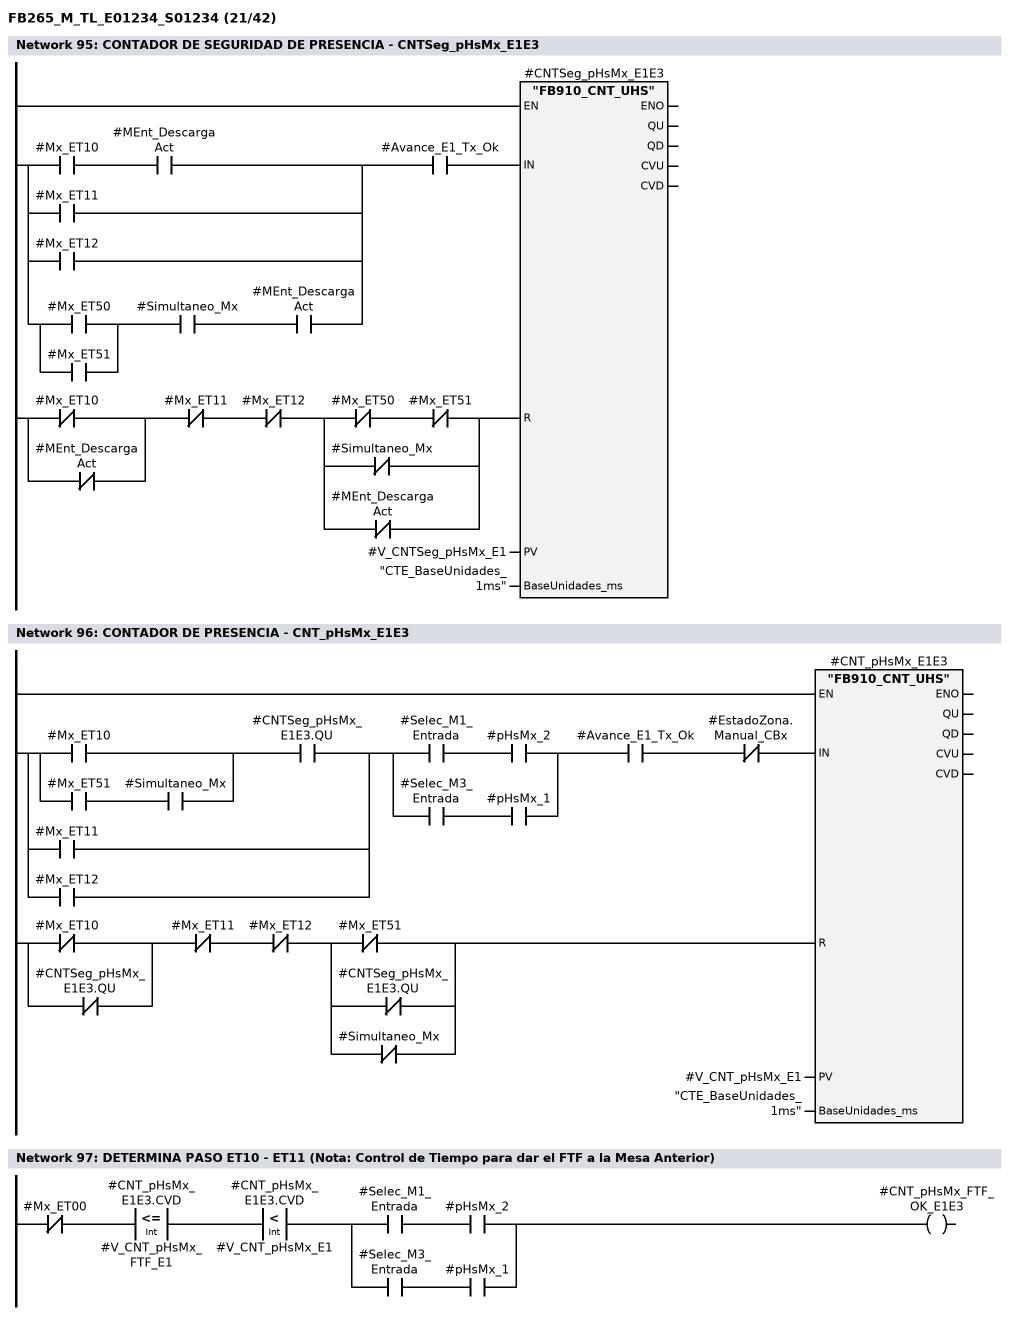
   RUNG wire#powerrail
      #CNTSeg_pHsMx_E1E3(IN := wire#w3, R := wire#w6, PV := #V_CNTSeg_pHsMx_E1, BaseUnidades_ms := "CTE_BaseUnidades_1ms", QU =>, QD =>, CVU =>, CVD =>)
   END_RUNG
   RUNG wire#powerrail
      Contact( #Mx_ET10 )
      Contact( #MEnt_DescargaAct )
      wire#w1
      Contact( #Avance_E1_Tx_Ok )
   END_RUNG wire#w3
   RUNG wire#powerrail
      Contact( #Mx_ET11 )
   END_RUNG wire#w1
   RUNG wire#powerrail
      Contact( #Mx_ET12 )
   END_RUNG wire#w1
   RUNG wire#powerrail
      Contact( #Mx_ET50 )
      wire#w2
      Contact( #Simultaneo_Mx )
      Contact( #MEnt_DescargaAct )
   END_RUNG wire#w1
   RUNG wire#powerrail
      Contact( #Mx_ET51 )
   END_RUNG wire#w2
   RUNG wire#powerrail
      I_Contact( #Mx_ET10 )
      wire#w4
      I_Contact( #Mx_ET11 )
      I_Contact( #Mx_ET12 )
      wire#w5
      I_Contact( #Mx_ET50 )
      I_Contact( #Mx_ET51 )
   END_RUNG wire#w6
   RUNG wire#powerrail
      I_Contact( #MEnt_DescargaAct )
   END_RUNG wire#w4
   RUNG wire#w5
      I_Contact( #Simultaneo_Mx )
   END_RUNG wire#w6
   RUNG wire#w5
      I_Contact( #MEnt_DescargaAct )
   END_RUNG wire#w6
   // the same network as SCL:
   #CNTSeg_pHsMx_E1E3(IN := ((#Mx_ET10 AND #MEnt_DescargaAct) OR #Mx_ET11 OR #Mx_ET12 OR ((#Mx_ET50 OR #Mx_ET51) AND #Simultaneo_Mx AND #MEnt_DescargaAct)) AND #Avance_E1_Tx_Ok,   // "FB910_CNT_UHS"
                      R := (NOT #Mx_ET10 OR NOT #MEnt_DescargaAct) AND NOT #Mx_ET11 AND NOT #Mx_ET12 AND ((NOT #Mx_ET50 AND NOT #Mx_ET51) OR NOT #Simultaneo_Mx OR NOT #MEnt_DescargaAct),
                      PV := #V_CNTSeg_pHsMx_E1,
                      BaseUnidades_ms := "CTE_BaseUnidades_1ms");
END_REGION

